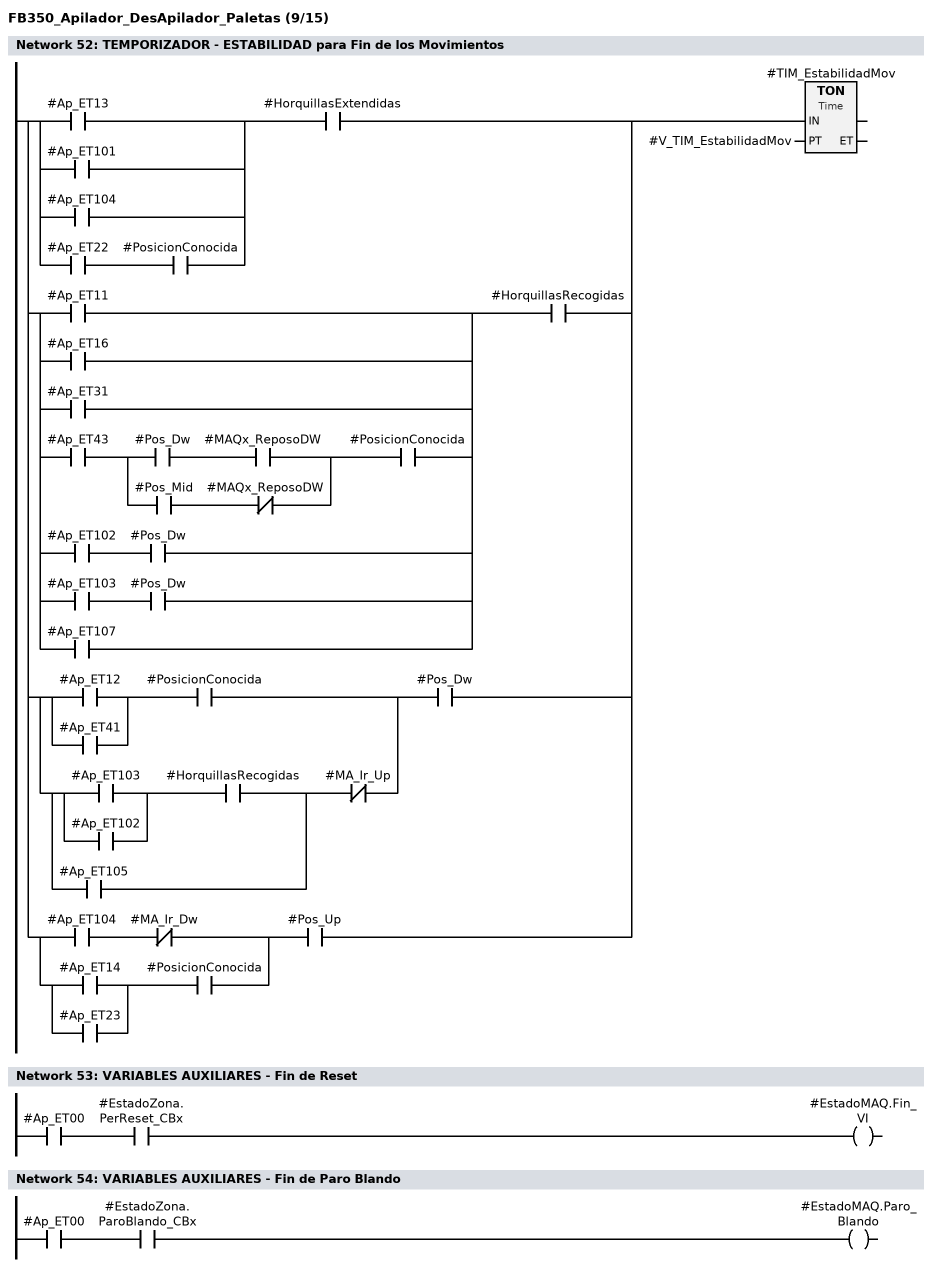
   RUNG wire#powerrail
      Contact( #Ap_ET13 )
      wire#w1
      Contact( #HorquillasExtendidas )
      wire#w2
      { S7_Templates := "time_type := Time" } #TIM_EstabilidadMov.TON(pt := #V_TIM_EstabilidadMov, et =>)
   END_RUNG
   RUNG wire#powerrail
      Contact( #Ap_ET101 )
   END_RUNG wire#w1
   RUNG wire#powerrail
      Contact( #Ap_ET104 )
   END_RUNG wire#w1
   RUNG wire#powerrail
      Contact( #Ap_ET22 )
      Contact( #PosicionConocida )
   END_RUNG wire#w1
   RUNG wire#powerrail
      Contact( #Ap_ET11 )
      wire#w3
      Contact( #HorquillasRecogidas )
   END_RUNG wire#w2
   RUNG wire#powerrail
      Contact( #Ap_ET16 )
   END_RUNG wire#w3
   RUNG wire#powerrail
      Contact( #Ap_ET31 )
   END_RUNG wire#w3
   RUNG wire#powerrail
      Contact( #Ap_ET43 )
      wire#w4
      Contact( #Pos_Dw )
      Contact( #MAQx_ReposoDW )
      wire#w5
      Contact( #PosicionConocida )
   END_RUNG wire#w3
   RUNG wire#w4
      Contact( #Pos_Mid )
      I_Contact( #MAQx_ReposoDW )
   END_RUNG wire#w5
   RUNG wire#powerrail
      Contact( #Ap_ET102 )
      Contact( #Pos_Dw )
   END_RUNG wire#w3
   RUNG wire#powerrail
      Contact( #Ap_ET103 )
      Contact( #Pos_Dw )
   END_RUNG wire#w3
   RUNG wire#powerrail
      Contact( #Ap_ET107 )
   END_RUNG wire#w3
   RUNG wire#powerrail
      Contact( #Ap_ET12 )
      wire#w6
      Contact( #PosicionConocida )
      wire#w7
      Contact( #Pos_Dw )
   END_RUNG wire#w2
   RUNG wire#powerrail
      Contact( #Ap_ET41 )
   END_RUNG wire#w6
   RUNG wire#powerrail
      Contact( #Ap_ET103 )
      wire#w8
      Contact( #HorquillasRecogidas )
      wire#w9
      I_Contact( #MA_Ir_Up )
   END_RUNG wire#w7
   RUNG wire#powerrail
      Contact( #Ap_ET102 )
   END_RUNG wire#w8
   RUNG wire#powerrail
      Contact( #Ap_ET105 )
   END_RUNG wire#w9
   RUNG wire#powerrail
      Contact( #Ap_ET104 )
      I_Contact( #MA_Ir_Dw )
      wire#w10
      Contact( #Pos_Up )
   END_RUNG wire#w2
   RUNG wire#powerrail
      Contact( #Ap_ET14 )
      wire#w11
      Contact( #PosicionConocida )
   END_RUNG wire#w10
   RUNG wire#powerrail
      Contact( #Ap_ET23 )
   END_RUNG wire#w11
   // the same network as SCL:
   #TIM_EstabilidadMov(IN := ((#Ap_ET13 OR #Ap_ET101 OR #Ap_ET104 OR (#Ap_ET22 AND #PosicionConocida)) AND #HorquillasExtendidas) OR ((#Ap_ET11 OR #Ap_ET16 OR #Ap_ET31 OR (#Ap_ET43 AND ((#Pos_Dw AND #MAQx_ReposoDW) OR (#Pos_Mid AND NOT #MAQx_ReposoDW)) AND #PosicionConocida) OR (#Ap_ET102 AND #Pos_Dw) OR (#Ap_ET103 AND #Pos_Dw) OR #Ap_ET107) AND #HorquillasRecogidas) OR ((((#Ap_ET12 OR #Ap_ET41) AND #PosicionConocida) OR ((((#Ap_ET103 OR #Ap_ET102) AND #HorquillasRecogidas) OR #Ap_ET105) AND NOT #MA_Ir_Up)) AND #Pos_Dw) OR (((#Ap_ET104 AND NOT #MA_Ir_Dw) OR ((#Ap_ET14 OR #Ap_ET23) AND #PosicionConocida)) AND #Pos_Up),   // TON
                       PT := #V_TIM_EstabilidadMov);
END_REGION

REGION Network 53: VARIABLES AUXILIARES - Fin de Reset
   RUNG wire#powerrail
      Contact( #Ap_ET00 )
      Contact( #EstadoZona.PerReset_CBx )
      Coil( #EstadoMAQ.Fin_VI )
   END_RUNG
   // the same network as SCL:
   #EstadoMAQ.Fin_VI := #Ap_ET00 AND #EstadoZona.PerReset_CBx;
END_REGION

REGION Network 54: VARIABLES AUXILIARES - Fin de Paro Blando
   RUNG wire#powerrail
      Contact( #Ap_ET00 )
      Contact( #EstadoZona.ParoBlando_CBx )
      Coil( #EstadoMAQ.Paro_Blando )
   END_RUNG
   // the same network as SCL:
   #EstadoMAQ.Paro_Blando := #Ap_ET00 AND #EstadoZona.ParoBlando_CBx;
END_REGION

REGION Network 55: VARIABLES AUXILIARES - Posicion Conocida
   // MODIFICACION DANI: SI MUEVO EN MANUAL NO PIERDE LA POSCION
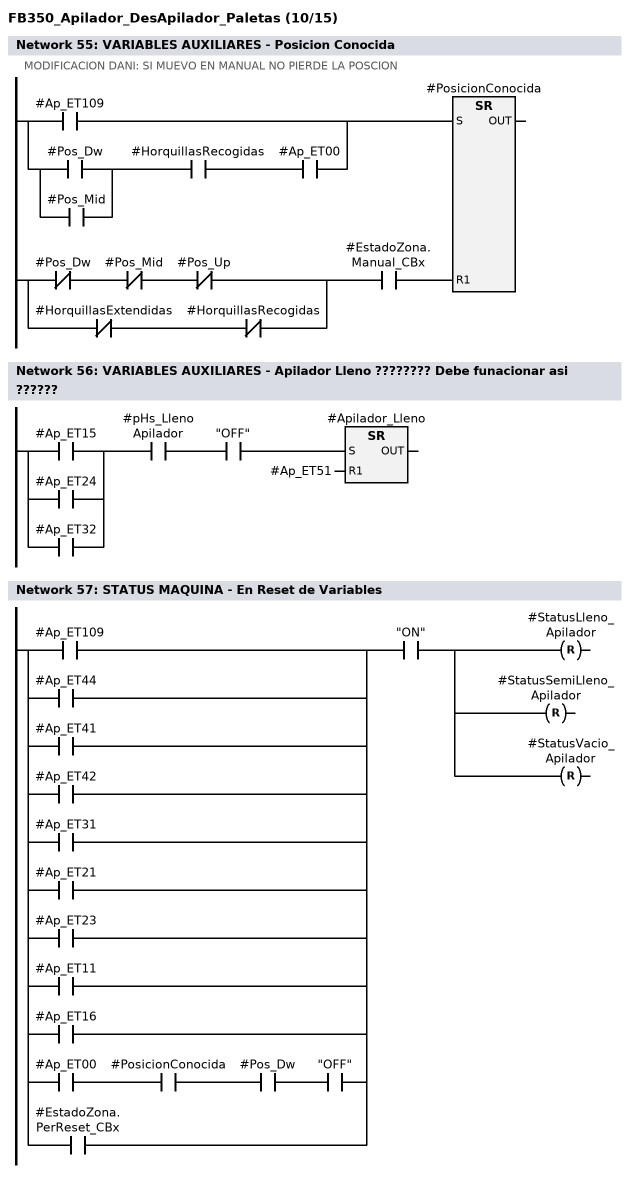
   RUNG wire#powerrail
      Contact( #Ap_ET109 )
      wire#w1
      S_SR(operand := #PosicionConocida, r1 := wire#w4)
   END_RUNG
   RUNG wire#powerrail
      Contact( #Pos_Dw )
      wire#w2
      Contact( #HorquillasRecogidas )
      Contact( #Ap_ET00 )
   END_RUNG wire#w1
   RUNG wire#powerrail
      Contact( #Pos_Mid )
   END_RUNG wire#w2
   RUNG wire#powerrail
      I_Contact( #Pos_Dw )
      I_Contact( #Pos_Mid )
      I_Contact( #Pos_Up )
      wire#w3
      Contact( #EstadoZona.Manual_CBx )
   END_RUNG wire#w4
   RUNG wire#powerrail
      I_Contact( #HorquillasExtendidas )
      I_Contact( #HorquillasRecogidas )
   END_RUNG wire#w3
   // the same network as SCL:
   IF #Ap_ET109 OR ((#Pos_Dw OR #Pos_Mid) AND #HorquillasRecogidas AND #Ap_ET00) THEN
       #PosicionConocida := TRUE;   // SR flip-flop
   END_IF;
   IF ((NOT #Pos_Dw AND NOT #Pos_Mid AND NOT #Pos_Up) OR (NOT #HorquillasExtendidas AND NOT #HorquillasRecogidas)) AND #EstadoZona.Manual_CBx THEN
       #PosicionConocida := FALSE;
   END_IF;
END_REGION

REGION Network 56: VARIABLES AUXILIARES - Apilador Lleno ???????? Debe funacionar asi ??????
   RUNG wire#powerrail
      Contact( #Ap_ET15 )
      wire#w1
      Contact( #pHs_LlenoApilador )
      Contact( "OFF" )
      S_SR(operand := #Apilador_Lleno, r1 := #Ap_ET51)
   END_RUNG
   RUNG wire#powerrail
      Contact( #Ap_ET24 )
   END_RUNG wire#w1
   RUNG wire#powerrail
      Contact( #Ap_ET32 )
   END_RUNG wire#w1
   // the same network as SCL:
   IF (#Ap_ET15 OR #Ap_ET24 OR #Ap_ET32) AND #pHs_LlenoApilador AND "OFF" THEN
       #Apilador_Lleno := TRUE;   // SR flip-flop
   END_IF;
   IF #Ap_ET51 THEN #Apilador_Lleno := FALSE; END_IF;
END_REGION

REGION Network 57: STATUS MAQUINA - En Reset de Variables
   RUNG wire#powerrail
      Contact( #Ap_ET109 )
      wire#w1
      Contact( "ON" )
      wire#w2
      R_Coil( #StatusLleno_Apilador )
   END_RUNG
   RUNG wire#powerrail
      Contact( #Ap_ET44 )
   END_RUNG wire#w1
   RUNG wire#powerrail
      Contact( #Ap_ET41 )
   END_RUNG wire#w1
   RUNG wire#powerrail
      Contact( #Ap_ET42 )
   END_RUNG wire#w1
   RUNG wire#powerrail
      Contact( #Ap_ET31 )
   END_RUNG wire#w1
   RUNG wire#powerrail
      Contact( #Ap_ET21 )
   END_RUNG wire#w1
   RUNG wire#powerrail
      Contact( #Ap_ET23 )
   END_RUNG wire#w1
   RUNG wire#powerrail
      Contact( #Ap_ET11 )
   END_RUNG wire#w1
   RUNG wire#powerrail
      Contact( #Ap_ET16 )
   END_RUNG wire#w1
   RUNG wire#powerrail
      Contact( #Ap_ET00 )
      Contact( #PosicionConocida )
      Contact( #Pos_Dw )
      Contact( "OFF" )
   END_RUNG wire#w1
   RUNG wire#powerrail
      Contact( #EstadoZona.PerReset_CBx )
   END_RUNG wire#w1
   RUNG wire#w2
      R_Coil( #StatusSemiLleno_Apilador )
   END_RUNG
   RUNG wire#w2
      R_Coil( #StatusVacio_Apilador )
   END_RUNG
   // the same network as SCL:
   IF (#Ap_ET109 OR #Ap_ET44 OR #Ap_ET41 OR #Ap_ET42 OR #Ap_ET31 OR #Ap_ET21 OR #Ap_ET23 OR #Ap_ET11 OR #Ap_ET16 OR (#Ap_ET00 AND #PosicionConocida AND #Pos_Dw AND "OFF") OR #EstadoZona.PerReset_CBx) AND "ON" THEN
       #StatusLleno_Apilador := FALSE;
       #StatusSemiLleno_Apilador := FALSE;
       #StatusVacio_Apilador := FALSE;
   END_IF;
END_REGION

REGION Network 58: STATUS MAQUINA - En set de Variables
   // DANI SI ESTA EN ETAPA 0, POS CONOCIDA Y POS REPOSO ACTUALICE EL ESTATUS
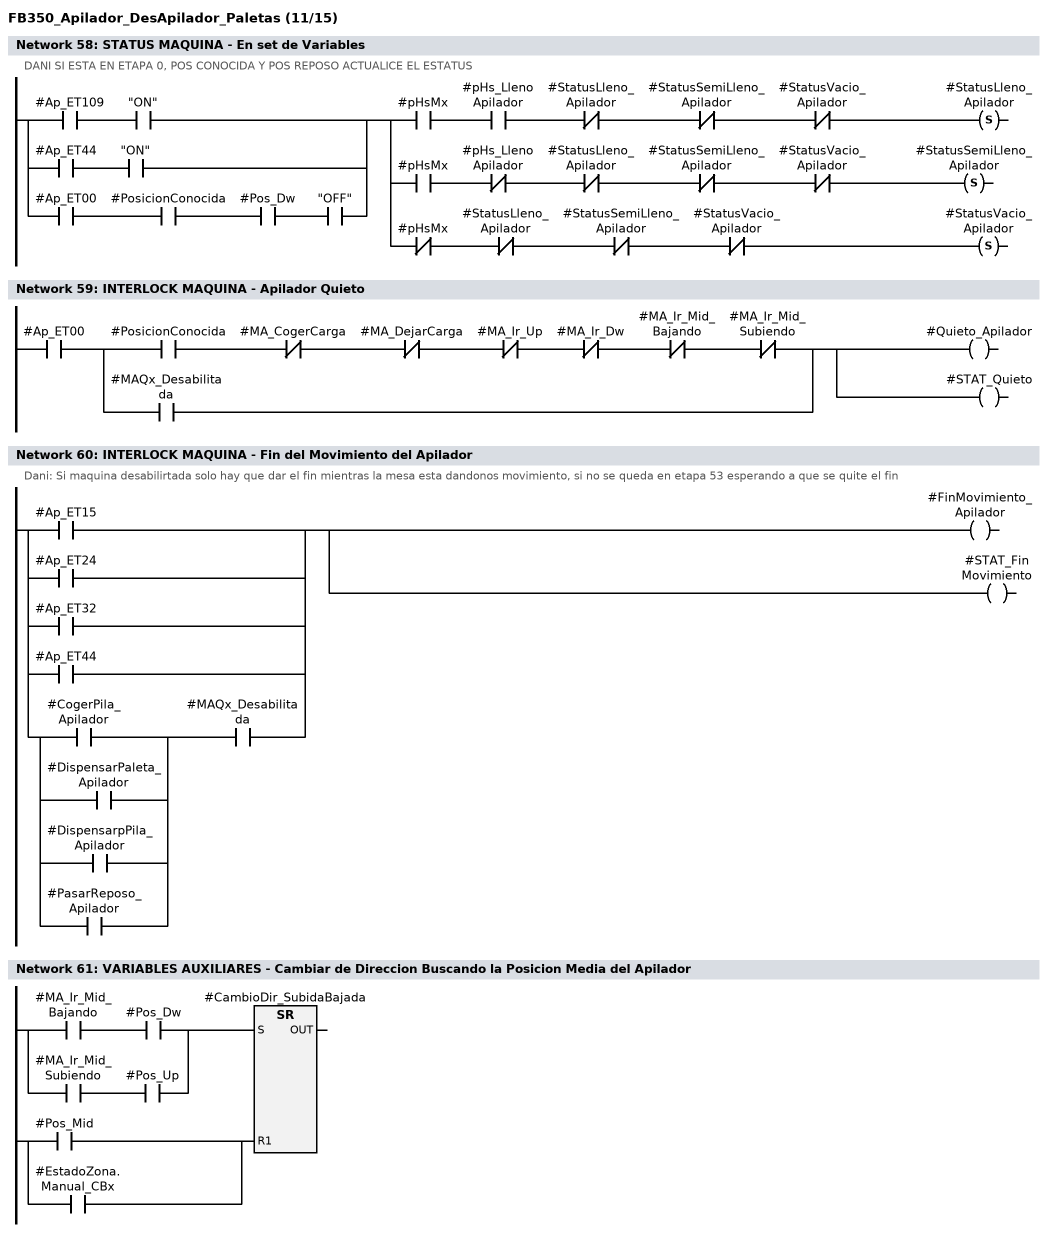
   RUNG wire#powerrail
      Contact( #Ap_ET109 )
      Contact( "ON" )
      wire#w1
      Contact( #pHsMx )
      Contact( #pHs_LlenoApilador )
      I_Contact( #StatusLleno_Apilador )
      I_Contact( #StatusSemiLleno_Apilador )
      I_Contact( #StatusVacio_Apilador )
      S_Coil( #StatusLleno_Apilador )
   END_RUNG
   RUNG wire#powerrail
      Contact( #Ap_ET44 )
      Contact( "ON" )
   END_RUNG wire#w1
   RUNG wire#powerrail
      Contact( #Ap_ET00 )
      Contact( #PosicionConocida )
      Contact( #Pos_Dw )
      Contact( "OFF" )
   END_RUNG wire#w1
   RUNG wire#w1
      Contact( #pHsMx )
      I_Contact( #pHs_LlenoApilador )
      I_Contact( #StatusLleno_Apilador )
      I_Contact( #StatusSemiLleno_Apilador )
      I_Contact( #StatusVacio_Apilador )
      S_Coil( #StatusSemiLleno_Apilador )
   END_RUNG
   RUNG wire#w1
      I_Contact( #pHsMx )
      I_Contact( #StatusLleno_Apilador )
      I_Contact( #StatusSemiLleno_Apilador )
      I_Contact( #StatusVacio_Apilador )
      S_Coil( #StatusVacio_Apilador )
   END_RUNG
   // the same network as SCL:
   #_w1 := (#Ap_ET109 AND "ON") OR (#Ap_ET44 AND "ON") OR (#Ap_ET00 AND #PosicionConocida AND #Pos_Dw AND "OFF");
   IF #_w1 AND #pHsMx AND #pHs_LlenoApilador AND NOT #StatusLleno_Apilador AND NOT #StatusSemiLleno_Apilador AND NOT #StatusVacio_Apilador THEN
       #StatusLleno_Apilador := TRUE;
   END_IF;
   IF #_w1 AND #pHsMx AND NOT #pHs_LlenoApilador AND NOT #StatusLleno_Apilador AND NOT #StatusSemiLleno_Apilador AND NOT #StatusVacio_Apilador THEN
       #StatusSemiLleno_Apilador := TRUE;
   END_IF;
   IF #_w1 AND NOT #pHsMx AND NOT #StatusLleno_Apilador AND NOT #StatusSemiLleno_Apilador AND NOT #StatusVacio_Apilador THEN
       #StatusVacio_Apilador := TRUE;
   END_IF;
END_REGION

REGION Network 59: INTERLOCK MAQUINA - Apilador Quieto
   RUNG wire#powerrail
      Contact( #Ap_ET00 )
      wire#w1
      Contact( #PosicionConocida )
      I_Contact( #MA_CogerCarga )
      I_Contact( #MA_DejarCarga )
      I_Contact( #MA_Ir_Up )
      I_Contact( #MA_Ir_Dw )
      I_Contact( #MA_Ir_Mid_Bajando )
      I_Contact( #MA_Ir_Mid_Subiendo )
      wire#w2
      Coil( #Quieto_Apilador )
   END_RUNG
   RUNG wire#w1
      Contact( #MAQx_Desabilitada )
   END_RUNG wire#w2
   RUNG wire#w2
      Coil( #STAT_Quieto )
   END_RUNG
   // the same network as SCL:
   #Quieto_Apilador := #Ap_ET00 AND ((#PosicionConocida AND NOT #MA_CogerCarga AND NOT #MA_DejarCarga AND NOT #MA_Ir_Up AND NOT #MA_Ir_Dw AND NOT #MA_Ir_Mid_Bajando AND NOT #MA_Ir_Mid_Subiendo) OR #MAQx_Desabilitada);
   #STAT_Quieto := #Quieto_Apilador;
END_REGION

REGION Network 60: INTERLOCK MAQUINA - Fin del Movimiento del Apilador
   // Dani: Si maquina desabilirtada solo hay que dar el fin mientras la mesa esta dandonos movimiento, si no se queda en etapa 53 esperando a que se quite el fin
   RUNG wire#powerrail
      Contact( #Ap_ET15 )
      wire#w1
      Coil( #FinMovimiento_Apilador )
   END_RUNG
   RUNG wire#powerrail
      Contact( #Ap_ET24 )
   END_RUNG wire#w1
   RUNG wire#powerrail
      Contact( #Ap_ET32 )
   END_RUNG wire#w1
   RUNG wire#powerrail
      Contact( #Ap_ET44 )
   END_RUNG wire#w1
   RUNG wire#powerrail
      Contact( #CogerPila_Apilador )
      wire#w2
      Contact( #MAQx_Desabilitada )
   END_RUNG wire#w1
   RUNG wire#powerrail
      Contact( #DispensarPaleta_Apilador )
   END_RUNG wire#w2
   RUNG wire#powerrail
      Contact( #DispensarpPila_Apilador )
   END_RUNG wire#w2
   RUNG wire#powerrail
      Contact( #PasarReposo_Apilador )
   END_RUNG wire#w2
   RUNG wire#w1
      Coil( #STAT_FinMovimiento )
   END_RUNG
   // the same network as SCL:
   #FinMovimiento_Apilador := #Ap_ET15 OR #Ap_ET24 OR #Ap_ET32 OR #Ap_ET44 OR ((#CogerPila_Apilador OR #DispensarPaleta_Apilador OR #DispensarpPila_Apilador OR #PasarReposo_Apilador) AND #MAQx_Desabilitada);
   #STAT_FinMovimiento := #FinMovimiento_Apilador;
END_REGION

REGION Network 61: VARIABLES AUXILIARES - Cambiar de Direccion Buscando la Posicion Media del Apilador
   RUNG wire#powerrail
      Contact( #MA_Ir_Mid_Bajando )
      Contact( #Pos_Dw )
      wire#w1
      S_SR(operand := #CambioDir_SubidaBajada, r1 := wire#w2)
   END_RUNG
   RUNG wire#powerrail
      Contact( #MA_Ir_Mid_Subiendo )
      Contact( #Pos_Up )
   END_RUNG wire#w1
   RUNG wire#powerrail
      Contact( #Pos_Mid )
   END_RUNG wire#w2
   RUNG wire#powerrail
      Contact( #EstadoZona.Manual_CBx )
   END_RUNG wire#w2
   // the same network as SCL:
   IF (#MA_Ir_Mid_Bajando AND #Pos_Dw) OR (#MA_Ir_Mid_Subiendo AND #Pos_Up) THEN
       #CambioDir_SubidaBajada := TRUE;   // SR flip-flop
   END_IF;
   IF #Pos_Mid OR #EstadoZona.Manual_CBx THEN #CambioDir_SubidaBajada := FALSE; END_IF;
END_REGION

REGION Network 62: SALIDAS EXTERIORES - Hoquilla - Coger Carga / Extender 4 Horquillas
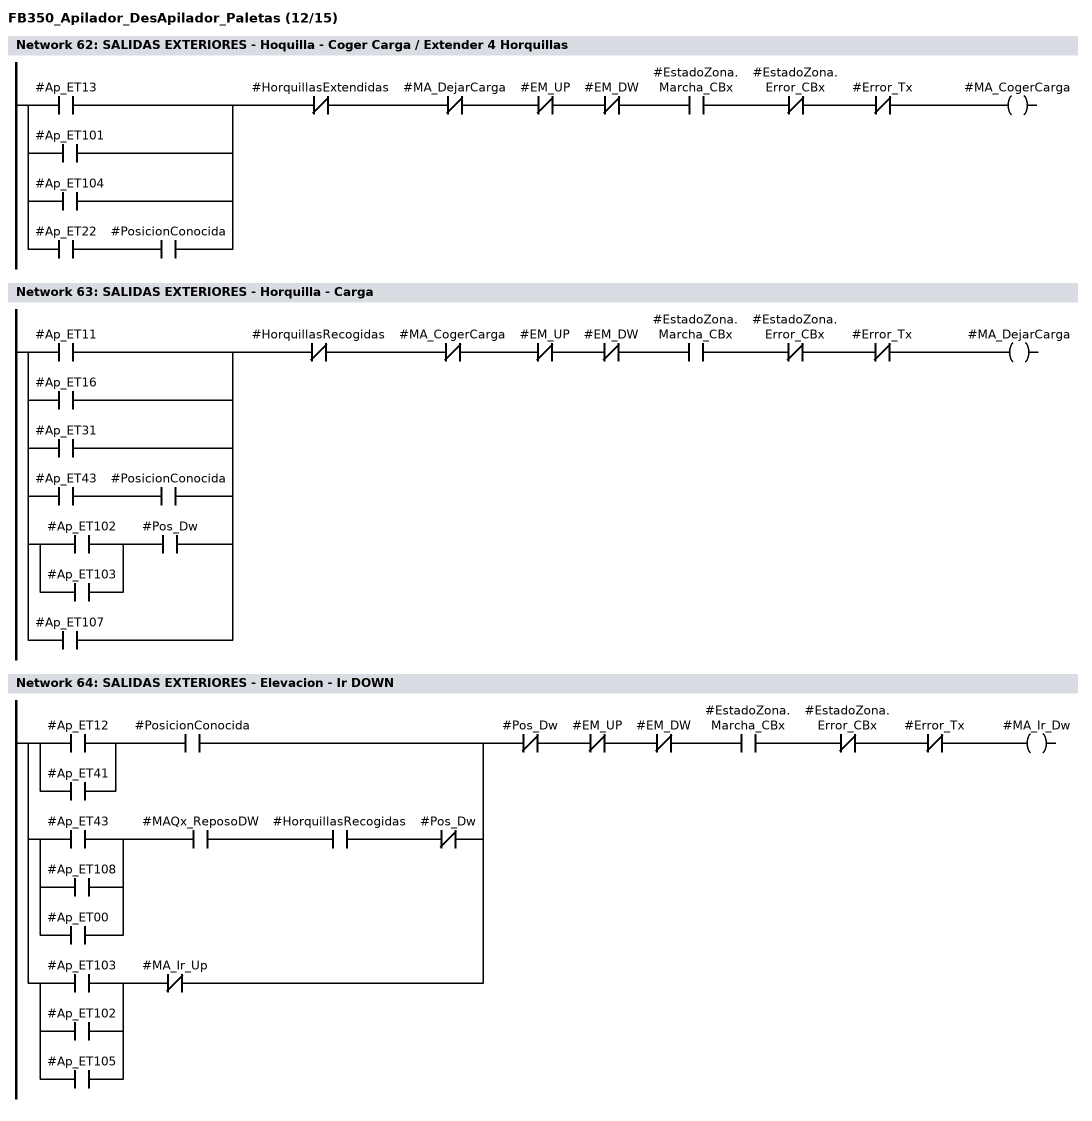
   RUNG wire#powerrail
      Contact( #Ap_ET13 )
      wire#w1
      I_Contact( #HorquillasExtendidas )
      I_Contact( #MA_DejarCarga )
      I_Contact( #EM_UP )
      I_Contact( #EM_DW )
      Contact( #EstadoZona.Marcha_CBx )
      I_Contact( #EstadoZona.Error_CBx )
      I_Contact( #Error_Tx )
      Coil( #MA_CogerCarga )
   END_RUNG
   RUNG wire#powerrail
      Contact( #Ap_ET101 )
   END_RUNG wire#w1
   RUNG wire#powerrail
      Contact( #Ap_ET104 )
   END_RUNG wire#w1
   RUNG wire#powerrail
      Contact( #Ap_ET22 )
      Contact( #PosicionConocida )
   END_RUNG wire#w1
   // the same network as SCL:
   #MA_CogerCarga := (#Ap_ET13 OR #Ap_ET101 OR #Ap_ET104 OR (#Ap_ET22 AND #PosicionConocida)) AND NOT #HorquillasExtendidas AND NOT #MA_DejarCarga AND NOT #EM_UP AND NOT #EM_DW AND #EstadoZona.Marcha_CBx AND NOT #EstadoZona.Error_CBx AND NOT #Error_Tx;
END_REGION

REGION Network 63: SALIDAS EXTERIORES - Horquilla - Carga
   RUNG wire#powerrail
      Contact( #Ap_ET11 )
      wire#w1
      I_Contact( #HorquillasRecogidas )
      I_Contact( #MA_CogerCarga )
      I_Contact( #EM_UP )
      I_Contact( #EM_DW )
      Contact( #EstadoZona.Marcha_CBx )
      I_Contact( #EstadoZona.Error_CBx )
      I_Contact( #Error_Tx )
      Coil( #MA_DejarCarga )
   END_RUNG
   RUNG wire#powerrail
      Contact( #Ap_ET16 )
   END_RUNG wire#w1
   RUNG wire#powerrail
      Contact( #Ap_ET31 )
   END_RUNG wire#w1
   RUNG wire#powerrail
      Contact( #Ap_ET43 )
      Contact( #PosicionConocida )
   END_RUNG wire#w1
   RUNG wire#powerrail
      Contact( #Ap_ET102 )
      wire#w2
      Contact( #Pos_Dw )
   END_RUNG wire#w1
   RUNG wire#powerrail
      Contact( #Ap_ET103 )
   END_RUNG wire#w2
   RUNG wire#powerrail
      Contact( #Ap_ET107 )
   END_RUNG wire#w1
   // the same network as SCL:
   #MA_DejarCarga := (#Ap_ET11 OR #Ap_ET16 OR #Ap_ET31 OR (#Ap_ET43 AND #PosicionConocida) OR ((#Ap_ET102 OR #Ap_ET103) AND #Pos_Dw) OR #Ap_ET107) AND NOT #HorquillasRecogidas AND NOT #MA_CogerCarga AND NOT #EM_UP AND NOT #EM_DW AND #EstadoZona.Marcha_CBx AND NOT #EstadoZona.Error_CBx AND NOT #Error_Tx;
END_REGION

REGION Network 64: SALIDAS EXTERIORES - Elevacion - Ir DOWN
   RUNG wire#powerrail
      Contact( #Ap_ET12 )
      wire#w1
      Contact( #PosicionConocida )
      wire#w2
      I_Contact( #Pos_Dw )
      I_Contact( #EM_UP )
      I_Contact( #EM_DW )
      Contact( #EstadoZona.Marcha_CBx )
      I_Contact( #EstadoZona.Error_CBx )
      I_Contact( #Error_Tx )
      Coil( #MA_Ir_Dw )
   END_RUNG
   RUNG wire#powerrail
      Contact( #Ap_ET41 )
   END_RUNG wire#w1
   RUNG wire#powerrail
      Contact( #Ap_ET43 )
      wire#w3
      Contact( #MAQx_ReposoDW )
      Contact( #HorquillasRecogidas )
      I_Contact( #Pos_Dw )
   END_RUNG wire#w2
   RUNG wire#powerrail
      Contact( #Ap_ET108 )
   END_RUNG wire#w3
   RUNG wire#powerrail
      Contact( #Ap_ET00 )
   END_RUNG wire#w3
   RUNG wire#powerrail
      Contact( #Ap_ET103 )
      wire#w4
      I_Contact( #MA_Ir_Up )
   END_RUNG wire#w2
   RUNG wire#powerrail
      Contact( #Ap_ET102 )
   END_RUNG wire#w4
   RUNG wire#powerrail
      Contact( #Ap_ET105 )
   END_RUNG wire#w4
   // the same network as SCL:
   #MA_Ir_Dw := (((#Ap_ET12 OR #Ap_ET41) AND #PosicionConocida) OR ((#Ap_ET43 OR #Ap_ET108 OR #Ap_ET00) AND #MAQx_ReposoDW AND #HorquillasRecogidas AND NOT #Pos_Dw) OR ((#Ap_ET103 OR #Ap_ET102 OR #Ap_ET105) AND NOT #MA_Ir_Up)) AND NOT #Pos_Dw AND NOT #EM_UP AND NOT #EM_DW AND #EstadoZona.Marcha_CBx AND NOT #EstadoZona.Error_CBx AND NOT #Error_Tx;
END_REGION

REGION Network 65: SALIDAS EXTERIORES - Elevacion - Ir MID Bajando
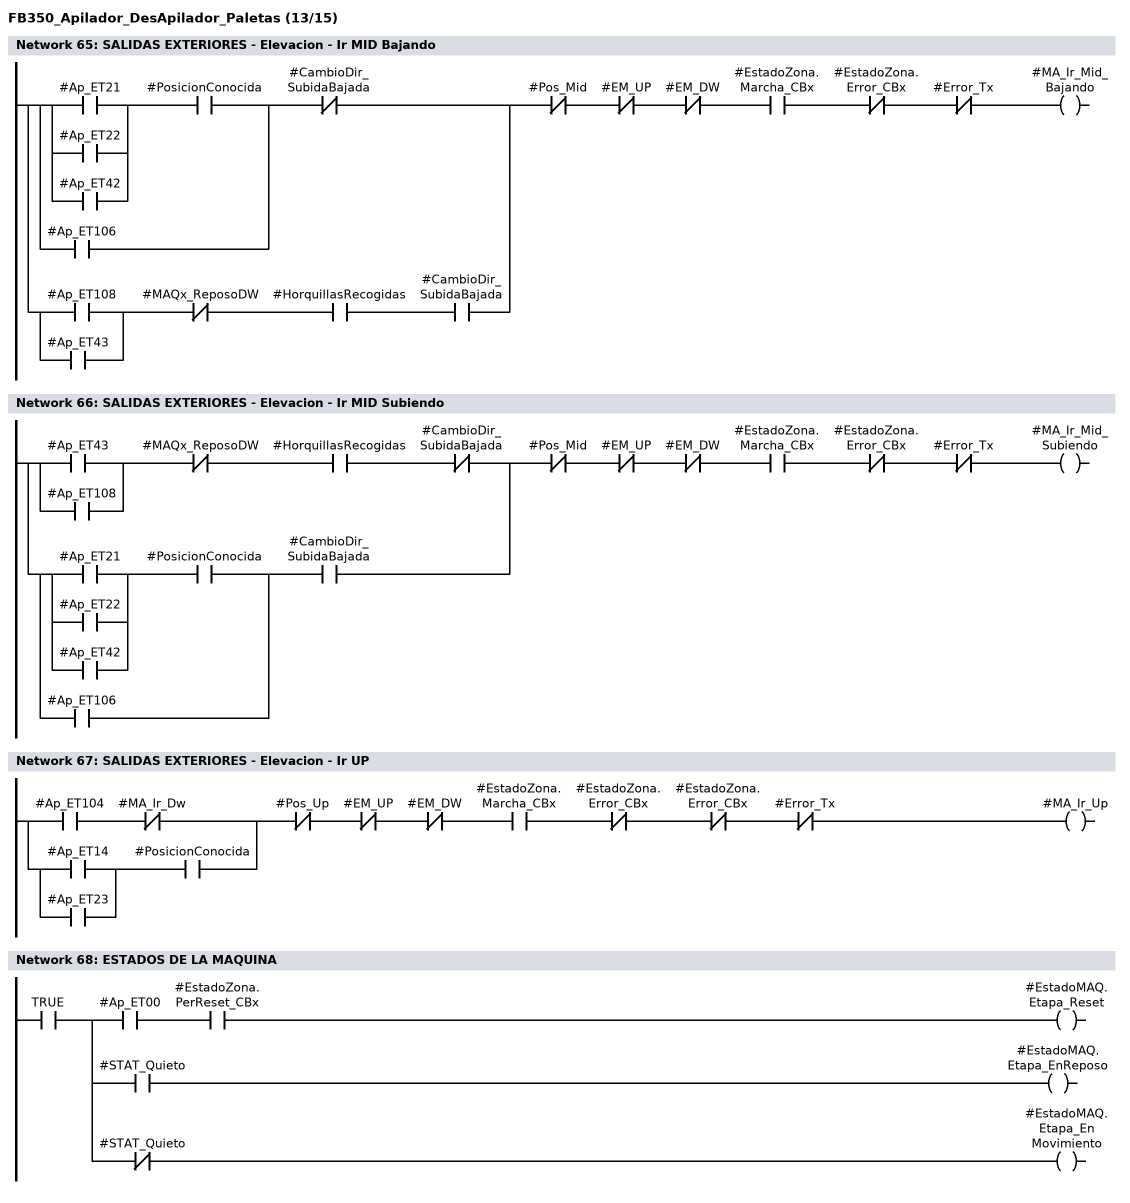
   RUNG wire#powerrail
      Contact( #Ap_ET21 )
      wire#w1
      Contact( #PosicionConocida )
      wire#w2
      I_Contact( #CambioDir_SubidaBajada )
      wire#w3
      I_Contact( #Pos_Mid )
      I_Contact( #EM_UP )
      I_Contact( #EM_DW )
      Contact( #EstadoZona.Marcha_CBx )
      I_Contact( #EstadoZona.Error_CBx )
      I_Contact( #Error_Tx )
      Coil( #MA_Ir_Mid_Bajando )
   END_RUNG
   RUNG wire#powerrail
      Contact( #Ap_ET22 )
   END_RUNG wire#w1
   RUNG wire#powerrail
      Contact( #Ap_ET42 )
   END_RUNG wire#w1
   RUNG wire#powerrail
      Contact( #Ap_ET106 )
   END_RUNG wire#w2
   RUNG wire#powerrail
      Contact( #Ap_ET108 )
      wire#w4
      I_Contact( #MAQx_ReposoDW )
      Contact( #HorquillasRecogidas )
      Contact( #CambioDir_SubidaBajada )
   END_RUNG wire#w3
   RUNG wire#powerrail
      Contact( #Ap_ET43 )
   END_RUNG wire#w4
   // the same network as SCL:
   #MA_Ir_Mid_Bajando := (((((#Ap_ET21 OR #Ap_ET22 OR #Ap_ET42) AND #PosicionConocida) OR #Ap_ET106) AND NOT #CambioDir_SubidaBajada) OR ((#Ap_ET108 OR #Ap_ET43) AND NOT #MAQx_ReposoDW AND #HorquillasRecogidas AND #CambioDir_SubidaBajada)) AND NOT #Pos_Mid AND NOT #EM_UP AND NOT #EM_DW AND #EstadoZona.Marcha_CBx AND NOT #EstadoZona.Error_CBx AND NOT #Error_Tx;
END_REGION

REGION Network 66: SALIDAS EXTERIORES - Elevacion - Ir MID Subiendo
   RUNG wire#powerrail
      Contact( #Ap_ET43 )
      wire#w1
      I_Contact( #MAQx_ReposoDW )
      Contact( #HorquillasRecogidas )
      I_Contact( #CambioDir_SubidaBajada )
      wire#w2
      I_Contact( #Pos_Mid )
      I_Contact( #EM_UP )
      I_Contact( #EM_DW )
      Contact( #EstadoZona.Marcha_CBx )
      I_Contact( #EstadoZona.Error_CBx )
      I_Contact( #Error_Tx )
      Coil( #MA_Ir_Mid_Subiendo )
   END_RUNG
   RUNG wire#powerrail
      Contact( #Ap_ET108 )
   END_RUNG wire#w1
   RUNG wire#powerrail
      Contact( #Ap_ET21 )
      wire#w3
      Contact( #PosicionConocida )
      wire#w4
      Contact( #CambioDir_SubidaBajada )
   END_RUNG wire#w2
   RUNG wire#powerrail
      Contact( #Ap_ET22 )
   END_RUNG wire#w3
   RUNG wire#powerrail
      Contact( #Ap_ET42 )
   END_RUNG wire#w3
   RUNG wire#powerrail
      Contact( #Ap_ET106 )
   END_RUNG wire#w4
   // the same network as SCL:
   #MA_Ir_Mid_Subiendo := (((#Ap_ET43 OR #Ap_ET108) AND NOT #MAQx_ReposoDW AND #HorquillasRecogidas AND NOT #CambioDir_SubidaBajada) OR ((((#Ap_ET21 OR #Ap_ET22 OR #Ap_ET42) AND #PosicionConocida) OR #Ap_ET106) AND #CambioDir_SubidaBajada)) AND NOT #Pos_Mid AND NOT #EM_UP AND NOT #EM_DW AND #EstadoZona.Marcha_CBx AND NOT #EstadoZona.Error_CBx AND NOT #Error_Tx;
END_REGION

REGION Network 67: SALIDAS EXTERIORES - Elevacion - Ir UP
   RUNG wire#powerrail
      Contact( #Ap_ET104 )
      I_Contact( #MA_Ir_Dw )
      wire#w1
      I_Contact( #Pos_Up )
      I_Contact( #EM_UP )
      I_Contact( #EM_DW )
      Contact( #EstadoZona.Marcha_CBx )
      I_Contact( #EstadoZona.Error_CBx )
      I_Contact( #EstadoZona.Error_CBx )
      I_Contact( #Error_Tx )
      Coil( #MA_Ir_Up )
   END_RUNG
   RUNG wire#powerrail
      Contact( #Ap_ET14 )
      wire#w2
      Contact( #PosicionConocida )
   END_RUNG wire#w1
   RUNG wire#powerrail
      Contact( #Ap_ET23 )
   END_RUNG wire#w2
   // the same network as SCL:
   #MA_Ir_Up := ((#Ap_ET104 AND NOT #MA_Ir_Dw) OR ((#Ap_ET14 OR #Ap_ET23) AND #PosicionConocida)) AND NOT #Pos_Up AND NOT #EM_UP AND NOT #EM_DW AND #EstadoZona.Marcha_CBx AND NOT #EstadoZona.Error_CBx AND NOT #EstadoZona.Error_CBx AND NOT #Error_Tx;
END_REGION

REGION Network 68: ESTADOS DE LA MAQUINA
   RUNG wire#powerrail
      Contact( TRUE )
      wire#w1
      Contact( #Ap_ET00 )
      Contact( #EstadoZona.PerReset_CBx )
      Coil( #EstadoMAQ.Etapa_Reset )
   END_RUNG
   RUNG wire#w1
      Contact( #STAT_Quieto )
      Coil( #EstadoMAQ.Etapa_EnReposo )
   END_RUNG
   RUNG wire#w1
      I_Contact( #STAT_Quieto )
      Coil( #EstadoMAQ.Etapa_EnMovimiento )
   END_RUNG
   // the same network as SCL:
   #EstadoMAQ.Etapa_Reset := TRUE AND #Ap_ET00 AND #EstadoZona.PerReset_CBx;
   #EstadoMAQ.Etapa_EnReposo := TRUE AND #STAT_Quieto;
   #EstadoMAQ.Etapa_EnMovimiento := TRUE AND NOT #STAT_Quieto;
END_REGION

REGION Network 69: ENTRADAS DE LA MAQUINA
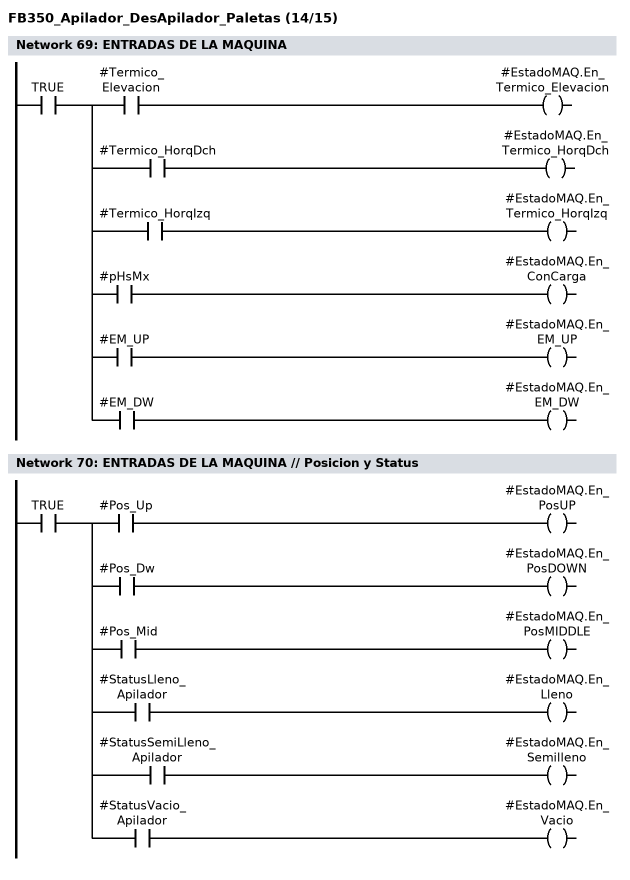
   RUNG wire#powerrail
      Contact( TRUE )
      wire#w1
      Contact( #Termico_Elevacion )
      Coil( #EstadoMAQ.En_Termico_Elevacion )
   END_RUNG
   RUNG wire#w1
      Contact( #Termico_HorqDch )
      Coil( #EstadoMAQ.En_Termico_HorqDch )
   END_RUNG
   RUNG wire#w1
      Contact( #Termico_HorqIzq )
      Coil( #EstadoMAQ.En_Termico_HorqIzq )
   END_RUNG
   RUNG wire#w1
      Contact( #pHsMx )
      Coil( #EstadoMAQ.En_ConCarga )
   END_RUNG
   RUNG wire#w1
      Contact( #EM_UP )
      Coil( #EstadoMAQ.En_EM_UP )
   END_RUNG
   RUNG wire#w1
      Contact( #EM_DW )
      Coil( #EstadoMAQ.En_EM_DW )
   END_RUNG
   // the same network as SCL:
   #EstadoMAQ.En_Termico_Elevacion := TRUE AND #Termico_Elevacion;
   #EstadoMAQ.En_Termico_HorqDch := TRUE AND #Termico_HorqDch;
   #EstadoMAQ.En_Termico_HorqIzq := TRUE AND #Termico_HorqIzq;
   #EstadoMAQ.En_ConCarga := TRUE AND #pHsMx;
   #EstadoMAQ.En_EM_UP := TRUE AND #EM_UP;
   #EstadoMAQ.En_EM_DW := TRUE AND #EM_DW;
END_REGION

REGION Network 70: ENTRADAS DE LA MAQUINA // Posicion y Status
   RUNG wire#powerrail
      Contact( TRUE )
      wire#w1
      Contact( #Pos_Up )
      Coil( #EstadoMAQ.En_PosUP )
   END_RUNG
   RUNG wire#w1
      Contact( #Pos_Dw )
      Coil( #EstadoMAQ.En_PosDOWN )
   END_RUNG
   RUNG wire#w1
      Contact( #Pos_Mid )
      Coil( #EstadoMAQ.En_PosMIDDLE )
   END_RUNG
   RUNG wire#w1
      Contact( #StatusLleno_Apilador )
      Coil( #EstadoMAQ.En_Lleno )
   END_RUNG
   RUNG wire#w1
      Contact( #StatusSemiLleno_Apilador )
      Coil( #EstadoMAQ.En_Semilleno )
   END_RUNG
   RUNG wire#w1
      Contact( #StatusVacio_Apilador )
      Coil( #EstadoMAQ.En_Vacio )
   END_RUNG
   // the same network as SCL:
   #EstadoMAQ.En_PosUP := TRUE AND #Pos_Up;
   #EstadoMAQ.En_PosDOWN := TRUE AND #Pos_Dw;
   #EstadoMAQ.En_PosMIDDLE := TRUE AND #Pos_Mid;
   #EstadoMAQ.En_Lleno := TRUE AND #StatusLleno_Apilador;
   #EstadoMAQ.En_Semilleno := TRUE AND #StatusSemiLleno_Apilador;
   #EstadoMAQ.En_Vacio := TRUE AND #StatusVacio_Apilador;
END_REGION

REGION Network 71: ENTRADAS DE LA MAQUINA // Sensores de las horquillas
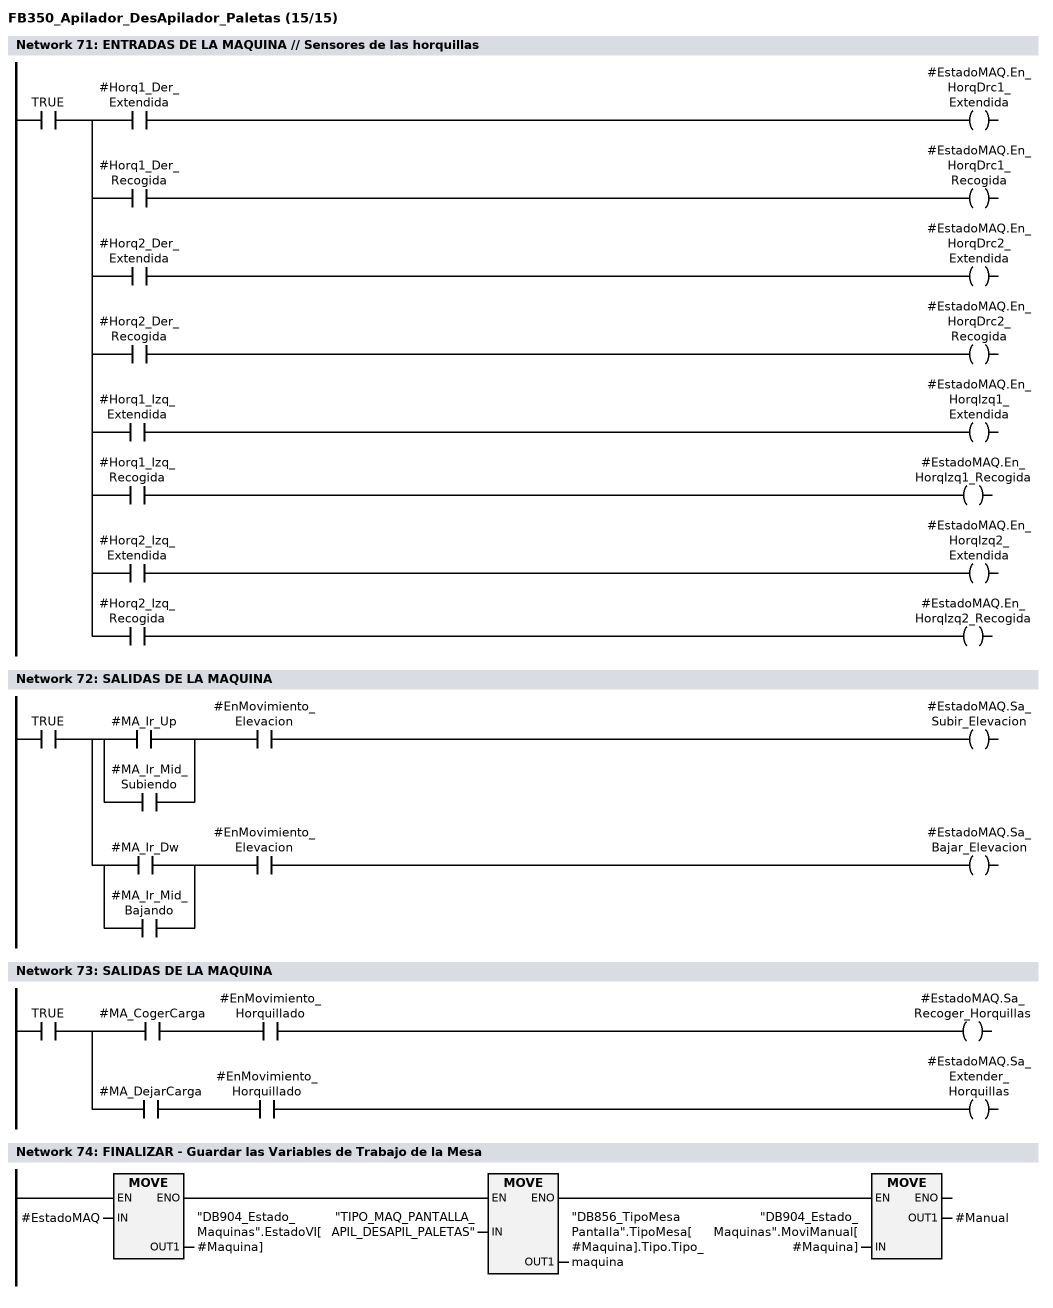
   RUNG wire#powerrail
      Contact( TRUE )
      wire#w1
      Contact( #Horq1_Der_Extendida )
      Coil( #EstadoMAQ.En_HorqDrc1_Extendida )
   END_RUNG
   RUNG wire#w1
      Contact( #Horq1_Der_Recogida )
      Coil( #EstadoMAQ.En_HorqDrc1_Recogida )
   END_RUNG
   RUNG wire#w1
      Contact( #Horq2_Der_Extendida )
      Coil( #EstadoMAQ.En_HorqDrc2_Extendida )
   END_RUNG
   RUNG wire#w1
      Contact( #Horq2_Der_Recogida )
      Coil( #EstadoMAQ.En_HorqDrc2_Recogida )
   END_RUNG
   RUNG wire#w1
      Contact( #Horq1_Izq_Extendida )
      Coil( #EstadoMAQ.En_HorqIzq1_Extendida )
   END_RUNG
   RUNG wire#w1
      Contact( #Horq1_Izq_Recogida )
      Coil( #EstadoMAQ.En_HorqIzq1_Recogida )
   END_RUNG
   RUNG wire#w1
      Contact( #Horq2_Izq_Extendida )
      Coil( #EstadoMAQ.En_HorqIzq2_Extendida )
   END_RUNG
   RUNG wire#w1
      Contact( #Horq2_Izq_Recogida )
      Coil( #EstadoMAQ.En_HorqIzq2_Recogida )
   END_RUNG
   // the same network as SCL:
   #EstadoMAQ.En_HorqDrc1_Extendida := TRUE AND #Horq1_Der_Extendida;
   #EstadoMAQ.En_HorqDrc1_Recogida := TRUE AND #Horq1_Der_Recogida;
   #EstadoMAQ.En_HorqDrc2_Extendida := TRUE AND #Horq2_Der_Extendida;
   #EstadoMAQ.En_HorqDrc2_Recogida := TRUE AND #Horq2_Der_Recogida;
   #EstadoMAQ.En_HorqIzq1_Extendida := TRUE AND #Horq1_Izq_Extendida;
   #EstadoMAQ.En_HorqIzq1_Recogida := TRUE AND #Horq1_Izq_Recogida;
   #EstadoMAQ.En_HorqIzq2_Extendida := TRUE AND #Horq2_Izq_Extendida;
   #EstadoMAQ.En_HorqIzq2_Recogida := TRUE AND #Horq2_Izq_Recogida;
END_REGION

REGION Network 72: SALIDAS DE LA MAQUINA
   RUNG wire#powerrail
      Contact( TRUE )
      wire#w1
      Contact( #MA_Ir_Up )
      wire#w2
      Contact( #EnMovimiento_Elevacion )
      Coil( #EstadoMAQ.Sa_Subir_Elevacion )
   END_RUNG
   RUNG wire#w1
      Contact( #MA_Ir_Mid_Subiendo )
   END_RUNG wire#w2
   RUNG wire#w1
      Contact( #MA_Ir_Dw )
      wire#w3
      Contact( #EnMovimiento_Elevacion )
      Coil( #EstadoMAQ.Sa_Bajar_Elevacion )
   END_RUNG
   RUNG wire#w1
      Contact( #MA_Ir_Mid_Bajando )
   END_RUNG wire#w3
   // the same network as SCL:
   #EstadoMAQ.Sa_Subir_Elevacion := TRUE AND (#MA_Ir_Up OR #MA_Ir_Mid_Subiendo) AND #EnMovimiento_Elevacion;
   #EstadoMAQ.Sa_Bajar_Elevacion := TRUE AND (#MA_Ir_Dw OR #MA_Ir_Mid_Bajando) AND #EnMovimiento_Elevacion;
END_REGION

REGION Network 73: SALIDAS DE LA MAQUINA
   RUNG wire#powerrail
      Contact( TRUE )
      wire#w1
      Contact( #MA_CogerCarga )
      Contact( #EnMovimiento_Horquillado )
      Coil( #EstadoMAQ.Sa_Recoger_Horquillas )
   END_RUNG
   RUNG wire#w1
      Contact( #MA_DejarCarga )
      Contact( #EnMovimiento_Horquillado )
      Coil( #EstadoMAQ.Sa_Extender_Horquillas )
   END_RUNG
   // the same network as SCL:
   #EstadoMAQ.Sa_Recoger_Horquillas := TRUE AND #MA_CogerCarga AND #EnMovimiento_Horquillado;
   #EstadoMAQ.Sa_Extender_Horquillas := TRUE AND #MA_DejarCarga AND #EnMovimiento_Horquillado;
END_REGION

REGION Network 74: FINALIZAR - Guardar las Variables de Trabajo de la Mesa
   RUNG wire#powerrail
      Move(in := #EstadoMAQ, out1 => "DB904_Estado_Maquinas".EstadoVI[#Maquina])
      Move(in := "TIPO_MAQ_PANTALLA_APIL_DESAPIL_PALETAS", out1 => "DB856_TipoMesaPantalla".TipoMesa[#Maquina].Tipo.Tipo_maquina)
      Move(in := "DB904_Estado_Maquinas".MoviManual[#Maquina], out1 => #Manual)
   END_RUNG
   // the same network as SCL:
   "DB904_Estado_Maquinas".EstadoVI[#Maquina] := #EstadoMAQ;
   "DB856_TipoMesaPantalla".TipoMesa[#Maquina].Tipo.Tipo_maquina := "TIPO_MAQ_PANTALLA_APIL_DESAPIL_PALETAS";
   #Manual := "DB904_Estado_Maquinas".MoviManual[#Maquina];
END_REGION
END_FUNCTION_BLOCK

FUNCTION_BLOCK "FB351_DesRemontador_Remontador_Horquilla"   // FB351, LAD
TITLE = Control del Ramal de Salidas
{ S7_Optimized_Access := 'FALSE' }
AUTHOR : REFORMAR
NAME : 20160211
VERSION : 3.1
// Dani Palacios: Modificación octubre 2017 para poder desabilitar la maquina con un bit (por ejemplo en la puesta a punto si no esta montada o en el simulador)
// La modificación esta sin probar y es todo lo relativo a la variable Maquina_Desabilitada
// (bloqueo evolución desde etapa 0, bloqueo activación salidas en etapa 0 , fin vi sin mirar detectores y activación posición de reposo sin mirar detectores y variabkles de fin de movimiento).
// ES RESPONSABILIDAD DEL QUE DESABILITA LA MAQUINA QUE ESTA ESTE EN UNA POSICION QUE PERMITA EL MOVIMIENTO DE LAS CARGAS A TRAVES DE ELLA
// stored: AutoNumber false, SetENOAutomatically false
   VAR_INPUT
      Maquina : UInt;   // Numero de Maquina (Mesa)
      Error_Tx : Bool;   // Error en el Tx
      EnTension : Bool;   // Existe Tension en la Mesa
      MAQx_Desabilitada : Bool;   // Config MAQ. >>> DesHabilitada
      TipoPaleta : Bool;   // Si 1, EUR. Si 0, medio paleta
      Termico_Elevacion : Bool;   // Termico de la Elevacion
      Termico_Horquilla : Bool;   // Termico de la Horquilla
      ParElevacion_ErrorRotura : Bool;
      pHsMx : Bool;   // pHs de la Mesa
      EnMovimiento_Tx : Bool;   // En Movimiento Tx
      ELEV_SegUp : Bool;   // ELEV >> Seguridad Up
      ELEV_SegDw : Bool;   // ELEV >> Seguridad Down
      ELEV_PosUp : Bool;   // ELEV >> Posicion Up
      ELEV_PosMid : Bool;   // ELEV >> Posicion Midle
      ELEV_PosDw : Bool;   // ELEV >> Posicion Down
      ELEV_EnMovimiento : Bool;   // ELEV >> En Movimiento
      HORQ_SegRecogida : Bool;   // HORQ >> Seguridad Atras
      HORQ_SegExtendida : Bool;   // HORQ >> Seguridad Adelante
      HORQ_Recogida : Bool;   // HORQ >> Posicion Atras
      HORQ_Medio : Bool;   // HORQ >> Posicion Medio
      HORQ_Extendida : Bool;   // HORQ >> Posicion Adelante
      HORQ_CV_Recogida : Bool;   // HORQ >> Cambio de Velocidad Atras
      HORQ_CV_Medio : Bool;   // HORQ >> Cambio de Velocidad Medio
      HORQ_CV_Extendida : Bool;   // HORQ >> Cambio de Velocidad Adelante
      HORQ_EnMovimiento : Bool;   // HORQ >> En Movimiento
      Elev_Carga_OK : Bool;
      RH_PasarReposo : Bool;   // Interlock >> Pasar a Reposo
      RH_SubirPaleta : Bool;   // Interlock >> Subir Paleta
      RH_DejarPaleta : Bool;   // Interlock >> Dejar Paleta
      RH_RemontarPaleta : Bool;   // Interlock >> Remontar Paleta
      RH_DesRemontarPaleta : Bool;   // Interlock >> DesRemontar Paleta
      V_TIM_EstabilidadMov : Time;   // TIM de Estabilidad de los Mov.
      V_TOut_Elevacion : Int := 7000;   // TimeOut del Mov. de Elevacion
      V_TOut_Horquillado : Int := 7000;   // TimeOut del Mov. de Horquillado
   END_VAR
   VAR_OUTPUT
      RH_Quieto : Bool;   // Interlock >> Quieto
      RH_FinMovimiento : Bool;   // Interlock >> Fin del Movimiento
   END_VAR
   VAR
      Rh_ET00 : Bool;
      Rh_ET100 : Bool;
      Rh_ET101 : Bool;
      Rh_ET102 : Bool;
      Rh_ET103 : Bool;
      Rh_ET104 : Bool;
      Rh_ET105 : Bool;
      Rh_ET106 : Bool;
      Rh_ET107 : Bool;
      Rh_ET108 : Bool;
      Rh_ET109 : Bool;
      Rh_ET11 : Bool;
      Rh_ET12 : Bool;
      Rh_ET13 : Bool;
      Rh_ET14 : Bool;
      Rh_ET15 : Bool;
      Rh_ET16 : Bool;
      Rh_ET21 : Bool;
      Rh_ET22 : Bool;
      Rh_ET23 : Bool;
      Rh_ET24 : Bool;
      Rh_ET31 : Bool;
      Rh_ET32 : Bool;
      Rh_ET41 : Bool;
      Rh_ET42 : Bool;
      Rh_ET43 : Bool;
      Rh_ET44 : Bool;
      Rh_ET51 : Bool;
      Rh_ET52 : Bool;
      Rh_ET53 : Bool;
      PosicionConocida : Bool;
      STAT_Quieto : Bool;   // Interna >> Quieto la Maquina
      STAT_FinMovimiento : Bool;   // Interna >> Fin de Movimiento
      CambioDir_SubidaBajada : Bool;   // Interna >> Cambio de Dir. Subida o Bajada
      MA_Ir_Up : Bool;
      MA_Ir_Dw : Bool;
      MA_Ir_Mid_Bajando : Bool;
      MA_Ir_Mid_Subiendo : Bool;
      MA_Ir_Adelante : Bool;
      MA_Ir_Atras : Bool;
      HORQ_VelocidadRapida : Bool;
      TIM_EstabilidadMov { S7_SetPoint := 'True'} : TON_TIME;
      TMP_EnTension { S7_SetPoint := 'True'} : "FB910_CNT_UHS";
      TOut_Elevacion { S7_SetPoint := 'True'} : "FB910_CNT_UHS";
      TOut_Horquillado { S7_SetPoint := 'True'} : "FB910_CNT_UHS";
      Manual : "MoviManualMaquina_Remontador";
   END_VAR
   VAR_TEMP
      EstadoZona : "EstadoZona";   // Estado de Zona de la Mesa
      EstadoMAQ : "EstadoMaquina_Remontador";   // Estado del Vehiculo Inteliguente de la Maquina
      Aux_ET00 : Bool;
   END_VAR
BEGIN

REGION Network 1: INICIALIZAR - Recoger las Variables de Estado de la Maquina
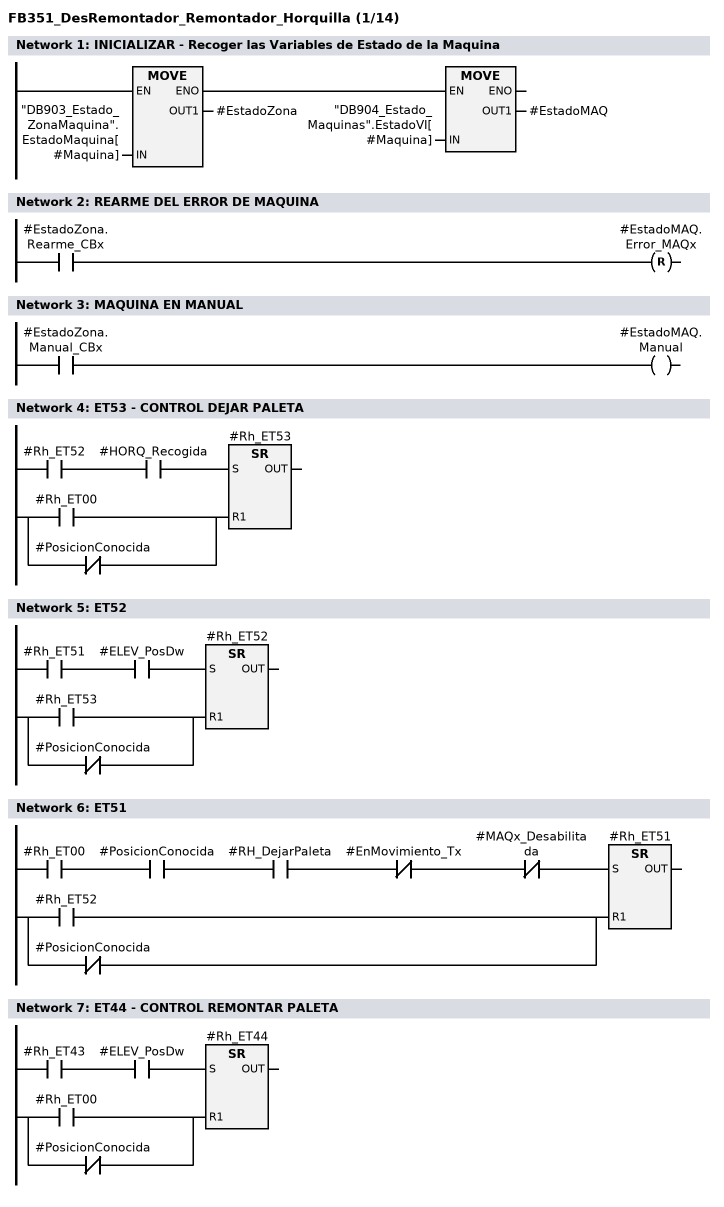
   RUNG wire#powerrail
      Move(in := "DB903_Estado_ZonaMaquina".EstadoMaquina[#Maquina], out1 => #EstadoZona)
      Move(in := "DB904_Estado_Maquinas".EstadoVI[#Maquina], out1 => #EstadoMAQ)
   END_RUNG
   // the same network as SCL:
   #EstadoZona := "DB903_Estado_ZonaMaquina".EstadoMaquina[#Maquina];
   #EstadoMAQ := "DB904_Estado_Maquinas".EstadoVI[#Maquina];
END_REGION

REGION Network 2: REARME DEL ERROR DE MAQUINA
   RUNG wire#powerrail
      Contact( #EstadoZona.Rearme_CBx )
      R_Coil( #EstadoMAQ.Error_MAQx )
   END_RUNG
   // the same network as SCL:
   IF #EstadoZona.Rearme_CBx THEN #EstadoMAQ.Error_MAQx := FALSE; END_IF;
END_REGION

REGION Network 3: MAQUINA EN MANUAL
   RUNG wire#powerrail
      Contact( #EstadoZona.Manual_CBx )
      Coil( #EstadoMAQ.Manual )
   END_RUNG
   // the same network as SCL:
   #EstadoMAQ.Manual := #EstadoZona.Manual_CBx;
END_REGION

REGION Network 4: ET53 - CONTROL DEJAR PALETA
   RUNG wire#powerrail
      Contact( #Rh_ET52 )
      Contact( #HORQ_Recogida )
      S_SR(operand := #Rh_ET53, r1 := wire#w1)
   END_RUNG
   RUNG wire#powerrail
      Contact( #Rh_ET00 )
   END_RUNG wire#w1
   RUNG wire#powerrail
      I_Contact( #PosicionConocida )
   END_RUNG wire#w1
   // the same network as SCL:
   IF #Rh_ET52 AND #HORQ_Recogida THEN
       #Rh_ET53 := TRUE;   // SR flip-flop
   END_IF;
   IF #Rh_ET00 OR NOT #PosicionConocida THEN #Rh_ET53 := FALSE; END_IF;
END_REGION

REGION Network 5: ET52
   RUNG wire#powerrail
      Contact( #Rh_ET51 )
      Contact( #ELEV_PosDw )
      S_SR(operand := #Rh_ET52, r1 := wire#w1)
   END_RUNG
   RUNG wire#powerrail
      Contact( #Rh_ET53 )
   END_RUNG wire#w1
   RUNG wire#powerrail
      I_Contact( #PosicionConocida )
   END_RUNG wire#w1
   // the same network as SCL:
   IF #Rh_ET51 AND #ELEV_PosDw THEN
       #Rh_ET52 := TRUE;   // SR flip-flop
   END_IF;
   IF #Rh_ET53 OR NOT #PosicionConocida THEN #Rh_ET52 := FALSE; END_IF;
END_REGION

REGION Network 6: ET51
   RUNG wire#powerrail
      Contact( #Rh_ET00 )
      Contact( #PosicionConocida )
      Contact( #RH_DejarPaleta )
      I_Contact( #EnMovimiento_Tx )
      I_Contact( #MAQx_Desabilitada )
      S_SR(operand := #Rh_ET51, r1 := wire#w1)
   END_RUNG
   RUNG wire#powerrail
      Contact( #Rh_ET52 )
   END_RUNG wire#w1
   RUNG wire#powerrail
      I_Contact( #PosicionConocida )
   END_RUNG wire#w1
   // the same network as SCL:
   IF #Rh_ET00 AND #PosicionConocida AND #RH_DejarPaleta AND NOT #EnMovimiento_Tx AND NOT #MAQx_Desabilitada THEN
       #Rh_ET51 := TRUE;   // SR flip-flop
   END_IF;
   IF #Rh_ET52 OR NOT #PosicionConocida THEN #Rh_ET51 := FALSE; END_IF;
END_REGION

REGION Network 7: ET44 - CONTROL REMONTAR PALETA
   RUNG wire#powerrail
      Contact( #Rh_ET43 )
      Contact( #ELEV_PosDw )
      S_SR(operand := #Rh_ET44, r1 := wire#w1)
   END_RUNG
   RUNG wire#powerrail
      Contact( #Rh_ET00 )
   END_RUNG wire#w1
   RUNG wire#powerrail
      I_Contact( #PosicionConocida )
   END_RUNG wire#w1
   // the same network as SCL:
   IF #Rh_ET43 AND #ELEV_PosDw THEN
       #Rh_ET44 := TRUE;   // SR flip-flop
   END_IF;
   IF #Rh_ET00 OR NOT #PosicionConocida THEN #Rh_ET44 := FALSE; END_IF;
END_REGION

REGION Network 8: ET43
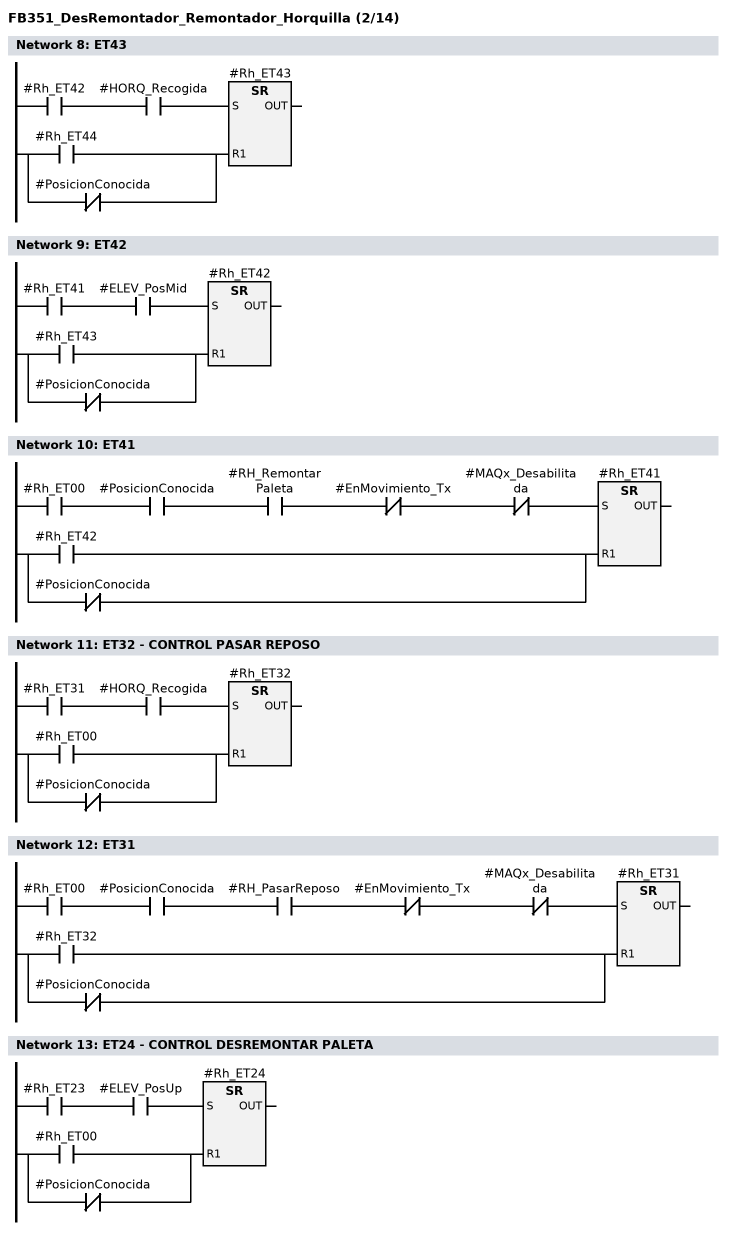
   RUNG wire#powerrail
      Contact( #Rh_ET42 )
      Contact( #HORQ_Recogida )
      S_SR(operand := #Rh_ET43, r1 := wire#w1)
   END_RUNG
   RUNG wire#powerrail
      Contact( #Rh_ET44 )
   END_RUNG wire#w1
   RUNG wire#powerrail
      I_Contact( #PosicionConocida )
   END_RUNG wire#w1
   // the same network as SCL:
   IF #Rh_ET42 AND #HORQ_Recogida THEN
       #Rh_ET43 := TRUE;   // SR flip-flop
   END_IF;
   IF #Rh_ET44 OR NOT #PosicionConocida THEN #Rh_ET43 := FALSE; END_IF;
END_REGION

REGION Network 9: ET42
   RUNG wire#powerrail
      Contact( #Rh_ET41 )
      Contact( #ELEV_PosMid )
      S_SR(operand := #Rh_ET42, r1 := wire#w1)
   END_RUNG
   RUNG wire#powerrail
      Contact( #Rh_ET43 )
   END_RUNG wire#w1
   RUNG wire#powerrail
      I_Contact( #PosicionConocida )
   END_RUNG wire#w1
   // the same network as SCL:
   IF #Rh_ET41 AND #ELEV_PosMid THEN
       #Rh_ET42 := TRUE;   // SR flip-flop
   END_IF;
   IF #Rh_ET43 OR NOT #PosicionConocida THEN #Rh_ET42 := FALSE; END_IF;
END_REGION

REGION Network 10: ET41
   RUNG wire#powerrail
      Contact( #Rh_ET00 )
      Contact( #PosicionConocida )
      Contact( #RH_RemontarPaleta )
      I_Contact( #EnMovimiento_Tx )
      I_Contact( #MAQx_Desabilitada )
      S_SR(operand := #Rh_ET41, r1 := wire#w1)
   END_RUNG
   RUNG wire#powerrail
      Contact( #Rh_ET42 )
   END_RUNG wire#w1
   RUNG wire#powerrail
      I_Contact( #PosicionConocida )
   END_RUNG wire#w1
   // the same network as SCL:
   IF #Rh_ET00 AND #PosicionConocida AND #RH_RemontarPaleta AND NOT #EnMovimiento_Tx AND NOT #MAQx_Desabilitada THEN
       #Rh_ET41 := TRUE;   // SR flip-flop
   END_IF;
   IF #Rh_ET42 OR NOT #PosicionConocida THEN #Rh_ET41 := FALSE; END_IF;
END_REGION

REGION Network 11: ET32 - CONTROL PASAR REPOSO
   RUNG wire#powerrail
      Contact( #Rh_ET31 )
      Contact( #HORQ_Recogida )
      S_SR(operand := #Rh_ET32, r1 := wire#w1)
   END_RUNG
   RUNG wire#powerrail
      Contact( #Rh_ET00 )
   END_RUNG wire#w1
   RUNG wire#powerrail
      I_Contact( #PosicionConocida )
   END_RUNG wire#w1
   // the same network as SCL:
   IF #Rh_ET31 AND #HORQ_Recogida THEN
       #Rh_ET32 := TRUE;   // SR flip-flop
   END_IF;
   IF #Rh_ET00 OR NOT #PosicionConocida THEN #Rh_ET32 := FALSE; END_IF;
END_REGION

REGION Network 12: ET31
   RUNG wire#powerrail
      Contact( #Rh_ET00 )
      Contact( #PosicionConocida )
      Contact( #RH_PasarReposo )
      I_Contact( #EnMovimiento_Tx )
      I_Contact( #MAQx_Desabilitada )
      S_SR(operand := #Rh_ET31, r1 := wire#w1)
   END_RUNG
   RUNG wire#powerrail
      Contact( #Rh_ET32 )
   END_RUNG wire#w1
   RUNG wire#powerrail
      I_Contact( #PosicionConocida )
   END_RUNG wire#w1
   // the same network as SCL:
   IF #Rh_ET00 AND #PosicionConocida AND #RH_PasarReposo AND NOT #EnMovimiento_Tx AND NOT #MAQx_Desabilitada THEN
       #Rh_ET31 := TRUE;   // SR flip-flop
   END_IF;
   IF #Rh_ET32 OR NOT #PosicionConocida THEN #Rh_ET31 := FALSE; END_IF;
END_REGION

REGION Network 13: ET24 - CONTROL DESREMONTAR PALETA
   RUNG wire#powerrail
      Contact( #Rh_ET23 )
      Contact( #ELEV_PosUp )
      S_SR(operand := #Rh_ET24, r1 := wire#w1)
   END_RUNG
   RUNG wire#powerrail
      Contact( #Rh_ET00 )
   END_RUNG wire#w1
   RUNG wire#powerrail
      I_Contact( #PosicionConocida )
   END_RUNG wire#w1
   // the same network as SCL:
   IF #Rh_ET23 AND #ELEV_PosUp THEN
       #Rh_ET24 := TRUE;   // SR flip-flop
   END_IF;
   IF #Rh_ET00 OR NOT #PosicionConocida THEN #Rh_ET24 := FALSE; END_IF;
END_REGION

REGION Network 14: ET23
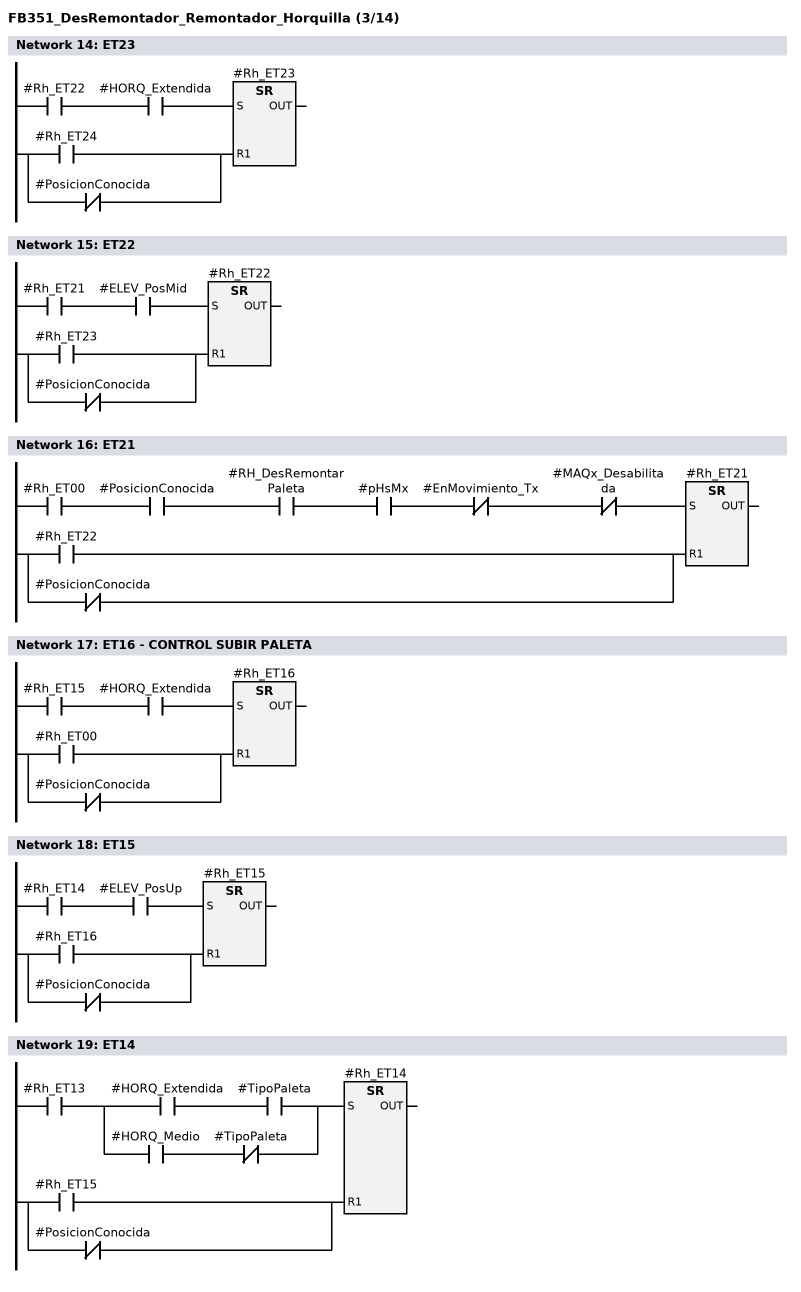
   RUNG wire#powerrail
      Contact( #Rh_ET22 )
      Contact( #HORQ_Extendida )
      S_SR(operand := #Rh_ET23, r1 := wire#w1)
   END_RUNG
   RUNG wire#powerrail
      Contact( #Rh_ET24 )
   END_RUNG wire#w1
   RUNG wire#powerrail
      I_Contact( #PosicionConocida )
   END_RUNG wire#w1
   // the same network as SCL:
   IF #Rh_ET22 AND #HORQ_Extendida THEN
       #Rh_ET23 := TRUE;   // SR flip-flop
   END_IF;
   IF #Rh_ET24 OR NOT #PosicionConocida THEN #Rh_ET23 := FALSE; END_IF;
END_REGION

REGION Network 15: ET22
   RUNG wire#powerrail
      Contact( #Rh_ET21 )
      Contact( #ELEV_PosMid )
      S_SR(operand := #Rh_ET22, r1 := wire#w1)
   END_RUNG
   RUNG wire#powerrail
      Contact( #Rh_ET23 )
   END_RUNG wire#w1
   RUNG wire#powerrail
      I_Contact( #PosicionConocida )
   END_RUNG wire#w1
   // the same network as SCL:
   IF #Rh_ET21 AND #ELEV_PosMid THEN
       #Rh_ET22 := TRUE;   // SR flip-flop
   END_IF;
   IF #Rh_ET23 OR NOT #PosicionConocida THEN #Rh_ET22 := FALSE; END_IF;
END_REGION

REGION Network 16: ET21
   RUNG wire#powerrail
      Contact( #Rh_ET00 )
      Contact( #PosicionConocida )
      Contact( #RH_DesRemontarPaleta )
      Contact( #pHsMx )
      I_Contact( #EnMovimiento_Tx )
      I_Contact( #MAQx_Desabilitada )
      S_SR(operand := #Rh_ET21, r1 := wire#w1)
   END_RUNG
   RUNG wire#powerrail
      Contact( #Rh_ET22 )
   END_RUNG wire#w1
   RUNG wire#powerrail
      I_Contact( #PosicionConocida )
   END_RUNG wire#w1
   // the same network as SCL:
   IF #Rh_ET00 AND #PosicionConocida AND #RH_DesRemontarPaleta AND #pHsMx AND NOT #EnMovimiento_Tx AND NOT #MAQx_Desabilitada THEN
       #Rh_ET21 := TRUE;   // SR flip-flop
   END_IF;
   IF #Rh_ET22 OR NOT #PosicionConocida THEN #Rh_ET21 := FALSE; END_IF;
END_REGION

REGION Network 17: ET16 - CONTROL SUBIR PALETA
   RUNG wire#powerrail
      Contact( #Rh_ET15 )
      Contact( #HORQ_Extendida )
      S_SR(operand := #Rh_ET16, r1 := wire#w1)
   END_RUNG
   RUNG wire#powerrail
      Contact( #Rh_ET00 )
   END_RUNG wire#w1
   RUNG wire#powerrail
      I_Contact( #PosicionConocida )
   END_RUNG wire#w1
   // the same network as SCL:
   IF #Rh_ET15 AND #HORQ_Extendida THEN
       #Rh_ET16 := TRUE;   // SR flip-flop
   END_IF;
   IF #Rh_ET00 OR NOT #PosicionConocida THEN #Rh_ET16 := FALSE; END_IF;
END_REGION

REGION Network 18: ET15
   RUNG wire#powerrail
      Contact( #Rh_ET14 )
      Contact( #ELEV_PosUp )
      S_SR(operand := #Rh_ET15, r1 := wire#w1)
   END_RUNG
   RUNG wire#powerrail
      Contact( #Rh_ET16 )
   END_RUNG wire#w1
   RUNG wire#powerrail
      I_Contact( #PosicionConocida )
   END_RUNG wire#w1
   // the same network as SCL:
   IF #Rh_ET14 AND #ELEV_PosUp THEN
       #Rh_ET15 := TRUE;   // SR flip-flop
   END_IF;
   IF #Rh_ET16 OR NOT #PosicionConocida THEN #Rh_ET15 := FALSE; END_IF;
END_REGION

REGION Network 19: ET14
   RUNG wire#powerrail
      Contact( #Rh_ET13 )
      wire#w1
      Contact( #HORQ_Extendida )
      Contact( #TipoPaleta )
      wire#w2
      S_SR(operand := #Rh_ET14, r1 := wire#w3)
   END_RUNG
   RUNG wire#w1
      Contact( #HORQ_Medio )
      I_Contact( #TipoPaleta )
   END_RUNG wire#w2
   RUNG wire#powerrail
      Contact( #Rh_ET15 )
   END_RUNG wire#w3
   RUNG wire#powerrail
      I_Contact( #PosicionConocida )
   END_RUNG wire#w3
   // the same network as SCL:
   IF #Rh_ET13 AND ((#HORQ_Extendida AND #TipoPaleta) OR (#HORQ_Medio AND NOT #TipoPaleta)) THEN
       #Rh_ET14 := TRUE;   // SR flip-flop
   END_IF;
   IF #Rh_ET15 OR NOT #PosicionConocida THEN #Rh_ET14 := FALSE; END_IF;
END_REGION

REGION Network 20: ET13
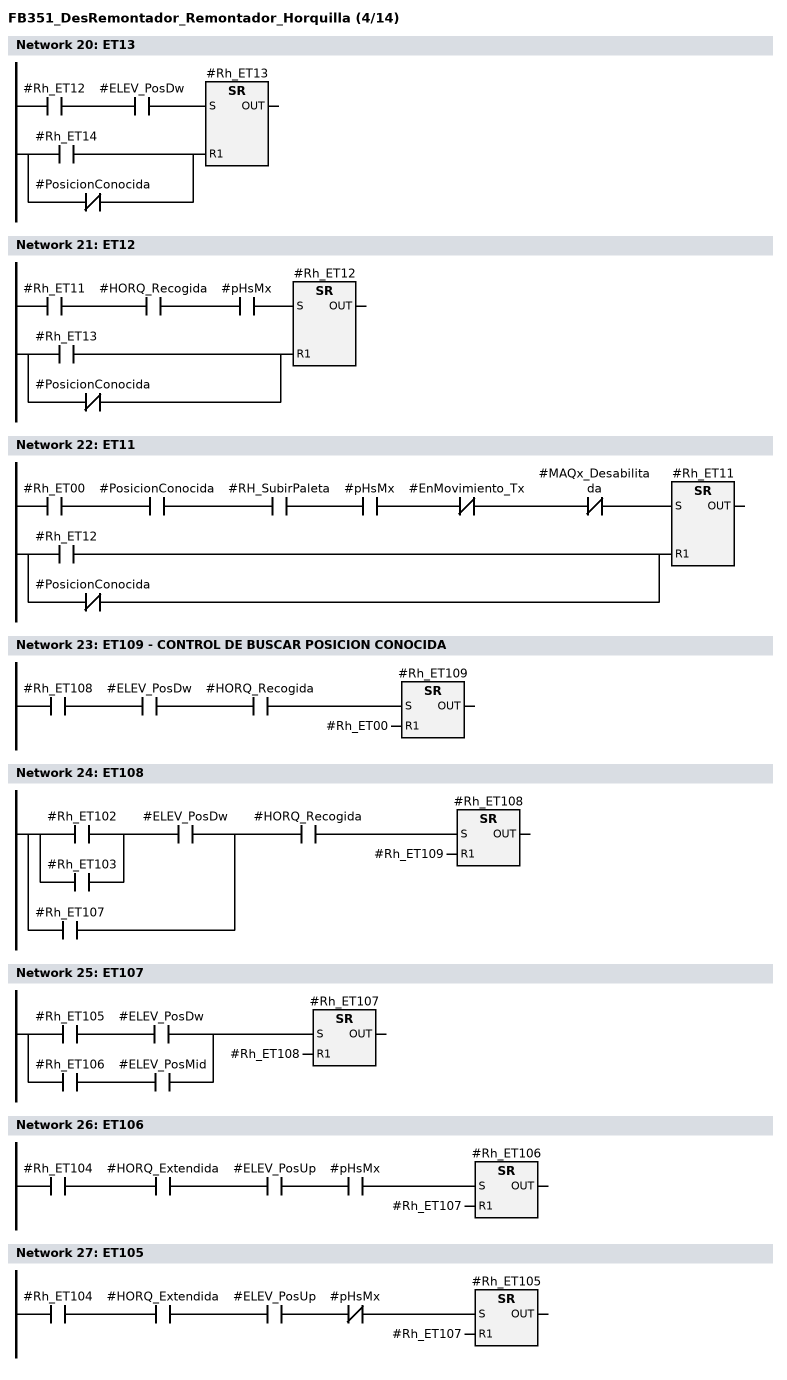
   RUNG wire#powerrail
      Contact( #Rh_ET12 )
      Contact( #ELEV_PosDw )
      S_SR(operand := #Rh_ET13, r1 := wire#w1)
   END_RUNG
   RUNG wire#powerrail
      Contact( #Rh_ET14 )
   END_RUNG wire#w1
   RUNG wire#powerrail
      I_Contact( #PosicionConocida )
   END_RUNG wire#w1
   // the same network as SCL:
   IF #Rh_ET12 AND #ELEV_PosDw THEN
       #Rh_ET13 := TRUE;   // SR flip-flop
   END_IF;
   IF #Rh_ET14 OR NOT #PosicionConocida THEN #Rh_ET13 := FALSE; END_IF;
END_REGION

REGION Network 21: ET12
   RUNG wire#powerrail
      Contact( #Rh_ET11 )
      Contact( #HORQ_Recogida )
      Contact( #pHsMx )
      S_SR(operand := #Rh_ET12, r1 := wire#w1)
   END_RUNG
   RUNG wire#powerrail
      Contact( #Rh_ET13 )
   END_RUNG wire#w1
   RUNG wire#powerrail
      I_Contact( #PosicionConocida )
   END_RUNG wire#w1
   // the same network as SCL:
   IF #Rh_ET11 AND #HORQ_Recogida AND #pHsMx THEN
       #Rh_ET12 := TRUE;   // SR flip-flop
   END_IF;
   IF #Rh_ET13 OR NOT #PosicionConocida THEN #Rh_ET12 := FALSE; END_IF;
END_REGION

REGION Network 22: ET11
   RUNG wire#powerrail
      Contact( #Rh_ET00 )
      Contact( #PosicionConocida )
      Contact( #RH_SubirPaleta )
      Contact( #pHsMx )
      I_Contact( #EnMovimiento_Tx )
      I_Contact( #MAQx_Desabilitada )
      S_SR(operand := #Rh_ET11, r1 := wire#w1)
   END_RUNG
   RUNG wire#powerrail
      Contact( #Rh_ET12 )
   END_RUNG wire#w1
   RUNG wire#powerrail
      I_Contact( #PosicionConocida )
   END_RUNG wire#w1
   // the same network as SCL:
   IF #Rh_ET00 AND #PosicionConocida AND #RH_SubirPaleta AND #pHsMx AND NOT #EnMovimiento_Tx AND NOT #MAQx_Desabilitada THEN
       #Rh_ET11 := TRUE;   // SR flip-flop
   END_IF;
   IF #Rh_ET12 OR NOT #PosicionConocida THEN #Rh_ET11 := FALSE; END_IF;
END_REGION

REGION Network 23: ET109 - CONTROL DE BUSCAR POSICION CONOCIDA
   RUNG wire#powerrail
      Contact( #Rh_ET108 )
      Contact( #ELEV_PosDw )
      Contact( #HORQ_Recogida )
      S_SR(operand := #Rh_ET109, r1 := #Rh_ET00)
   END_RUNG
   // the same network as SCL:
   IF #Rh_ET108 AND #ELEV_PosDw AND #HORQ_Recogida THEN
       #Rh_ET109 := TRUE;   // SR flip-flop
   END_IF;
   IF #Rh_ET00 THEN #Rh_ET109 := FALSE; END_IF;
END_REGION

REGION Network 24: ET108
   RUNG wire#powerrail
      Contact( #Rh_ET102 )
      wire#w1
      Contact( #ELEV_PosDw )
      wire#w2
      Contact( #HORQ_Recogida )
      S_SR(operand := #Rh_ET108, r1 := #Rh_ET109)
   END_RUNG
   RUNG wire#powerrail
      Contact( #Rh_ET103 )
   END_RUNG wire#w1
   RUNG wire#powerrail
      Contact( #Rh_ET107 )
   END_RUNG wire#w2
   // the same network as SCL:
   IF (((#Rh_ET102 OR #Rh_ET103) AND #ELEV_PosDw) OR #Rh_ET107) AND #HORQ_Recogida THEN
       #Rh_ET108 := TRUE;   // SR flip-flop
   END_IF;
   IF #Rh_ET109 THEN #Rh_ET108 := FALSE; END_IF;
END_REGION

REGION Network 25: ET107
   RUNG wire#powerrail
      Contact( #Rh_ET105 )
      Contact( #ELEV_PosDw )
      wire#w1
      S_SR(operand := #Rh_ET107, r1 := #Rh_ET108)
   END_RUNG
   RUNG wire#powerrail
      Contact( #Rh_ET106 )
      Contact( #ELEV_PosMid )
   END_RUNG wire#w1
   // the same network as SCL:
   IF (#Rh_ET105 AND #ELEV_PosDw) OR (#Rh_ET106 AND #ELEV_PosMid) THEN
       #Rh_ET107 := TRUE;   // SR flip-flop
   END_IF;
   IF #Rh_ET108 THEN #Rh_ET107 := FALSE; END_IF;
END_REGION

REGION Network 26: ET106
   RUNG wire#powerrail
      Contact( #Rh_ET104 )
      Contact( #HORQ_Extendida )
      Contact( #ELEV_PosUp )
      Contact( #pHsMx )
      S_SR(operand := #Rh_ET106, r1 := #Rh_ET107)
   END_RUNG
   // the same network as SCL:
   IF #Rh_ET104 AND #HORQ_Extendida AND #ELEV_PosUp AND #pHsMx THEN
       #Rh_ET106 := TRUE;   // SR flip-flop
   END_IF;
   IF #Rh_ET107 THEN #Rh_ET106 := FALSE; END_IF;
END_REGION

REGION Network 27: ET105
   RUNG wire#powerrail
      Contact( #Rh_ET104 )
      Contact( #HORQ_Extendida )
      Contact( #ELEV_PosUp )
      I_Contact( #pHsMx )
      S_SR(operand := #Rh_ET105, r1 := #Rh_ET107)
   END_RUNG
   // the same network as SCL:
   IF #Rh_ET104 AND #HORQ_Extendida AND #ELEV_PosUp AND NOT #pHsMx THEN
       #Rh_ET105 := TRUE;   // SR flip-flop
   END_IF;
   IF #Rh_ET107 THEN #Rh_ET105 := FALSE; END_IF;
END_REGION

REGION Network 28: ET104
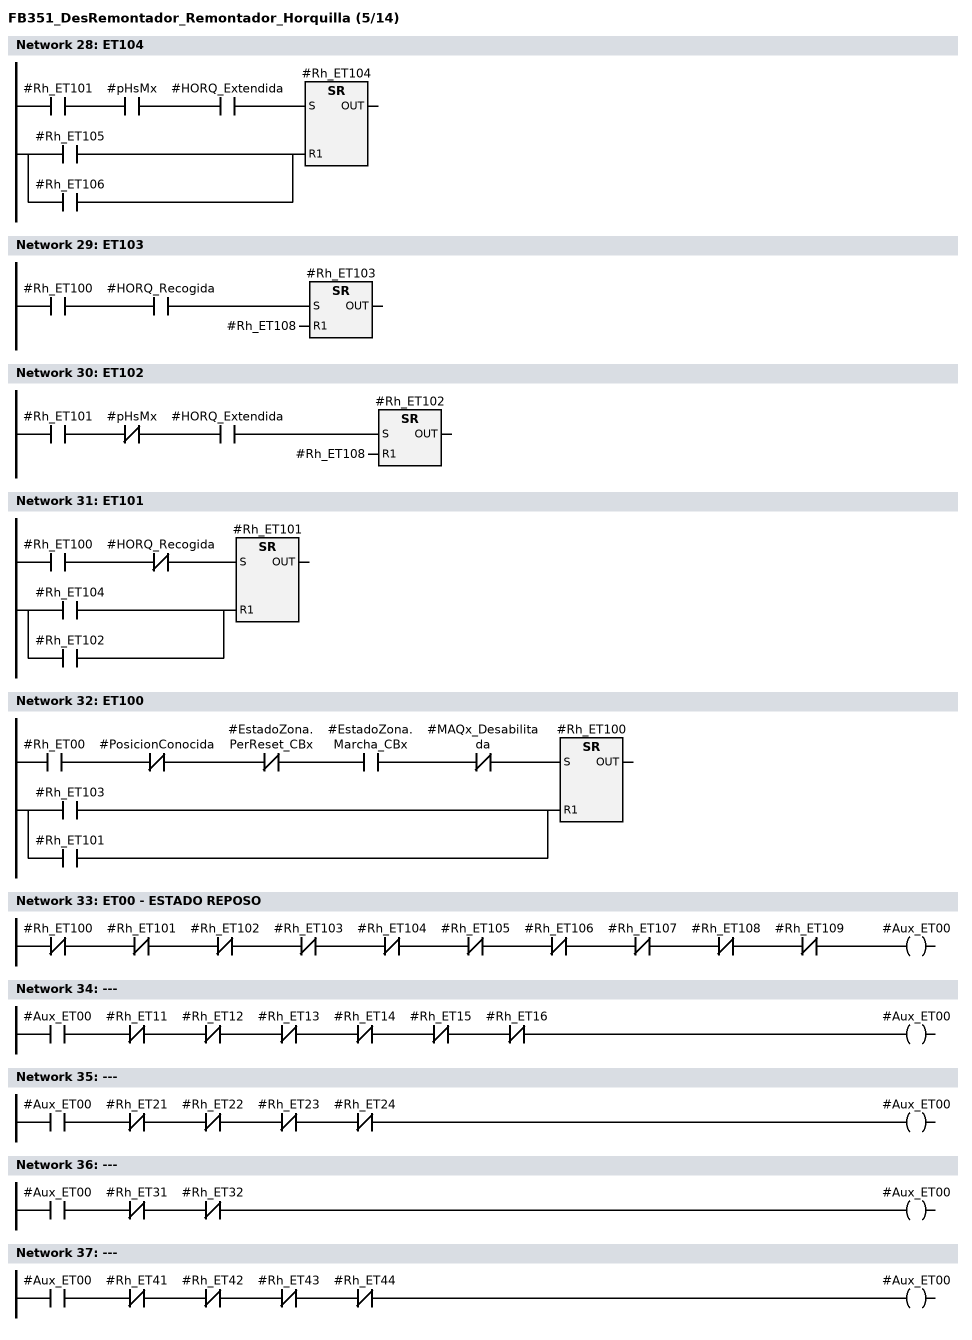
   RUNG wire#powerrail
      Contact( #Rh_ET101 )
      Contact( #pHsMx )
      Contact( #HORQ_Extendida )
      S_SR(operand := #Rh_ET104, r1 := wire#w1)
   END_RUNG
   RUNG wire#powerrail
      Contact( #Rh_ET105 )
   END_RUNG wire#w1
   RUNG wire#powerrail
      Contact( #Rh_ET106 )
   END_RUNG wire#w1
   // the same network as SCL:
   IF #Rh_ET101 AND #pHsMx AND #HORQ_Extendida THEN
       #Rh_ET104 := TRUE;   // SR flip-flop
   END_IF;
   IF #Rh_ET105 OR #Rh_ET106 THEN #Rh_ET104 := FALSE; END_IF;
END_REGION

REGION Network 29: ET103
   RUNG wire#powerrail
      Contact( #Rh_ET100 )
      Contact( #HORQ_Recogida )
      S_SR(operand := #Rh_ET103, r1 := #Rh_ET108)
   END_RUNG
   // the same network as SCL:
   IF #Rh_ET100 AND #HORQ_Recogida THEN
       #Rh_ET103 := TRUE;   // SR flip-flop
   END_IF;
   IF #Rh_ET108 THEN #Rh_ET103 := FALSE; END_IF;
END_REGION

REGION Network 30: ET102
   RUNG wire#powerrail
      Contact( #Rh_ET101 )
      I_Contact( #pHsMx )
      Contact( #HORQ_Extendida )
      S_SR(operand := #Rh_ET102, r1 := #Rh_ET108)
   END_RUNG
   // the same network as SCL:
   IF #Rh_ET101 AND NOT #pHsMx AND #HORQ_Extendida THEN
       #Rh_ET102 := TRUE;   // SR flip-flop
   END_IF;
   IF #Rh_ET108 THEN #Rh_ET102 := FALSE; END_IF;
END_REGION

REGION Network 31: ET101
   RUNG wire#powerrail
      Contact( #Rh_ET100 )
      I_Contact( #HORQ_Recogida )
      S_SR(operand := #Rh_ET101, r1 := wire#w1)
   END_RUNG
   RUNG wire#powerrail
      Contact( #Rh_ET104 )
   END_RUNG wire#w1
   RUNG wire#powerrail
      Contact( #Rh_ET102 )
   END_RUNG wire#w1
   // the same network as SCL:
   IF #Rh_ET100 AND NOT #HORQ_Recogida THEN
       #Rh_ET101 := TRUE;   // SR flip-flop
   END_IF;
   IF #Rh_ET104 OR #Rh_ET102 THEN #Rh_ET101 := FALSE; END_IF;
END_REGION

REGION Network 32: ET100
   RUNG wire#powerrail
      Contact( #Rh_ET00 )
      I_Contact( #PosicionConocida )
      I_Contact( #EstadoZona.PerReset_CBx )
      Contact( #EstadoZona.Marcha_CBx )
      I_Contact( #MAQx_Desabilitada )
      S_SR(operand := #Rh_ET100, r1 := wire#w1)
   END_RUNG
   RUNG wire#powerrail
      Contact( #Rh_ET103 )
   END_RUNG wire#w1
   RUNG wire#powerrail
      Contact( #Rh_ET101 )
   END_RUNG wire#w1
   // the same network as SCL:
   IF #Rh_ET00 AND NOT #PosicionConocida AND NOT #EstadoZona.PerReset_CBx AND #EstadoZona.Marcha_CBx AND NOT #MAQx_Desabilitada THEN
       #Rh_ET100 := TRUE;   // SR flip-flop
   END_IF;
   IF #Rh_ET103 OR #Rh_ET101 THEN #Rh_ET100 := FALSE; END_IF;
END_REGION

REGION Network 33: ET00 - ESTADO REPOSO
   RUNG wire#powerrail
      I_Contact( #Rh_ET100 )
      I_Contact( #Rh_ET101 )
      I_Contact( #Rh_ET102 )
      I_Contact( #Rh_ET103 )
      I_Contact( #Rh_ET104 )
      I_Contact( #Rh_ET105 )
      I_Contact( #Rh_ET106 )
      I_Contact( #Rh_ET107 )
      I_Contact( #Rh_ET108 )
      I_Contact( #Rh_ET109 )
      Coil( #Aux_ET00 )
   END_RUNG
   // the same network as SCL:
   #Aux_ET00 := NOT #Rh_ET100 AND NOT #Rh_ET101 AND NOT #Rh_ET102 AND NOT #Rh_ET103 AND NOT #Rh_ET104 AND NOT #Rh_ET105 AND NOT #Rh_ET106 AND NOT #Rh_ET107 AND NOT #Rh_ET108 AND NOT #Rh_ET109;
END_REGION

REGION Network 34: ---
   RUNG wire#powerrail
      Contact( #Aux_ET00 )
      I_Contact( #Rh_ET11 )
      I_Contact( #Rh_ET12 )
      I_Contact( #Rh_ET13 )
      I_Contact( #Rh_ET14 )
      I_Contact( #Rh_ET15 )
      I_Contact( #Rh_ET16 )
      Coil( #Aux_ET00 )
   END_RUNG
   // the same network as SCL:
   #Aux_ET00 := #Aux_ET00 AND NOT #Rh_ET11 AND NOT #Rh_ET12 AND NOT #Rh_ET13 AND NOT #Rh_ET14 AND NOT #Rh_ET15 AND NOT #Rh_ET16;
END_REGION

REGION Network 35: ---
   RUNG wire#powerrail
      Contact( #Aux_ET00 )
      I_Contact( #Rh_ET21 )
      I_Contact( #Rh_ET22 )
      I_Contact( #Rh_ET23 )
      I_Contact( #Rh_ET24 )
      Coil( #Aux_ET00 )
   END_RUNG
   // the same network as SCL:
   #Aux_ET00 := #Aux_ET00 AND NOT #Rh_ET21 AND NOT #Rh_ET22 AND NOT #Rh_ET23 AND NOT #Rh_ET24;
END_REGION

REGION Network 36: ---
   RUNG wire#powerrail
      Contact( #Aux_ET00 )
      I_Contact( #Rh_ET31 )
      I_Contact( #Rh_ET32 )
      Coil( #Aux_ET00 )
   END_RUNG
   // the same network as SCL:
   #Aux_ET00 := #Aux_ET00 AND NOT #Rh_ET31 AND NOT #Rh_ET32;
END_REGION

REGION Network 37: ---
   RUNG wire#powerrail
      Contact( #Aux_ET00 )
      I_Contact( #Rh_ET41 )
      I_Contact( #Rh_ET42 )
      I_Contact( #Rh_ET43 )
      I_Contact( #Rh_ET44 )
      Coil( #Aux_ET00 )
   END_RUNG
   // the same network as SCL:
   #Aux_ET00 := #Aux_ET00 AND NOT #Rh_ET41 AND NOT #Rh_ET42 AND NOT #Rh_ET43 AND NOT #Rh_ET44;
END_REGION

REGION Network 38: ---
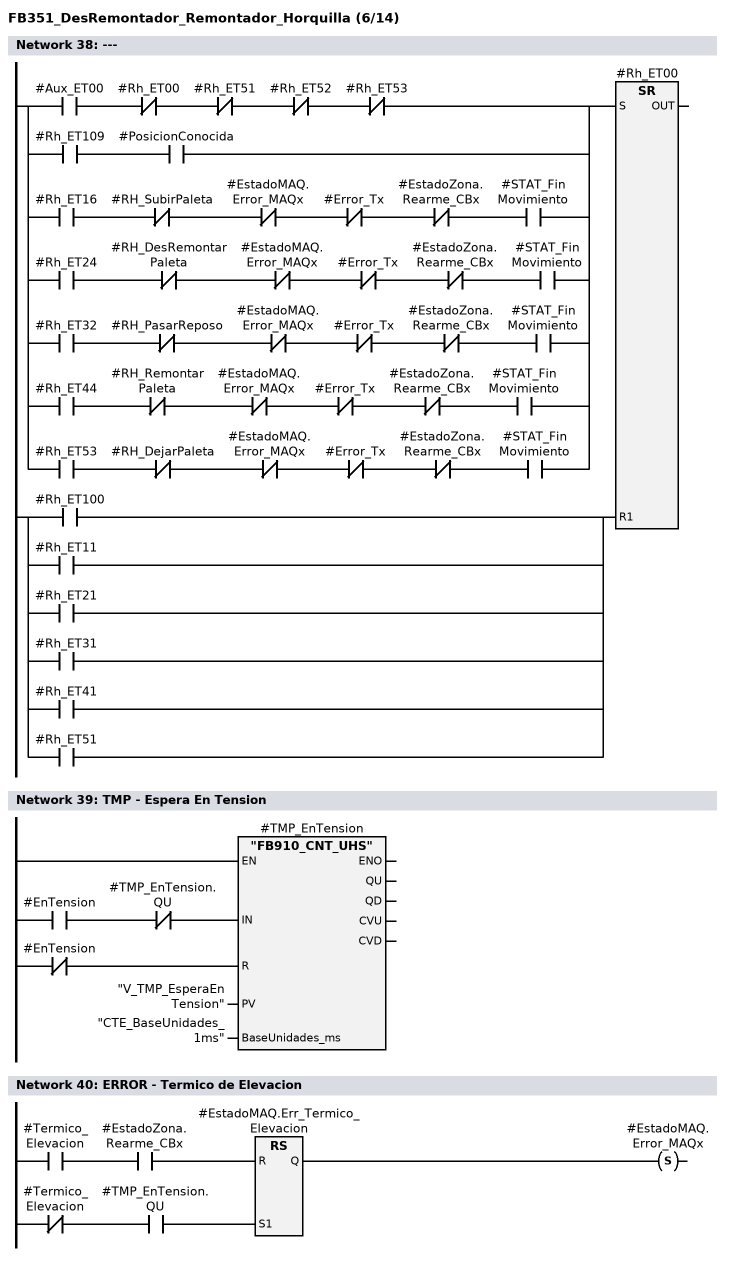
   RUNG wire#powerrail
      Contact( #Aux_ET00 )
      I_Contact( #Rh_ET00 )
      I_Contact( #Rh_ET51 )
      I_Contact( #Rh_ET52 )
      I_Contact( #Rh_ET53 )
      wire#w1
      S_SR(operand := #Rh_ET00, r1 := wire#w2)
   END_RUNG
   RUNG wire#powerrail
      Contact( #Rh_ET109 )
      Contact( #PosicionConocida )
   END_RUNG wire#w1
   RUNG wire#powerrail
      Contact( #Rh_ET16 )
      I_Contact( #RH_SubirPaleta )
      I_Contact( #EstadoMAQ.Error_MAQx )
      I_Contact( #Error_Tx )
      I_Contact( #EstadoZona.Rearme_CBx )
      Contact( #STAT_FinMovimiento )
   END_RUNG wire#w1
   RUNG wire#powerrail
      Contact( #Rh_ET24 )
      I_Contact( #RH_DesRemontarPaleta )
      I_Contact( #EstadoMAQ.Error_MAQx )
      I_Contact( #Error_Tx )
      I_Contact( #EstadoZona.Rearme_CBx )
      Contact( #STAT_FinMovimiento )
   END_RUNG wire#w1
   RUNG wire#powerrail
      Contact( #Rh_ET32 )
      I_Contact( #RH_PasarReposo )
      I_Contact( #EstadoMAQ.Error_MAQx )
      I_Contact( #Error_Tx )
      I_Contact( #EstadoZona.Rearme_CBx )
      Contact( #STAT_FinMovimiento )
   END_RUNG wire#w1
   RUNG wire#powerrail
      Contact( #Rh_ET44 )
      I_Contact( #RH_RemontarPaleta )
      I_Contact( #EstadoMAQ.Error_MAQx )
      I_Contact( #Error_Tx )
      I_Contact( #EstadoZona.Rearme_CBx )
      Contact( #STAT_FinMovimiento )
   END_RUNG wire#w1
   RUNG wire#powerrail
      Contact( #Rh_ET53 )
      I_Contact( #RH_DejarPaleta )
      I_Contact( #EstadoMAQ.Error_MAQx )
      I_Contact( #Error_Tx )
      I_Contact( #EstadoZona.Rearme_CBx )
      Contact( #STAT_FinMovimiento )
   END_RUNG wire#w1
   RUNG wire#powerrail
      Contact( #Rh_ET100 )
   END_RUNG wire#w2
   RUNG wire#powerrail
      Contact( #Rh_ET11 )
   END_RUNG wire#w2
   RUNG wire#powerrail
      Contact( #Rh_ET21 )
   END_RUNG wire#w2
   RUNG wire#powerrail
      Contact( #Rh_ET31 )
   END_RUNG wire#w2
   RUNG wire#powerrail
      Contact( #Rh_ET41 )
   END_RUNG wire#w2
   RUNG wire#powerrail
      Contact( #Rh_ET51 )
   END_RUNG wire#w2
   // the same network as SCL:
   IF (#Aux_ET00 AND NOT #Rh_ET00 AND NOT #Rh_ET51 AND NOT #Rh_ET52 AND NOT #Rh_ET53) OR (#Rh_ET109 AND #PosicionConocida) OR (#Rh_ET16 AND NOT #RH_SubirPaleta AND NOT #EstadoMAQ.Error_MAQx AND NOT #Error_Tx AND NOT #EstadoZona.Rearme_CBx AND #STAT_FinMovimiento) OR (#Rh_ET24 AND NOT #RH_DesRemontarPaleta AND NOT #EstadoMAQ.Error_MAQx AND NOT #Error_Tx AND NOT #EstadoZona.Rearme_CBx AND #STAT_FinMovimiento) OR (#Rh_ET32 AND NOT #RH_PasarReposo AND NOT #EstadoMAQ.Error_MAQx AND NOT #Error_Tx AND NOT #EstadoZona.Rearme_CBx AND #STAT_FinMovimiento) OR (#Rh_ET44 AND NOT #RH_RemontarPaleta AND NOT #EstadoMAQ.Error_MAQx AND NOT #Error_Tx AND NOT #EstadoZona.Rearme_CBx AND #STAT_FinMovimiento) OR (#Rh_ET53 AND NOT #RH_DejarPaleta AND NOT #EstadoMAQ.Error_MAQx AND NOT #Error_Tx AND NOT #EstadoZona.Rearme_CBx AND #STAT_FinMovimiento) THEN
       #Rh_ET00 := TRUE;   // SR flip-flop
   END_IF;
   IF #Rh_ET100 OR #Rh_ET11 OR #Rh_ET21 OR #Rh_ET31 OR #Rh_ET41 OR #Rh_ET51 THEN #Rh_ET00 := FALSE; END_IF;
END_REGION

REGION Network 39: TMP - Espera En Tension
   RUNG wire#powerrail
      #TMP_EnTension(IN := wire#w1, R := wire#w2, PV := "V_TMP_EsperaEnTension", BaseUnidades_ms := "CTE_BaseUnidades_1ms", QU =>, QD =>, CVU =>, CVD =>)
   END_RUNG
   RUNG wire#powerrail
      Contact( #EnTension )
      I_Contact( #TMP_EnTension.QU )
   END_RUNG wire#w1
   RUNG wire#powerrail
      I_Contact( #EnTension )
   END_RUNG wire#w2
   // the same network as SCL:
   #TMP_EnTension(IN := #EnTension AND NOT #TMP_EnTension.QU,   // "FB910_CNT_UHS"
                  R := NOT #EnTension,
                  PV := "V_TMP_EsperaEnTension",
                  BaseUnidades_ms := "CTE_BaseUnidades_1ms");
END_REGION

REGION Network 40: ERROR - Termico de Elevacion
   RUNG wire#powerrail
      Contact( #Termico_Elevacion )
      Contact( #EstadoZona.Rearme_CBx )
      S_RS(operand := #EstadoMAQ.Err_Termico_Elevacion, s1 := wire#w1)
      S_Coil( #EstadoMAQ.Error_MAQx )
   END_RUNG
   RUNG wire#powerrail
      I_Contact( #Termico_Elevacion )
      Contact( #TMP_EnTension.QU )
   END_RUNG wire#w1
   // the same network as SCL:
   IF #Termico_Elevacion AND #EstadoZona.Rearme_CBx THEN
       #EstadoMAQ.Err_Termico_Elevacion := FALSE;   // RS flip-flop
   END_IF;
   IF NOT #Termico_Elevacion AND #TMP_EnTension.QU THEN #EstadoMAQ.Err_Termico_Elevacion := TRUE; END_IF;
   IF #EstadoMAQ.Err_Termico_Elevacion THEN #EstadoMAQ.Error_MAQx := TRUE; END_IF;
END_REGION

REGION Network 41: ERROR - Termico de Horquilla
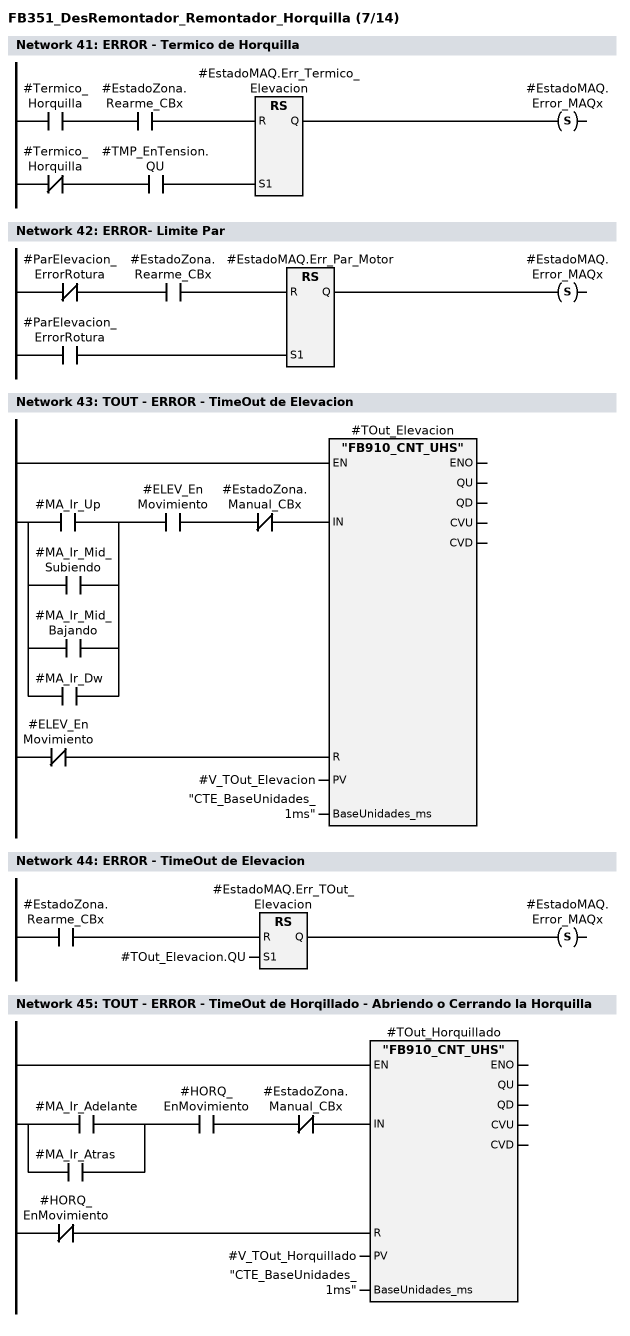
   RUNG wire#powerrail
      Contact( #Termico_Horquilla )
      Contact( #EstadoZona.Rearme_CBx )
      S_RS(operand := #EstadoMAQ.Err_Termico_Elevacion, s1 := wire#w1)
      S_Coil( #EstadoMAQ.Error_MAQx )
   END_RUNG
   RUNG wire#powerrail
      I_Contact( #Termico_Horquilla )
      Contact( #TMP_EnTension.QU )
   END_RUNG wire#w1
   // the same network as SCL:
   IF #Termico_Horquilla AND #EstadoZona.Rearme_CBx THEN
       #EstadoMAQ.Err_Termico_Elevacion := FALSE;   // RS flip-flop
   END_IF;
   IF NOT #Termico_Horquilla AND #TMP_EnTension.QU THEN #EstadoMAQ.Err_Termico_Elevacion := TRUE; END_IF;
   IF #EstadoMAQ.Err_Termico_Elevacion THEN #EstadoMAQ.Error_MAQx := TRUE; END_IF;
END_REGION

REGION Network 42: ERROR- Limite Par
   RUNG wire#powerrail
      I_Contact( #ParElevacion_ErrorRotura )
      Contact( #EstadoZona.Rearme_CBx )
      S_RS(operand := #EstadoMAQ.Err_Par_Motor, s1 := wire#w1)
      S_Coil( #EstadoMAQ.Error_MAQx )
   END_RUNG
   RUNG wire#powerrail
      Contact( #ParElevacion_ErrorRotura )
   END_RUNG wire#w1
   // the same network as SCL:
   IF NOT #ParElevacion_ErrorRotura AND #EstadoZona.Rearme_CBx THEN
       #EstadoMAQ.Err_Par_Motor := FALSE;   // RS flip-flop
   END_IF;
   IF #ParElevacion_ErrorRotura THEN #EstadoMAQ.Err_Par_Motor := TRUE; END_IF;
   IF #EstadoMAQ.Err_Par_Motor THEN #EstadoMAQ.Error_MAQx := TRUE; END_IF;
END_REGION

REGION Network 43: TOUT - ERROR - TimeOut de Elevacion
   RUNG wire#powerrail
      #TOut_Elevacion(IN := wire#w2, R := wire#w3, PV := #V_TOut_Elevacion, BaseUnidades_ms := "CTE_BaseUnidades_1ms", QU =>, QD =>, CVU =>, CVD =>)
   END_RUNG
   RUNG wire#powerrail
      Contact( #MA_Ir_Up )
      wire#w1
      Contact( #ELEV_EnMovimiento )
      I_Contact( #EstadoZona.Manual_CBx )
   END_RUNG wire#w2
   RUNG wire#powerrail
      Contact( #MA_Ir_Mid_Subiendo )
   END_RUNG wire#w1
   RUNG wire#powerrail
      Contact( #MA_Ir_Mid_Bajando )
   END_RUNG wire#w1
   RUNG wire#powerrail
      Contact( #MA_Ir_Dw )
   END_RUNG wire#w1
   RUNG wire#powerrail
      I_Contact( #ELEV_EnMovimiento )
   END_RUNG wire#w3
   // the same network as SCL:
   #TOut_Elevacion(IN := (#MA_Ir_Up OR #MA_Ir_Mid_Subiendo OR #MA_Ir_Mid_Bajando OR #MA_Ir_Dw) AND #ELEV_EnMovimiento AND NOT #EstadoZona.Manual_CBx,   // "FB910_CNT_UHS"
                   R := NOT #ELEV_EnMovimiento,
                   PV := #V_TOut_Elevacion,
                   BaseUnidades_ms := "CTE_BaseUnidades_1ms");
END_REGION

REGION Network 44: ERROR - TimeOut de Elevacion
   RUNG wire#powerrail
      Contact( #EstadoZona.Rearme_CBx )
      S_RS(operand := #EstadoMAQ.Err_TOut_Elevacion, s1 := #TOut_Elevacion.QU)
      S_Coil( #EstadoMAQ.Error_MAQx )
   END_RUNG
   // the same network as SCL:
   IF #EstadoZona.Rearme_CBx THEN
       #EstadoMAQ.Err_TOut_Elevacion := FALSE;   // RS flip-flop
   END_IF;
   IF #TOut_Elevacion.QU THEN #EstadoMAQ.Err_TOut_Elevacion := TRUE; END_IF;
   IF #EstadoMAQ.Err_TOut_Elevacion THEN #EstadoMAQ.Error_MAQx := TRUE; END_IF;
END_REGION

REGION Network 45: TOUT - ERROR - TimeOut de Horqillado - Abriendo o Cerrando la Horquilla
   RUNG wire#powerrail
      #TOut_Horquillado(IN := wire#w2, R := wire#w3, PV := #V_TOut_Horquillado, BaseUnidades_ms := "CTE_BaseUnidades_1ms", QU =>, QD =>, CVU =>, CVD =>)
   END_RUNG
   RUNG wire#powerrail
      Contact( #MA_Ir_Adelante )
      wire#w1
      Contact( #HORQ_EnMovimiento )
      I_Contact( #EstadoZona.Manual_CBx )
   END_RUNG wire#w2
   RUNG wire#powerrail
      Contact( #MA_Ir_Atras )
   END_RUNG wire#w1
   RUNG wire#powerrail
      I_Contact( #HORQ_EnMovimiento )
   END_RUNG wire#w3
   // the same network as SCL:
   #TOut_Horquillado(IN := (#MA_Ir_Adelante OR #MA_Ir_Atras) AND #HORQ_EnMovimiento AND NOT #EstadoZona.Manual_CBx,   // "FB910_CNT_UHS"
                     R := NOT #HORQ_EnMovimiento,
                     PV := #V_TOut_Horquillado,
                     BaseUnidades_ms := "CTE_BaseUnidades_1ms");
END_REGION

REGION Network 46: ERROR - TimeOut de Horqillado - Abriendo la Horquilla
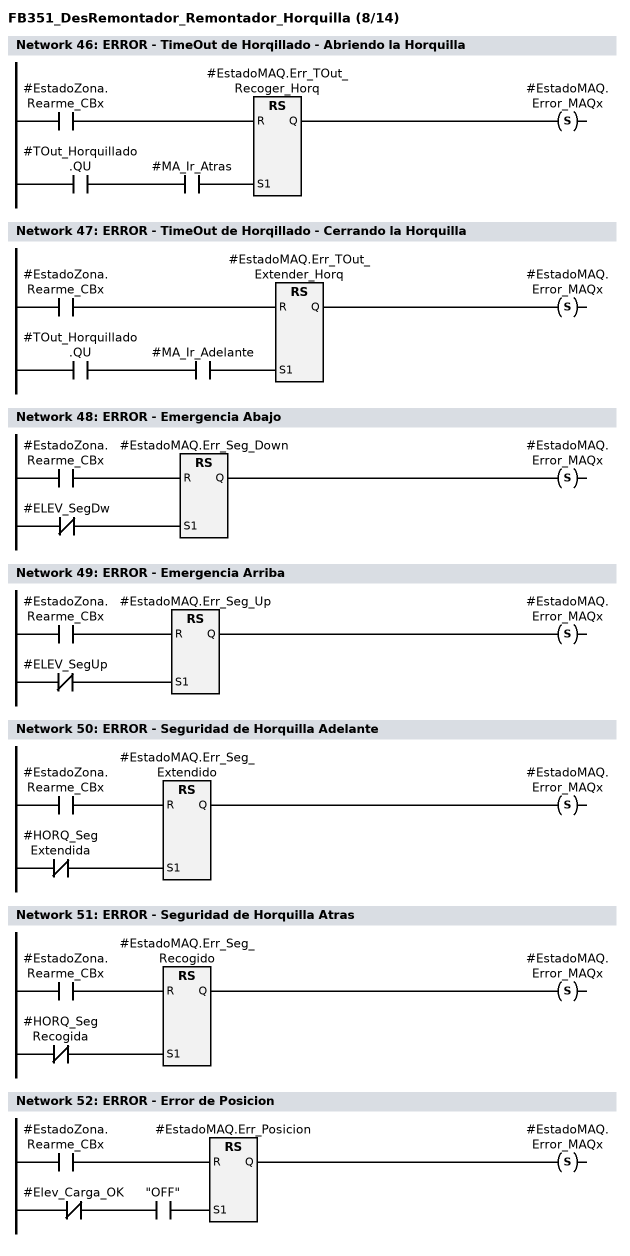
   RUNG wire#powerrail
      Contact( #EstadoZona.Rearme_CBx )
      S_RS(operand := #EstadoMAQ.Err_TOut_Recoger_Horq, s1 := wire#w1)
      S_Coil( #EstadoMAQ.Error_MAQx )
   END_RUNG
   RUNG wire#powerrail
      Contact( #TOut_Horquillado.QU )
      Contact( #MA_Ir_Atras )
   END_RUNG wire#w1
   // the same network as SCL:
   IF #EstadoZona.Rearme_CBx THEN
       #EstadoMAQ.Err_TOut_Recoger_Horq := FALSE;   // RS flip-flop
   END_IF;
   IF #TOut_Horquillado.QU AND #MA_Ir_Atras THEN #EstadoMAQ.Err_TOut_Recoger_Horq := TRUE; END_IF;
   IF #EstadoMAQ.Err_TOut_Recoger_Horq THEN #EstadoMAQ.Error_MAQx := TRUE; END_IF;
END_REGION

REGION Network 47: ERROR - TimeOut de Horqillado - Cerrando la Horquilla
   RUNG wire#powerrail
      Contact( #EstadoZona.Rearme_CBx )
      S_RS(operand := #EstadoMAQ.Err_TOut_Extender_Horq, s1 := wire#w1)
      S_Coil( #EstadoMAQ.Error_MAQx )
   END_RUNG
   RUNG wire#powerrail
      Contact( #TOut_Horquillado.QU )
      Contact( #MA_Ir_Adelante )
   END_RUNG wire#w1
   // the same network as SCL:
   IF #EstadoZona.Rearme_CBx THEN
       #EstadoMAQ.Err_TOut_Extender_Horq := FALSE;   // RS flip-flop
   END_IF;
   IF #TOut_Horquillado.QU AND #MA_Ir_Adelante THEN #EstadoMAQ.Err_TOut_Extender_Horq := TRUE; END_IF;
   IF #EstadoMAQ.Err_TOut_Extender_Horq THEN #EstadoMAQ.Error_MAQx := TRUE; END_IF;
END_REGION

REGION Network 48: ERROR - Emergencia Abajo
   RUNG wire#powerrail
      Contact( #EstadoZona.Rearme_CBx )
      S_RS(operand := #EstadoMAQ.Err_Seg_Down, s1 := wire#w1)
      S_Coil( #EstadoMAQ.Error_MAQx )
   END_RUNG
   RUNG wire#powerrail
      I_Contact( #ELEV_SegDw )
   END_RUNG wire#w1
   // the same network as SCL:
   IF #EstadoZona.Rearme_CBx THEN
       #EstadoMAQ.Err_Seg_Down := FALSE;   // RS flip-flop
   END_IF;
   IF NOT #ELEV_SegDw THEN #EstadoMAQ.Err_Seg_Down := TRUE; END_IF;
   IF #EstadoMAQ.Err_Seg_Down THEN #EstadoMAQ.Error_MAQx := TRUE; END_IF;
END_REGION

REGION Network 49: ERROR - Emergencia Arriba
   RUNG wire#powerrail
      Contact( #EstadoZona.Rearme_CBx )
      S_RS(operand := #EstadoMAQ.Err_Seg_Up, s1 := wire#w1)
      S_Coil( #EstadoMAQ.Error_MAQx )
   END_RUNG
   RUNG wire#powerrail
      I_Contact( #ELEV_SegUp )
   END_RUNG wire#w1
   // the same network as SCL:
   IF #EstadoZona.Rearme_CBx THEN
       #EstadoMAQ.Err_Seg_Up := FALSE;   // RS flip-flop
   END_IF;
   IF NOT #ELEV_SegUp THEN #EstadoMAQ.Err_Seg_Up := TRUE; END_IF;
   IF #EstadoMAQ.Err_Seg_Up THEN #EstadoMAQ.Error_MAQx := TRUE; END_IF;
END_REGION

REGION Network 50: ERROR - Seguridad de Horquilla Adelante
   RUNG wire#powerrail
      Contact( #EstadoZona.Rearme_CBx )
      S_RS(operand := #EstadoMAQ.Err_Seg_Extendido, s1 := wire#w1)
      S_Coil( #EstadoMAQ.Error_MAQx )
   END_RUNG
   RUNG wire#powerrail
      I_Contact( #HORQ_SegExtendida )
   END_RUNG wire#w1
   // the same network as SCL:
   IF #EstadoZona.Rearme_CBx THEN
       #EstadoMAQ.Err_Seg_Extendido := FALSE;   // RS flip-flop
   END_IF;
   IF NOT #HORQ_SegExtendida THEN #EstadoMAQ.Err_Seg_Extendido := TRUE; END_IF;
   IF #EstadoMAQ.Err_Seg_Extendido THEN #EstadoMAQ.Error_MAQx := TRUE; END_IF;
END_REGION

REGION Network 51: ERROR - Seguridad de Horquilla Atras
   RUNG wire#powerrail
      Contact( #EstadoZona.Rearme_CBx )
      S_RS(operand := #EstadoMAQ.Err_Seg_Recogido, s1 := wire#w1)
      S_Coil( #EstadoMAQ.Error_MAQx )
   END_RUNG
   RUNG wire#powerrail
      I_Contact( #HORQ_SegRecogida )
   END_RUNG wire#w1
   // the same network as SCL:
   IF #EstadoZona.Rearme_CBx THEN
       #EstadoMAQ.Err_Seg_Recogido := FALSE;   // RS flip-flop
   END_IF;
   IF NOT #HORQ_SegRecogida THEN #EstadoMAQ.Err_Seg_Recogido := TRUE; END_IF;
   IF #EstadoMAQ.Err_Seg_Recogido THEN #EstadoMAQ.Error_MAQx := TRUE; END_IF;
END_REGION

REGION Network 52: ERROR - Error de Posicion
   RUNG wire#powerrail
      Contact( #EstadoZona.Rearme_CBx )
      S_RS(operand := #EstadoMAQ.Err_Posicion, s1 := wire#w1)
      S_Coil( #EstadoMAQ.Error_MAQx )
   END_RUNG
   RUNG wire#powerrail
      I_Contact( #Elev_Carga_OK )
      Contact( "OFF" )
   END_RUNG wire#w1
   // the same network as SCL:
   IF #EstadoZona.Rearme_CBx THEN
       #EstadoMAQ.Err_Posicion := FALSE;   // RS flip-flop
   END_IF;
   IF NOT #Elev_Carga_OK AND "OFF" THEN #EstadoMAQ.Err_Posicion := TRUE; END_IF;
   IF #EstadoMAQ.Err_Posicion THEN #EstadoMAQ.Error_MAQx := TRUE; END_IF;
END_REGION

REGION Network 53: Error Carga
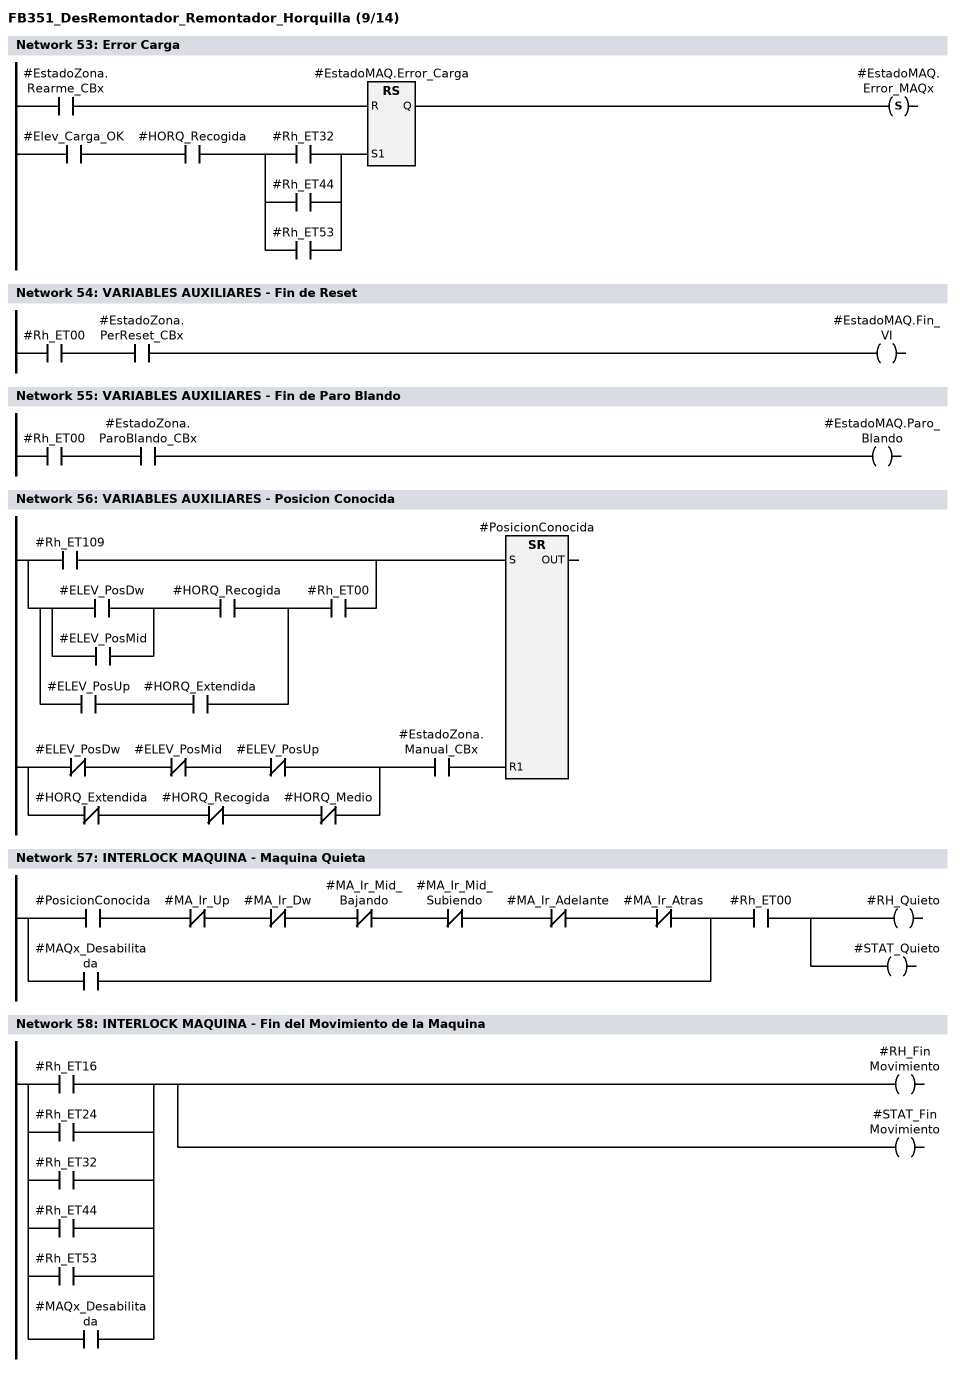
   RUNG wire#powerrail
      Contact( #EstadoZona.Rearme_CBx )
      S_RS(operand := #EstadoMAQ.Error_Carga, s1 := wire#w2)
      S_Coil( #EstadoMAQ.Error_MAQx )
   END_RUNG
   RUNG wire#powerrail
      Contact( #Elev_Carga_OK )
      Contact( #HORQ_Recogida )
      wire#w1
      Contact( #Rh_ET32 )
   END_RUNG wire#w2
   RUNG wire#w1
      Contact( #Rh_ET44 )
   END_RUNG wire#w2
   RUNG wire#w1
      Contact( #Rh_ET53 )
   END_RUNG wire#w2
   // the same network as SCL:
   IF #EstadoZona.Rearme_CBx THEN
       #EstadoMAQ.Error_Carga := FALSE;   // RS flip-flop
   END_IF;
   IF #Elev_Carga_OK AND #HORQ_Recogida AND (#Rh_ET32 OR #Rh_ET44 OR #Rh_ET53) THEN
       #EstadoMAQ.Error_Carga := TRUE;
   END_IF;
   IF #EstadoMAQ.Error_Carga THEN #EstadoMAQ.Error_MAQx := TRUE; END_IF;
END_REGION

REGION Network 54: VARIABLES AUXILIARES - Fin de Reset
   RUNG wire#powerrail
      Contact( #Rh_ET00 )
      Contact( #EstadoZona.PerReset_CBx )
      Coil( #EstadoMAQ.Fin_VI )
   END_RUNG
   // the same network as SCL:
   #EstadoMAQ.Fin_VI := #Rh_ET00 AND #EstadoZona.PerReset_CBx;
END_REGION

REGION Network 55: VARIABLES AUXILIARES - Fin de Paro Blando
   RUNG wire#powerrail
      Contact( #Rh_ET00 )
      Contact( #EstadoZona.ParoBlando_CBx )
      Coil( #EstadoMAQ.Paro_Blando )
   END_RUNG
   // the same network as SCL:
   #EstadoMAQ.Paro_Blando := #Rh_ET00 AND #EstadoZona.ParoBlando_CBx;
END_REGION

REGION Network 56: VARIABLES AUXILIARES - Posicion Conocida
   RUNG wire#powerrail
      Contact( #Rh_ET109 )
      wire#w1
      S_SR(operand := #PosicionConocida, r1 := wire#w5)
   END_RUNG
   RUNG wire#powerrail
      Contact( #ELEV_PosDw )
      wire#w2
      Contact( #HORQ_Recogida )
      wire#w3
      Contact( #Rh_ET00 )
   END_RUNG wire#w1
   RUNG wire#powerrail
      Contact( #ELEV_PosMid )
   END_RUNG wire#w2
   RUNG wire#powerrail
      Contact( #ELEV_PosUp )
      Contact( #HORQ_Extendida )
   END_RUNG wire#w3
   RUNG wire#powerrail
      I_Contact( #ELEV_PosDw )
      I_Contact( #ELEV_PosMid )
      I_Contact( #ELEV_PosUp )
      wire#w4
      Contact( #EstadoZona.Manual_CBx )
   END_RUNG wire#w5
   RUNG wire#powerrail
      I_Contact( #HORQ_Extendida )
      I_Contact( #HORQ_Recogida )
      I_Contact( #HORQ_Medio )
   END_RUNG wire#w4
   // the same network as SCL:
   IF #Rh_ET109 OR ((((#ELEV_PosDw OR #ELEV_PosMid) AND #HORQ_Recogida) OR (#ELEV_PosUp AND #HORQ_Extendida)) AND #Rh_ET00) THEN
       #PosicionConocida := TRUE;   // SR flip-flop
   END_IF;
   IF ((NOT #ELEV_PosDw AND NOT #ELEV_PosMid AND NOT #ELEV_PosUp) OR (NOT #HORQ_Extendida AND NOT #HORQ_Recogida AND NOT #HORQ_Medio)) AND #EstadoZona.Manual_CBx THEN
       #PosicionConocida := FALSE;
   END_IF;
END_REGION

REGION Network 57: INTERLOCK MAQUINA - Maquina Quieta
   RUNG wire#powerrail
      Contact( #PosicionConocida )
      I_Contact( #MA_Ir_Up )
      I_Contact( #MA_Ir_Dw )
      I_Contact( #MA_Ir_Mid_Bajando )
      I_Contact( #MA_Ir_Mid_Subiendo )
      I_Contact( #MA_Ir_Adelante )
      I_Contact( #MA_Ir_Atras )
      wire#w1
      Contact( #Rh_ET00 )
      wire#w2
      Coil( #RH_Quieto )
   END_RUNG
   RUNG wire#powerrail
      Contact( #MAQx_Desabilitada )
   END_RUNG wire#w1
   RUNG wire#w2
      Coil( #STAT_Quieto )
   END_RUNG
   // the same network as SCL:
   #RH_Quieto := ((#PosicionConocida AND NOT #MA_Ir_Up AND NOT #MA_Ir_Dw AND NOT #MA_Ir_Mid_Bajando AND NOT #MA_Ir_Mid_Subiendo AND NOT #MA_Ir_Adelante AND NOT #MA_Ir_Atras) OR #MAQx_Desabilitada) AND #Rh_ET00;
   #STAT_Quieto := #RH_Quieto;
END_REGION

REGION Network 58: INTERLOCK MAQUINA - Fin del Movimiento de la Maquina
   RUNG wire#powerrail
      Contact( #Rh_ET16 )
      wire#w1
      Coil( #RH_FinMovimiento )
   END_RUNG
   RUNG wire#powerrail
      Contact( #Rh_ET24 )
   END_RUNG wire#w1
   RUNG wire#powerrail
      Contact( #Rh_ET32 )
   END_RUNG wire#w1
   RUNG wire#powerrail
      Contact( #Rh_ET44 )
   END_RUNG wire#w1
   RUNG wire#powerrail
      Contact( #Rh_ET53 )
   END_RUNG wire#w1
   RUNG wire#powerrail
      Contact( #MAQx_Desabilitada )
   END_RUNG wire#w1
   RUNG wire#w1
      Coil( #STAT_FinMovimiento )
   END_RUNG
   // the same network as SCL:
   #RH_FinMovimiento := #Rh_ET16 OR #Rh_ET24 OR #Rh_ET32 OR #Rh_ET44 OR #Rh_ET53 OR #MAQx_Desabilitada;
   #STAT_FinMovimiento := #RH_FinMovimiento;
END_REGION

REGION Network 59: VARIABLES AUXILIARES - Cambiar de Direccion Buscando la Posicion Media
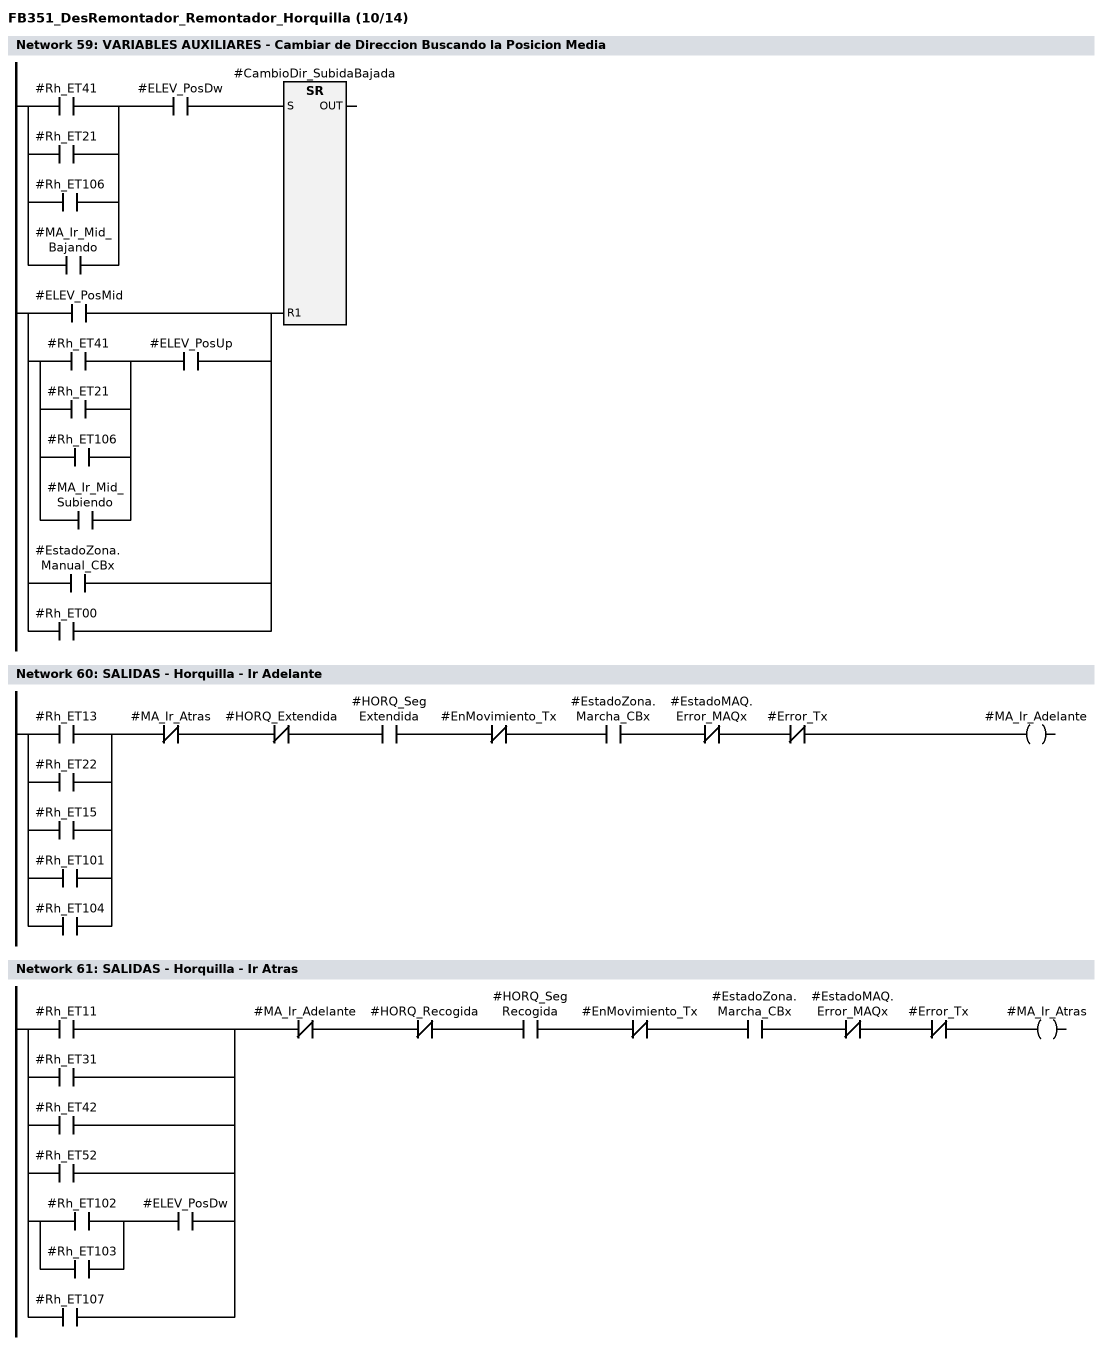
   RUNG wire#powerrail
      Contact( #Rh_ET41 )
      wire#w1
      Contact( #ELEV_PosDw )
      S_SR(operand := #CambioDir_SubidaBajada, r1 := wire#w3)
   END_RUNG
   RUNG wire#powerrail
      Contact( #Rh_ET21 )
   END_RUNG wire#w1
   RUNG wire#powerrail
      Contact( #Rh_ET106 )
   END_RUNG wire#w1
   RUNG wire#powerrail
      Contact( #MA_Ir_Mid_Bajando )
   END_RUNG wire#w1
   RUNG wire#powerrail
      Contact( #ELEV_PosMid )
   END_RUNG wire#w3
   RUNG wire#powerrail
      Contact( #Rh_ET41 )
      wire#w2
      Contact( #ELEV_PosUp )
   END_RUNG wire#w3
   RUNG wire#powerrail
      Contact( #Rh_ET21 )
   END_RUNG wire#w2
   RUNG wire#powerrail
      Contact( #Rh_ET106 )
   END_RUNG wire#w2
   RUNG wire#powerrail
      Contact( #MA_Ir_Mid_Subiendo )
   END_RUNG wire#w2
   RUNG wire#powerrail
      Contact( #EstadoZona.Manual_CBx )
   END_RUNG wire#w3
   RUNG wire#powerrail
      Contact( #Rh_ET00 )
   END_RUNG wire#w3
   // the same network as SCL:
   IF (#Rh_ET41 OR #Rh_ET21 OR #Rh_ET106 OR #MA_Ir_Mid_Bajando) AND #ELEV_PosDw THEN
       #CambioDir_SubidaBajada := TRUE;   // SR flip-flop
   END_IF;
   IF #ELEV_PosMid OR ((#Rh_ET41 OR #Rh_ET21 OR #Rh_ET106 OR #MA_Ir_Mid_Subiendo) AND #ELEV_PosUp) OR #EstadoZona.Manual_CBx OR #Rh_ET00 THEN
       #CambioDir_SubidaBajada := FALSE;
   END_IF;
END_REGION

REGION Network 60: SALIDAS - Horquilla - Ir Adelante
   RUNG wire#powerrail
      Contact( #Rh_ET13 )
      wire#w1
      I_Contact( #MA_Ir_Atras )
      I_Contact( #HORQ_Extendida )
      Contact( #HORQ_SegExtendida )
      I_Contact( #EnMovimiento_Tx )
      Contact( #EstadoZona.Marcha_CBx )
      I_Contact( #EstadoMAQ.Error_MAQx )
      I_Contact( #Error_Tx )
      Coil( #MA_Ir_Adelante )
   END_RUNG
   RUNG wire#powerrail
      Contact( #Rh_ET22 )
   END_RUNG wire#w1
   RUNG wire#powerrail
      Contact( #Rh_ET15 )
   END_RUNG wire#w1
   RUNG wire#powerrail
      Contact( #Rh_ET101 )
   END_RUNG wire#w1
   RUNG wire#powerrail
      Contact( #Rh_ET104 )
   END_RUNG wire#w1
   // the same network as SCL:
   #MA_Ir_Adelante := (#Rh_ET13 OR #Rh_ET22 OR #Rh_ET15 OR #Rh_ET101 OR #Rh_ET104) AND NOT #MA_Ir_Atras AND NOT #HORQ_Extendida AND #HORQ_SegExtendida AND NOT #EnMovimiento_Tx AND #EstadoZona.Marcha_CBx AND NOT #EstadoMAQ.Error_MAQx AND NOT #Error_Tx;
END_REGION

REGION Network 61: SALIDAS - Horquilla - Ir Atras
   RUNG wire#powerrail
      Contact( #Rh_ET11 )
      wire#w1
      I_Contact( #MA_Ir_Adelante )
      I_Contact( #HORQ_Recogida )
      Contact( #HORQ_SegRecogida )
      I_Contact( #EnMovimiento_Tx )
      Contact( #EstadoZona.Marcha_CBx )
      I_Contact( #EstadoMAQ.Error_MAQx )
      I_Contact( #Error_Tx )
      Coil( #MA_Ir_Atras )
   END_RUNG
   RUNG wire#powerrail
      Contact( #Rh_ET31 )
   END_RUNG wire#w1
   RUNG wire#powerrail
      Contact( #Rh_ET42 )
   END_RUNG wire#w1
   RUNG wire#powerrail
      Contact( #Rh_ET52 )
   END_RUNG wire#w1
   RUNG wire#powerrail
      Contact( #Rh_ET102 )
      wire#w2
      Contact( #ELEV_PosDw )
   END_RUNG wire#w1
   RUNG wire#powerrail
      Contact( #Rh_ET103 )
   END_RUNG wire#w2
   RUNG wire#powerrail
      Contact( #Rh_ET107 )
   END_RUNG wire#w1
   // the same network as SCL:
   #MA_Ir_Atras := (#Rh_ET11 OR #Rh_ET31 OR #Rh_ET42 OR #Rh_ET52 OR ((#Rh_ET102 OR #Rh_ET103) AND #ELEV_PosDw) OR #Rh_ET107) AND NOT #MA_Ir_Adelante AND NOT #HORQ_Recogida AND #HORQ_SegRecogida AND NOT #EnMovimiento_Tx AND #EstadoZona.Marcha_CBx AND NOT #EstadoMAQ.Error_MAQx AND NOT #Error_Tx;
END_REGION

REGION Network 62: SALIDAS - Elevacion - Ir DOWN
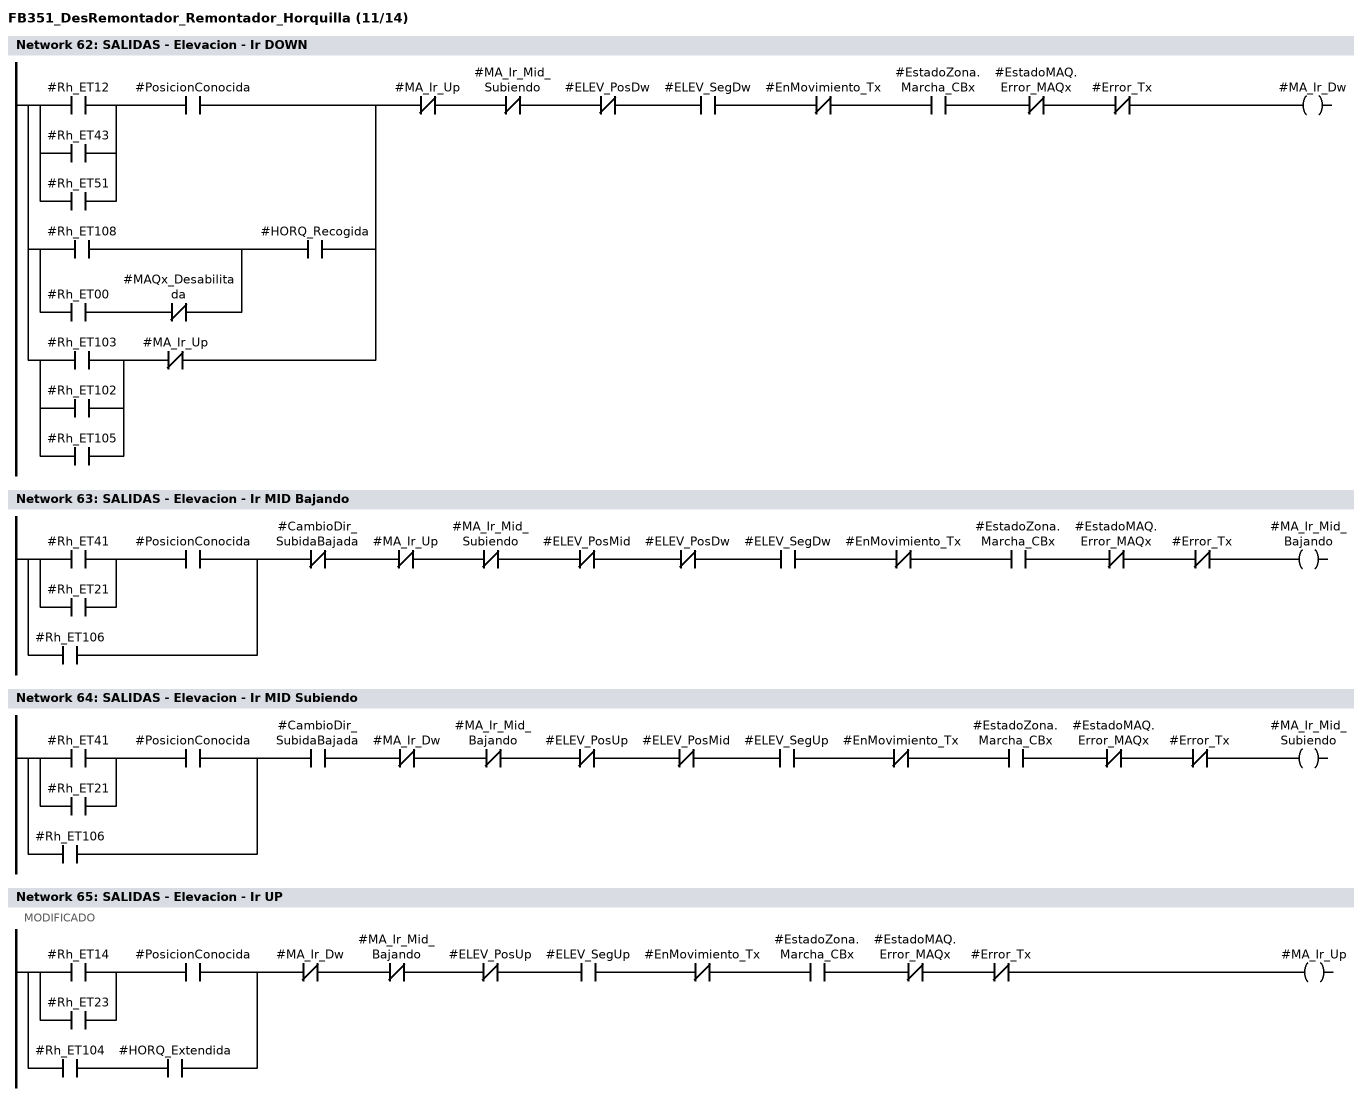
   RUNG wire#powerrail
      Contact( #Rh_ET12 )
      wire#w1
      Contact( #PosicionConocida )
      wire#w2
      I_Contact( #MA_Ir_Up )
      I_Contact( #MA_Ir_Mid_Subiendo )
      I_Contact( #ELEV_PosDw )
      Contact( #ELEV_SegDw )
      I_Contact( #EnMovimiento_Tx )
      Contact( #EstadoZona.Marcha_CBx )
      I_Contact( #EstadoMAQ.Error_MAQx )
      I_Contact( #Error_Tx )
      Coil( #MA_Ir_Dw )
   END_RUNG
   RUNG wire#powerrail
      Contact( #Rh_ET43 )
   END_RUNG wire#w1
   RUNG wire#powerrail
      Contact( #Rh_ET51 )
   END_RUNG wire#w1
   RUNG wire#powerrail
      Contact( #Rh_ET108 )
      wire#w3
      Contact( #HORQ_Recogida )
   END_RUNG wire#w2
   RUNG wire#powerrail
      Contact( #Rh_ET00 )
      I_Contact( #MAQx_Desabilitada )
   END_RUNG wire#w3
   RUNG wire#powerrail
      Contact( #Rh_ET103 )
      wire#w4
      I_Contact( #MA_Ir_Up )
   END_RUNG wire#w2
   RUNG wire#powerrail
      Contact( #Rh_ET102 )
   END_RUNG wire#w4
   RUNG wire#powerrail
      Contact( #Rh_ET105 )
   END_RUNG wire#w4
   // the same network as SCL:
   #MA_Ir_Dw := (((#Rh_ET12 OR #Rh_ET43 OR #Rh_ET51) AND #PosicionConocida) OR ((#Rh_ET108 OR (#Rh_ET00 AND NOT #MAQx_Desabilitada)) AND #HORQ_Recogida) OR ((#Rh_ET103 OR #Rh_ET102 OR #Rh_ET105) AND NOT #MA_Ir_Up)) AND NOT #MA_Ir_Up AND NOT #MA_Ir_Mid_Subiendo AND NOT #ELEV_PosDw AND #ELEV_SegDw AND NOT #EnMovimiento_Tx AND #EstadoZona.Marcha_CBx AND NOT #EstadoMAQ.Error_MAQx AND NOT #Error_Tx;
END_REGION

REGION Network 63: SALIDAS - Elevacion - Ir MID Bajando
   RUNG wire#powerrail
      Contact( #Rh_ET41 )
      wire#w1
      Contact( #PosicionConocida )
      wire#w2
      I_Contact( #CambioDir_SubidaBajada )
      I_Contact( #MA_Ir_Up )
      I_Contact( #MA_Ir_Mid_Subiendo )
      I_Contact( #ELEV_PosMid )
      I_Contact( #ELEV_PosDw )
      Contact( #ELEV_SegDw )
      I_Contact( #EnMovimiento_Tx )
      Contact( #EstadoZona.Marcha_CBx )
      I_Contact( #EstadoMAQ.Error_MAQx )
      I_Contact( #Error_Tx )
      Coil( #MA_Ir_Mid_Bajando )
   END_RUNG
   RUNG wire#powerrail
      Contact( #Rh_ET21 )
   END_RUNG wire#w1
   RUNG wire#powerrail
      Contact( #Rh_ET106 )
   END_RUNG wire#w2
   // the same network as SCL:
   #MA_Ir_Mid_Bajando := (((#Rh_ET41 OR #Rh_ET21) AND #PosicionConocida) OR #Rh_ET106) AND NOT #CambioDir_SubidaBajada AND NOT #MA_Ir_Up AND NOT #MA_Ir_Mid_Subiendo AND NOT #ELEV_PosMid AND NOT #ELEV_PosDw AND #ELEV_SegDw AND NOT #EnMovimiento_Tx AND #EstadoZona.Marcha_CBx AND NOT #EstadoMAQ.Error_MAQx AND NOT #Error_Tx;
END_REGION

REGION Network 64: SALIDAS - Elevacion - Ir MID Subiendo
   RUNG wire#powerrail
      Contact( #Rh_ET41 )
      wire#w1
      Contact( #PosicionConocida )
      wire#w2
      Contact( #CambioDir_SubidaBajada )
      I_Contact( #MA_Ir_Dw )
      I_Contact( #MA_Ir_Mid_Bajando )
      I_Contact( #ELEV_PosUp )
      I_Contact( #ELEV_PosMid )
      Contact( #ELEV_SegUp )
      I_Contact( #EnMovimiento_Tx )
      Contact( #EstadoZona.Marcha_CBx )
      I_Contact( #EstadoMAQ.Error_MAQx )
      I_Contact( #Error_Tx )
      Coil( #MA_Ir_Mid_Subiendo )
   END_RUNG
   RUNG wire#powerrail
      Contact( #Rh_ET21 )
   END_RUNG wire#w1
   RUNG wire#powerrail
      Contact( #Rh_ET106 )
   END_RUNG wire#w2
   // the same network as SCL:
   #MA_Ir_Mid_Subiendo := (((#Rh_ET41 OR #Rh_ET21) AND #PosicionConocida) OR #Rh_ET106) AND #CambioDir_SubidaBajada AND NOT #MA_Ir_Dw AND NOT #MA_Ir_Mid_Bajando AND NOT #ELEV_PosUp AND NOT #ELEV_PosMid AND #ELEV_SegUp AND NOT #EnMovimiento_Tx AND #EstadoZona.Marcha_CBx AND NOT #EstadoMAQ.Error_MAQx AND NOT #Error_Tx;
END_REGION

REGION Network 65: SALIDAS - Elevacion - Ir UP
   // MODIFICADO
   RUNG wire#powerrail
      Contact( #Rh_ET14 )
      wire#w1
      Contact( #PosicionConocida )
      wire#w2
      I_Contact( #MA_Ir_Dw )
      I_Contact( #MA_Ir_Mid_Bajando )
      I_Contact( #ELEV_PosUp )
      Contact( #ELEV_SegUp )
      I_Contact( #EnMovimiento_Tx )
      Contact( #EstadoZona.Marcha_CBx )
      I_Contact( #EstadoMAQ.Error_MAQx )
      I_Contact( #Error_Tx )
      Coil( #MA_Ir_Up )
   END_RUNG
   RUNG wire#powerrail
      Contact( #Rh_ET23 )
   END_RUNG wire#w1
   RUNG wire#powerrail
      Contact( #Rh_ET104 )
      Contact( #HORQ_Extendida )
   END_RUNG wire#w2
   // the same network as SCL:
   #MA_Ir_Up := (((#Rh_ET14 OR #Rh_ET23) AND #PosicionConocida) OR (#Rh_ET104 AND #HORQ_Extendida)) AND NOT #MA_Ir_Dw AND NOT #MA_Ir_Mid_Bajando AND NOT #ELEV_PosUp AND #ELEV_SegUp AND NOT #EnMovimiento_Tx AND #EstadoZona.Marcha_CBx AND NOT #EstadoMAQ.Error_MAQx AND NOT #Error_Tx;
END_REGION

REGION Network 66: SALIDAS - Hoquilla - Velocidad Rapida
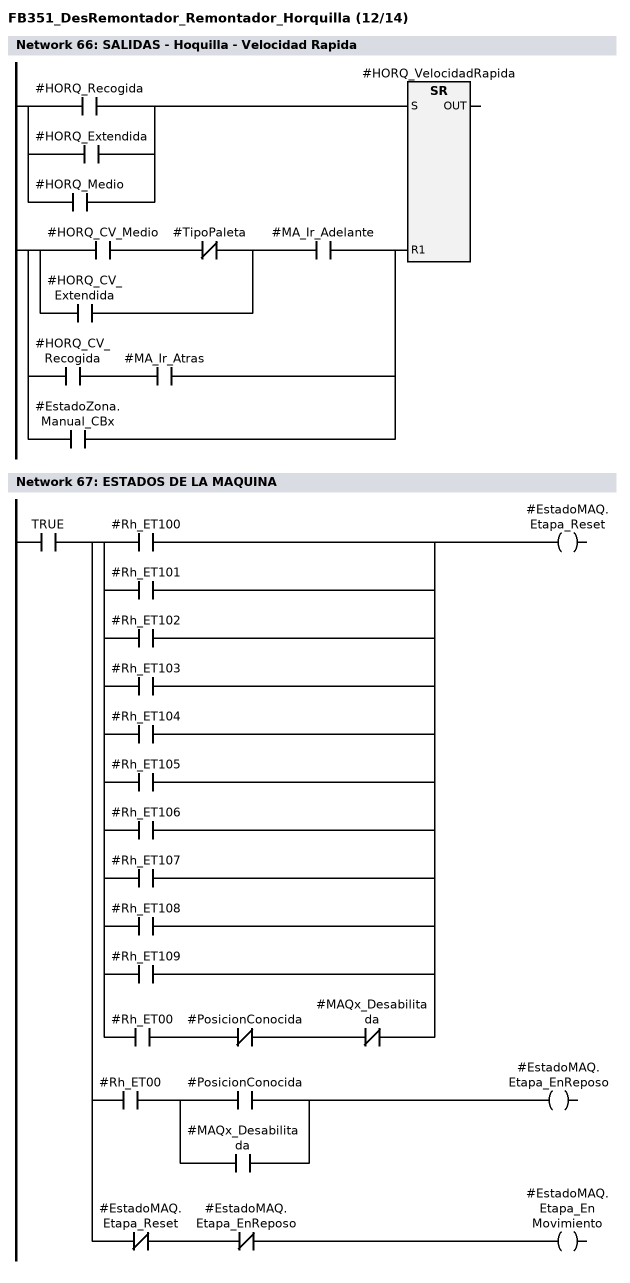
   RUNG wire#powerrail
      Contact( #HORQ_Recogida )
      wire#w1
      S_SR(operand := #HORQ_VelocidadRapida, r1 := wire#w3)
   END_RUNG
   RUNG wire#powerrail
      Contact( #HORQ_Extendida )
   END_RUNG wire#w1
   RUNG wire#powerrail
      Contact( #HORQ_Medio )
   END_RUNG wire#w1
   RUNG wire#powerrail
      Contact( #HORQ_CV_Medio )
      I_Contact( #TipoPaleta )
      wire#w2
      Contact( #MA_Ir_Adelante )
   END_RUNG wire#w3
   RUNG wire#powerrail
      Contact( #HORQ_CV_Extendida )
   END_RUNG wire#w2
   RUNG wire#powerrail
      Contact( #HORQ_CV_Recogida )
      Contact( #MA_Ir_Atras )
   END_RUNG wire#w3
   RUNG wire#powerrail
      Contact( #EstadoZona.Manual_CBx )
   END_RUNG wire#w3
   // the same network as SCL:
   IF #HORQ_Recogida OR #HORQ_Extendida OR #HORQ_Medio THEN
       #HORQ_VelocidadRapida := TRUE;   // SR flip-flop
   END_IF;
   IF (((#HORQ_CV_Medio AND NOT #TipoPaleta) OR #HORQ_CV_Extendida) AND #MA_Ir_Adelante) OR (#HORQ_CV_Recogida AND #MA_Ir_Atras) OR #EstadoZona.Manual_CBx THEN
       #HORQ_VelocidadRapida := FALSE;
   END_IF;
END_REGION

REGION Network 67: ESTADOS DE LA MAQUINA
   RUNG wire#powerrail
      Contact( TRUE )
      wire#w1
      Contact( #Rh_ET100 )
      wire#w2
      Coil( #EstadoMAQ.Etapa_Reset )
   END_RUNG
   RUNG wire#w1
      Contact( #Rh_ET101 )
   END_RUNG wire#w2
   RUNG wire#w1
      Contact( #Rh_ET102 )
   END_RUNG wire#w2
   RUNG wire#w1
      Contact( #Rh_ET103 )
   END_RUNG wire#w2
   RUNG wire#w1
      Contact( #Rh_ET104 )
   END_RUNG wire#w2
   RUNG wire#w1
      Contact( #Rh_ET105 )
   END_RUNG wire#w2
   RUNG wire#w1
      Contact( #Rh_ET106 )
   END_RUNG wire#w2
   RUNG wire#w1
      Contact( #Rh_ET107 )
   END_RUNG wire#w2
   RUNG wire#w1
      Contact( #Rh_ET108 )
   END_RUNG wire#w2
   RUNG wire#w1
      Contact( #Rh_ET109 )
   END_RUNG wire#w2
   RUNG wire#w1
      Contact( #Rh_ET00 )
      I_Contact( #PosicionConocida )
      I_Contact( #MAQx_Desabilitada )
   END_RUNG wire#w2
   RUNG wire#w1
      Contact( #Rh_ET00 )
      wire#w3
      Contact( #PosicionConocida )
      wire#w4
      Coil( #EstadoMAQ.Etapa_EnReposo )
   END_RUNG
   RUNG wire#w3
      Contact( #MAQx_Desabilitada )
   END_RUNG wire#w4
   RUNG wire#w1
      I_Contact( #EstadoMAQ.Etapa_Reset )
      I_Contact( #EstadoMAQ.Etapa_EnReposo )
      Coil( #EstadoMAQ.Etapa_EnMovimiento )
   END_RUNG
   // the same network as SCL:
   #EstadoMAQ.Etapa_Reset := TRUE AND (#Rh_ET100 OR #Rh_ET101 OR #Rh_ET102 OR #Rh_ET103 OR #Rh_ET104 OR #Rh_ET105 OR #Rh_ET106 OR #Rh_ET107 OR #Rh_ET108 OR #Rh_ET109 OR (#Rh_ET00 AND NOT #PosicionConocida AND NOT #MAQx_Desabilitada));
   #EstadoMAQ.Etapa_EnReposo := TRUE AND #Rh_ET00 AND (#PosicionConocida OR #MAQx_Desabilitada);
   #EstadoMAQ.Etapa_EnMovimiento := TRUE AND NOT #EstadoMAQ.Etapa_Reset AND NOT #EstadoMAQ.Etapa_EnReposo;
END_REGION

REGION Network 68: ENTRADAS DE LA MAQUINA
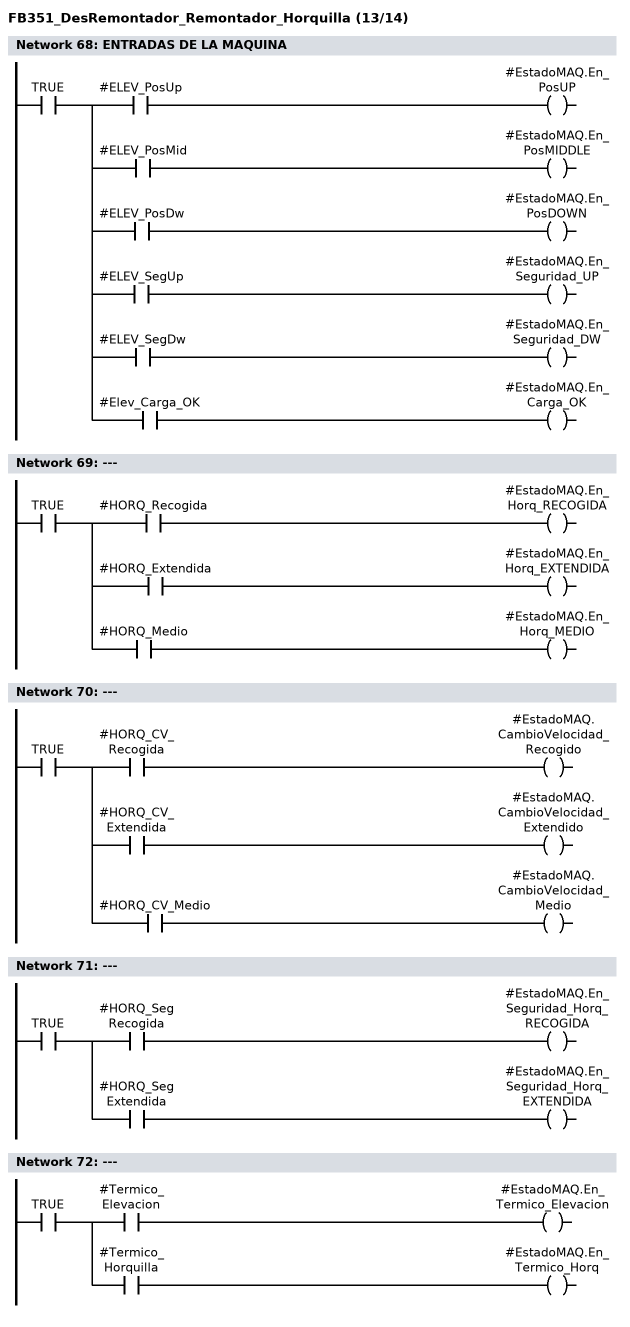
   RUNG wire#powerrail
      Contact( TRUE )
      wire#w1
      Contact( #ELEV_PosUp )
      Coil( #EstadoMAQ.En_PosUP )
   END_RUNG
   RUNG wire#w1
      Contact( #ELEV_PosMid )
      Coil( #EstadoMAQ.En_PosMIDDLE )
   END_RUNG
   RUNG wire#w1
      Contact( #ELEV_PosDw )
      Coil( #EstadoMAQ.En_PosDOWN )
   END_RUNG
   RUNG wire#w1
      Contact( #ELEV_SegUp )
      Coil( #EstadoMAQ.En_Seguridad_UP )
   END_RUNG
   RUNG wire#w1
      Contact( #ELEV_SegDw )
      Coil( #EstadoMAQ.En_Seguridad_DW )
   END_RUNG
   RUNG wire#w1
      Contact( #Elev_Carga_OK )
      Coil( #EstadoMAQ.En_Carga_OK )
   END_RUNG
   // the same network as SCL:
   #EstadoMAQ.En_PosUP := TRUE AND #ELEV_PosUp;
   #EstadoMAQ.En_PosMIDDLE := TRUE AND #ELEV_PosMid;
   #EstadoMAQ.En_PosDOWN := TRUE AND #ELEV_PosDw;
   #EstadoMAQ.En_Seguridad_UP := TRUE AND #ELEV_SegUp;
   #EstadoMAQ.En_Seguridad_DW := TRUE AND #ELEV_SegDw;
   #EstadoMAQ.En_Carga_OK := TRUE AND #Elev_Carga_OK;
END_REGION

REGION Network 69: ---
   RUNG wire#powerrail
      Contact( TRUE )
      wire#w1
      Contact( #HORQ_Recogida )
      Coil( #EstadoMAQ.En_Horq_RECOGIDA )
   END_RUNG
   RUNG wire#w1
      Contact( #HORQ_Extendida )
      Coil( #EstadoMAQ.En_Horq_EXTENDIDA )
   END_RUNG
   RUNG wire#w1
      Contact( #HORQ_Medio )
      Coil( #EstadoMAQ.En_Horq_MEDIO )
   END_RUNG
   // the same network as SCL:
   #EstadoMAQ.En_Horq_RECOGIDA := TRUE AND #HORQ_Recogida;
   #EstadoMAQ.En_Horq_EXTENDIDA := TRUE AND #HORQ_Extendida;
   #EstadoMAQ.En_Horq_MEDIO := TRUE AND #HORQ_Medio;
END_REGION

REGION Network 70: ---
   RUNG wire#powerrail
      Contact( TRUE )
      wire#w1
      Contact( #HORQ_CV_Recogida )
      Coil( #EstadoMAQ.CambioVelocidad_Recogido )
   END_RUNG
   RUNG wire#w1
      Contact( #HORQ_CV_Extendida )
      Coil( #EstadoMAQ.CambioVelocidad_Extendido )
   END_RUNG
   RUNG wire#w1
      Contact( #HORQ_CV_Medio )
      Coil( #EstadoMAQ.CambioVelocidad_Medio )
   END_RUNG
   // the same network as SCL:
   #EstadoMAQ.CambioVelocidad_Recogido := TRUE AND #HORQ_CV_Recogida;
   #EstadoMAQ.CambioVelocidad_Extendido := TRUE AND #HORQ_CV_Extendida;
   #EstadoMAQ.CambioVelocidad_Medio := TRUE AND #HORQ_CV_Medio;
END_REGION

REGION Network 71: ---
   RUNG wire#powerrail
      Contact( TRUE )
      wire#w1
      Contact( #HORQ_SegRecogida )
      Coil( #EstadoMAQ.En_Seguridad_Horq_RECOGIDA )
   END_RUNG
   RUNG wire#w1
      Contact( #HORQ_SegExtendida )
      Coil( #EstadoMAQ.En_Seguridad_Horq_EXTENDIDA )
   END_RUNG
   // the same network as SCL:
   #EstadoMAQ.En_Seguridad_Horq_RECOGIDA := TRUE AND #HORQ_SegRecogida;
   #EstadoMAQ.En_Seguridad_Horq_EXTENDIDA := TRUE AND #HORQ_SegExtendida;
END_REGION

REGION Network 72: ---
   RUNG wire#powerrail
      Contact( TRUE )
      wire#w1
      Contact( #Termico_Elevacion )
      Coil( #EstadoMAQ.En_Termico_Elevacion )
   END_RUNG
   RUNG wire#w1
      Contact( #Termico_Horquilla )
      Coil( #EstadoMAQ.En_Termico_Horq )
   END_RUNG
   // the same network as SCL:
   #EstadoMAQ.En_Termico_Elevacion := TRUE AND #Termico_Elevacion;
   #EstadoMAQ.En_Termico_Horq := TRUE AND #Termico_Horquilla;
END_REGION

REGION Network 73: SALIDAS DE LA MAQUINA
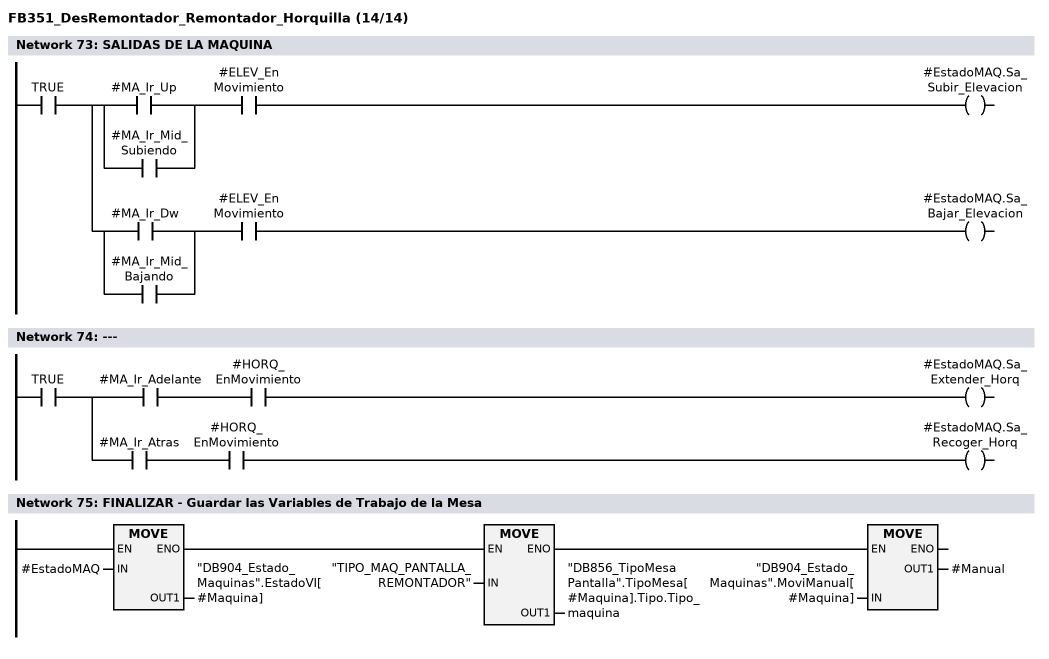
   RUNG wire#powerrail
      Contact( TRUE )
      wire#w1
      Contact( #MA_Ir_Up )
      wire#w2
      Contact( #ELEV_EnMovimiento )
      Coil( #EstadoMAQ.Sa_Subir_Elevacion )
   END_RUNG
   RUNG wire#w1
      Contact( #MA_Ir_Mid_Subiendo )
   END_RUNG wire#w2
   RUNG wire#w1
      Contact( #MA_Ir_Dw )
      wire#w3
      Contact( #ELEV_EnMovimiento )
      Coil( #EstadoMAQ.Sa_Bajar_Elevacion )
   END_RUNG
   RUNG wire#w1
      Contact( #MA_Ir_Mid_Bajando )
   END_RUNG wire#w3
   // the same network as SCL:
   #EstadoMAQ.Sa_Subir_Elevacion := TRUE AND (#MA_Ir_Up OR #MA_Ir_Mid_Subiendo) AND #ELEV_EnMovimiento;
   #EstadoMAQ.Sa_Bajar_Elevacion := TRUE AND (#MA_Ir_Dw OR #MA_Ir_Mid_Bajando) AND #ELEV_EnMovimiento;
END_REGION

REGION Network 74: ---
   RUNG wire#powerrail
      Contact( TRUE )
      wire#w1
      Contact( #MA_Ir_Adelante )
      Contact( #HORQ_EnMovimiento )
      Coil( #EstadoMAQ.Sa_Extender_Horq )
   END_RUNG
   RUNG wire#w1
      Contact( #MA_Ir_Atras )
      Contact( #HORQ_EnMovimiento )
      Coil( #EstadoMAQ.Sa_Recoger_Horq )
   END_RUNG
   // the same network as SCL:
   #EstadoMAQ.Sa_Extender_Horq := TRUE AND #MA_Ir_Adelante AND #HORQ_EnMovimiento;
   #EstadoMAQ.Sa_Recoger_Horq := TRUE AND #MA_Ir_Atras AND #HORQ_EnMovimiento;
END_REGION

REGION Network 75: FINALIZAR - Guardar las Variables de Trabajo de la Mesa
   RUNG wire#powerrail
      Move(in := #EstadoMAQ, out1 => "DB904_Estado_Maquinas".EstadoVI[#Maquina])
      Move(in := "TIPO_MAQ_PANTALLA_REMONTADOR", out1 => "DB856_TipoMesaPantalla".TipoMesa[#Maquina].Tipo.Tipo_maquina)
      Move(in := "DB904_Estado_Maquinas".MoviManual[#Maquina], out1 => #Manual)
   END_RUNG
   // the same network as SCL:
   "DB904_Estado_Maquinas".EstadoVI[#Maquina] := #EstadoMAQ;
   "DB856_TipoMesaPantalla".TipoMesa[#Maquina].Tipo.Tipo_maquina := "TIPO_MAQ_PANTALLA_REMONTADOR";
   #Manual := "DB904_Estado_Maquinas".MoviManual[#Maquina];
END_REGION
END_FUNCTION_BLOCK

FUNCTION_BLOCK "FB364_Mesa_ApiladorBandejas_ULMA"   // FB364, LAD
TITLE = Control del Ramal de Salidas
{ S7_Optimized_Access := 'FALSE' }
AUTHOR : TE_FSS
NAME : 20160211
VERSION : 3.2
// stored: AutoNumber false, SetENOAutomatically false
   VAR_INPUT
      Mesa : UInt;   // Mesa de la FB
      Error_Tx : Bool;   // Error en el Tx
      pHsMx : Bool;   // pHs de la Mesa
      Avance_Tx : Bool;   // Avance de Tx
      TP_Up : Bool;   // Detector de TP Arriba
      TP_Down : Bool;   // Detector de TP Abajo
      PRV_AVTF_Bandeja : Bool;   // E1 >> Aviso de Entrada de Bandeja
      PRV_AVTF_Pila_Bandejas : Bool;   // E1 >> Aviso de Entrada de Pila
      NXT_Carga_OK : Bool;   // S3 >> Permiso de Salida
      DejarCargaEnMesa : Bool;   // Dejar la Bandeja En la Mesa
      V_pHsMx : Int;   // Valor de Presencia
      V_ApHsMx : Int;   // Valor de Ausencia
      V_TOut_Atasco : Int;   // Valor de TimeOut de Entrada
      V_TOut_TP : Int;   // Valor de TmeOut de Tope
      V_Vaciado : Int;   // Valor de Vaciado
   END_VAR
   VAR_OUTPUT
      PRV_Carga_OK : Bool;   // E1 >> Permiso de Entrada
      NXT_AVTF_Bandeja : Bool;   // S3 >> Aviso de Salida de Bandeja
      NXT_AVTF_Pila : Bool;   // S3 >> Aviso de Salida de Pila
   END_VAR
   VAR_IN_OUT
      Ord_ApilarBandeja : Bool;   // Orden de Apilar Bandeja
      Ord_SalidaPila : Bool;   // Orden de Salida de Pila
   END_VAR
   VAR
      Mx_ET00 : Bool;
      Mx_ET01 : Bool;
      Mx_ET02 : Bool;
      Mx_ET10 : Bool;
      Mx_ET11 : Bool;
      Mx_ET50 : Bool;   // Descarga de Bandeja
      Mx_ET51 : Bool;   // Descarga de Bandeja
      Mx_ET60 : Bool;   // Ciclo Apilado
      Mx_ET61 : Bool;   // Ciclo Apilado
      Mx_ET70 : Bool;   // Descarga De Pila de Bandejas
      Mx_ET71 : Bool;   // Descarga De Pila de Bandejas
      STAT_NXT_AVTF_Bandeja : Bool;   // Interna >> Aviso de Salida de Bandeja
      STAT_NXT_AVTF_Pila : Bool;   // Interna >> Aviso de Salida de Pila
      MA_Avanzar_Tx : Bool;
      MA_Parar_Tx : Bool;
      MA_Subir_TP : Bool;
      MA_Bajar_TP : Bool;
      CNT_pHsMx { S7_SetPoint := 'True'} : "FB910_CNT_UHS";
      CNT_ApHsMx { S7_SetPoint := 'True'} : "FB910_CNT_UHS";
      TMP_Vaciado { S7_SetPoint := 'True'} : "FB910_CNT_UHS";
      TOut_Atasco { S7_SetPoint := 'True'} : "FB910_CNT_UHS";
      TOut_Subir_TP { S7_SetPoint := 'True'} : "FB910_CNT_UHS";
      TOut_Bajar_TP { S7_SetPoint := 'True'} : "FB910_CNT_UHS";
   END_VAR
   VAR_TEMP
      EstadoZona : "EstadoZona";   // Estado de Zona de la Mesa
      EstadoVI : "EstadosMesa";   // Estado del Vehiculo Inteliguente de la Mesa
      ConfigFB : "UDT_ConfigFB";   // Configuracion de la FB de la Mesa
      Aux_ET00 : Bool;
   END_VAR
BEGIN

REGION Network 1: INICIALIZAR - Recoger las Variables de Estado de la Mesa
   // Se recoge - Estado_CBx
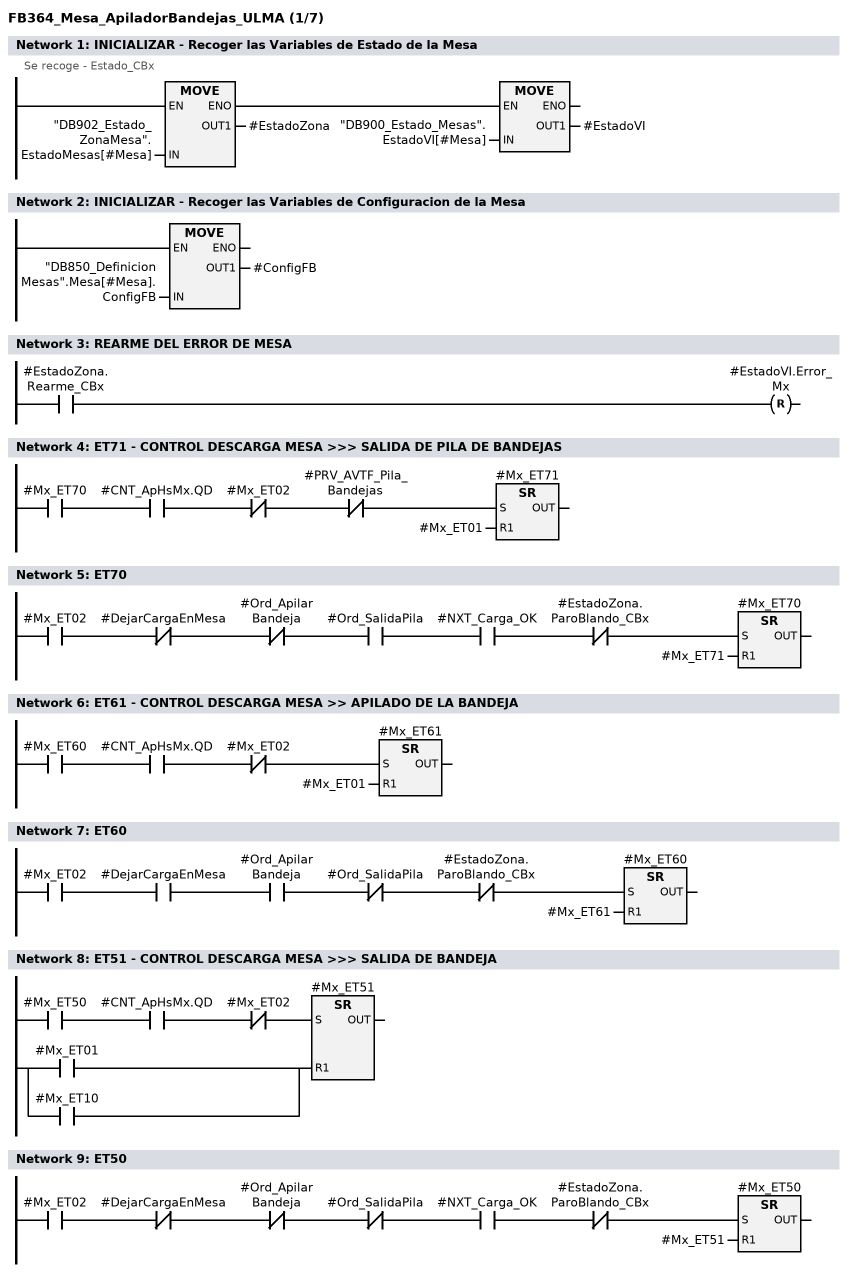
   RUNG wire#powerrail
      Move(in := "DB902_Estado_ZonaMesa".EstadoMesas[#Mesa], out1 => #EstadoZona)
      Move(in := "DB900_Estado_Mesas".EstadoVI[#Mesa], out1 => #EstadoVI)
   END_RUNG
   // the same network as SCL:
   #EstadoZona := "DB902_Estado_ZonaMesa".EstadoMesas[#Mesa];
   #EstadoVI := "DB900_Estado_Mesas".EstadoVI[#Mesa];
END_REGION

REGION Network 2: INICIALIZAR - Recoger las Variables de Configuracion de la Mesa
   RUNG wire#powerrail
      Move(in := "DB850_DefinicionMesas".Mesa[#Mesa].ConfigFB, out1 => #ConfigFB)
   END_RUNG
   // the same network as SCL:
   #ConfigFB := "DB850_DefinicionMesas".Mesa[#Mesa].ConfigFB;
END_REGION

REGION Network 3: REARME DEL ERROR DE MESA
   RUNG wire#powerrail
      Contact( #EstadoZona.Rearme_CBx )
      R_Coil( #EstadoVI.Error_Mx )
   END_RUNG
   // the same network as SCL:
   IF #EstadoZona.Rearme_CBx THEN #EstadoVI.Error_Mx := FALSE; END_IF;
END_REGION

REGION Network 4: ET71 - CONTROL DESCARGA MESA >>> SALIDA DE PILA DE BANDEJAS
   RUNG wire#powerrail
      Contact( #Mx_ET70 )
      Contact( #CNT_ApHsMx.QD )
      I_Contact( #Mx_ET02 )
      I_Contact( #PRV_AVTF_Pila_Bandejas )
      S_SR(operand := #Mx_ET71, r1 := #Mx_ET01)
   END_RUNG
   // the same network as SCL:
   IF #Mx_ET70 AND #CNT_ApHsMx.QD AND NOT #Mx_ET02 AND NOT #PRV_AVTF_Pila_Bandejas THEN
       #Mx_ET71 := TRUE;   // SR flip-flop
   END_IF;
   IF #Mx_ET01 THEN #Mx_ET71 := FALSE; END_IF;
END_REGION

REGION Network 5: ET70
   RUNG wire#powerrail
      Contact( #Mx_ET02 )
      I_Contact( #DejarCargaEnMesa )
      I_Contact( #Ord_ApilarBandeja )
      Contact( #Ord_SalidaPila )
      Contact( #NXT_Carga_OK )
      I_Contact( #EstadoZona.ParoBlando_CBx )
      S_SR(operand := #Mx_ET70, r1 := #Mx_ET71)
   END_RUNG
   // the same network as SCL:
   IF #Mx_ET02 AND NOT #DejarCargaEnMesa AND NOT #Ord_ApilarBandeja AND #Ord_SalidaPila AND #NXT_Carga_OK AND NOT #EstadoZona.ParoBlando_CBx THEN
       #Mx_ET70 := TRUE;   // SR flip-flop
   END_IF;
   IF #Mx_ET71 THEN #Mx_ET70 := FALSE; END_IF;
END_REGION

REGION Network 6: ET61 - CONTROL DESCARGA MESA >> APILADO DE LA BANDEJA
   RUNG wire#powerrail
      Contact( #Mx_ET60 )
      Contact( #CNT_ApHsMx.QD )
      I_Contact( #Mx_ET02 )
      S_SR(operand := #Mx_ET61, r1 := #Mx_ET01)
   END_RUNG
   // the same network as SCL:
   IF #Mx_ET60 AND #CNT_ApHsMx.QD AND NOT #Mx_ET02 THEN
       #Mx_ET61 := TRUE;   // SR flip-flop
   END_IF;
   IF #Mx_ET01 THEN #Mx_ET61 := FALSE; END_IF;
END_REGION

REGION Network 7: ET60
   RUNG wire#powerrail
      Contact( #Mx_ET02 )
      Contact( #DejarCargaEnMesa )
      Contact( #Ord_ApilarBandeja )
      I_Contact( #Ord_SalidaPila )
      I_Contact( #EstadoZona.ParoBlando_CBx )
      S_SR(operand := #Mx_ET60, r1 := #Mx_ET61)
   END_RUNG
   // the same network as SCL:
   IF #Mx_ET02 AND #DejarCargaEnMesa AND #Ord_ApilarBandeja AND NOT #Ord_SalidaPila AND NOT #EstadoZona.ParoBlando_CBx THEN
       #Mx_ET60 := TRUE;   // SR flip-flop
   END_IF;
   IF #Mx_ET61 THEN #Mx_ET60 := FALSE; END_IF;
END_REGION

REGION Network 8: ET51 - CONTROL DESCARGA MESA >>> SALIDA DE BANDEJA
   RUNG wire#powerrail
      Contact( #Mx_ET50 )
      Contact( #CNT_ApHsMx.QD )
      I_Contact( #Mx_ET02 )
      S_SR(operand := #Mx_ET51, r1 := wire#w1)
   END_RUNG
   RUNG wire#powerrail
      Contact( #Mx_ET01 )
   END_RUNG wire#w1
   RUNG wire#powerrail
      Contact( #Mx_ET10 )
   END_RUNG wire#w1
   // the same network as SCL:
   IF #Mx_ET50 AND #CNT_ApHsMx.QD AND NOT #Mx_ET02 THEN
       #Mx_ET51 := TRUE;   // SR flip-flop
   END_IF;
   IF #Mx_ET01 OR #Mx_ET10 THEN #Mx_ET51 := FALSE; END_IF;
END_REGION

REGION Network 9: ET50
   RUNG wire#powerrail
      Contact( #Mx_ET02 )
      I_Contact( #DejarCargaEnMesa )
      I_Contact( #Ord_ApilarBandeja )
      I_Contact( #Ord_SalidaPila )
      Contact( #NXT_Carga_OK )
      I_Contact( #EstadoZona.ParoBlando_CBx )
      S_SR(operand := #Mx_ET50, r1 := #Mx_ET51)
   END_RUNG
   // the same network as SCL:
   IF #Mx_ET02 AND NOT #DejarCargaEnMesa AND NOT #Ord_ApilarBandeja AND NOT #Ord_SalidaPila AND #NXT_Carga_OK AND NOT #EstadoZona.ParoBlando_CBx THEN
       #Mx_ET50 := TRUE;   // SR flip-flop
   END_IF;
   IF #Mx_ET51 THEN #Mx_ET50 := FALSE; END_IF;
END_REGION

REGION Network 10: ET02 - ESTADO REPOSO CARGADA
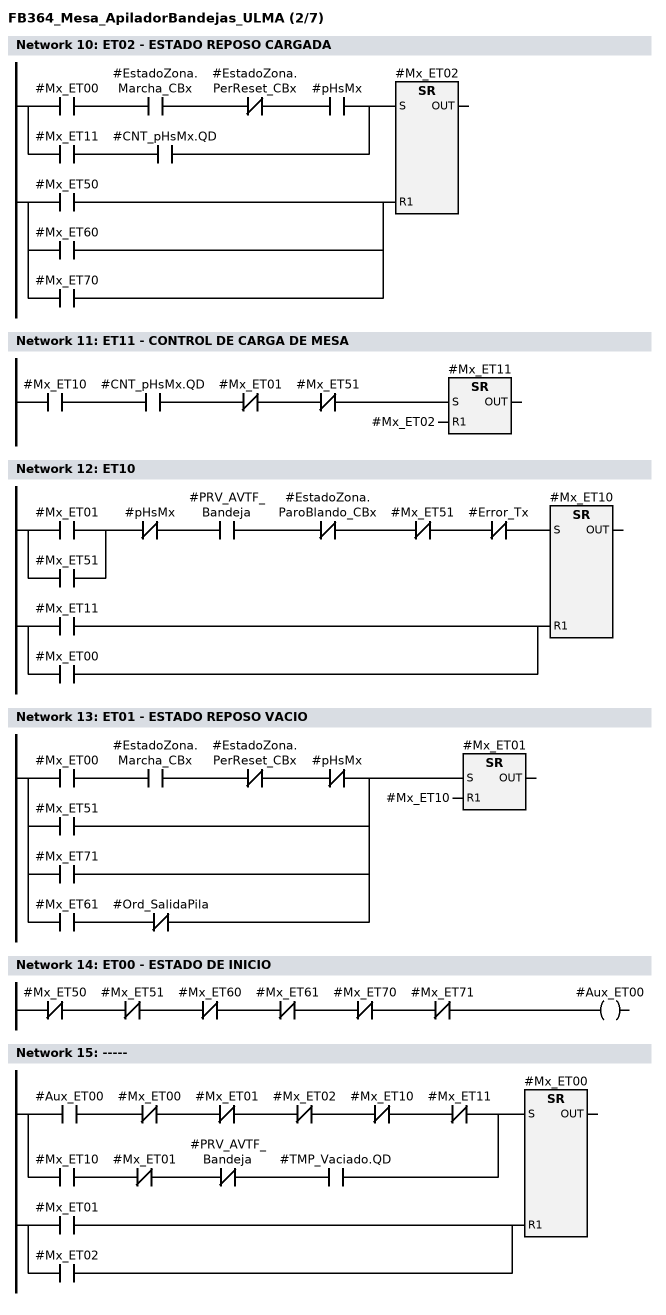
   RUNG wire#powerrail
      Contact( #Mx_ET00 )
      Contact( #EstadoZona.Marcha_CBx )
      I_Contact( #EstadoZona.PerReset_CBx )
      Contact( #pHsMx )
      wire#w1
      S_SR(operand := #Mx_ET02, r1 := wire#w2)
   END_RUNG
   RUNG wire#powerrail
      Contact( #Mx_ET11 )
      Contact( #CNT_pHsMx.QD )
   END_RUNG wire#w1
   RUNG wire#powerrail
      Contact( #Mx_ET50 )
   END_RUNG wire#w2
   RUNG wire#powerrail
      Contact( #Mx_ET60 )
   END_RUNG wire#w2
   RUNG wire#powerrail
      Contact( #Mx_ET70 )
   END_RUNG wire#w2
   // the same network as SCL:
   IF (#Mx_ET00 AND #EstadoZona.Marcha_CBx AND NOT #EstadoZona.PerReset_CBx AND #pHsMx) OR (#Mx_ET11 AND #CNT_pHsMx.QD) THEN
       #Mx_ET02 := TRUE;   // SR flip-flop
   END_IF;
   IF #Mx_ET50 OR #Mx_ET60 OR #Mx_ET70 THEN #Mx_ET02 := FALSE; END_IF;
END_REGION

REGION Network 11: ET11 - CONTROL DE CARGA DE MESA
   RUNG wire#powerrail
      Contact( #Mx_ET10 )
      Contact( #CNT_pHsMx.QD )
      I_Contact( #Mx_ET01 )
      I_Contact( #Mx_ET51 )
      S_SR(operand := #Mx_ET11, r1 := #Mx_ET02)
   END_RUNG
   // the same network as SCL:
   IF #Mx_ET10 AND #CNT_pHsMx.QD AND NOT #Mx_ET01 AND NOT #Mx_ET51 THEN
       #Mx_ET11 := TRUE;   // SR flip-flop
   END_IF;
   IF #Mx_ET02 THEN #Mx_ET11 := FALSE; END_IF;
END_REGION

REGION Network 12: ET10
   RUNG wire#powerrail
      Contact( #Mx_ET01 )
      wire#w1
      I_Contact( #pHsMx )
      Contact( #PRV_AVTF_Bandeja )
      I_Contact( #EstadoZona.ParoBlando_CBx )
      I_Contact( #Mx_ET51 )
      I_Contact( #Error_Tx )
      S_SR(operand := #Mx_ET10, r1 := wire#w2)
   END_RUNG
   RUNG wire#powerrail
      Contact( #Mx_ET51 )
   END_RUNG wire#w1
   RUNG wire#powerrail
      Contact( #Mx_ET11 )
   END_RUNG wire#w2
   RUNG wire#powerrail
      Contact( #Mx_ET00 )
   END_RUNG wire#w2
   // the same network as SCL:
   IF (#Mx_ET01 OR #Mx_ET51) AND NOT #pHsMx AND #PRV_AVTF_Bandeja AND NOT #EstadoZona.ParoBlando_CBx AND NOT #Mx_ET51 AND NOT #Error_Tx THEN
       #Mx_ET10 := TRUE;   // SR flip-flop
   END_IF;
   IF #Mx_ET11 OR #Mx_ET00 THEN #Mx_ET10 := FALSE; END_IF;
END_REGION

REGION Network 13: ET01 - ESTADO REPOSO VACIO
   RUNG wire#powerrail
      Contact( #Mx_ET00 )
      Contact( #EstadoZona.Marcha_CBx )
      I_Contact( #EstadoZona.PerReset_CBx )
      I_Contact( #pHsMx )
      wire#w1
      S_SR(operand := #Mx_ET01, r1 := #Mx_ET10)
   END_RUNG
   RUNG wire#powerrail
      Contact( #Mx_ET51 )
   END_RUNG wire#w1
   RUNG wire#powerrail
      Contact( #Mx_ET71 )
   END_RUNG wire#w1
   RUNG wire#powerrail
      Contact( #Mx_ET61 )
      I_Contact( #Ord_SalidaPila )
   END_RUNG wire#w1
   // the same network as SCL:
   IF (#Mx_ET00 AND #EstadoZona.Marcha_CBx AND NOT #EstadoZona.PerReset_CBx AND NOT #pHsMx) OR #Mx_ET51 OR #Mx_ET71 OR (#Mx_ET61 AND NOT #Ord_SalidaPila) THEN
       #Mx_ET01 := TRUE;   // SR flip-flop
   END_IF;
   IF #Mx_ET10 THEN #Mx_ET01 := FALSE; END_IF;
END_REGION

REGION Network 14: ET00 - ESTADO DE INICIO
   RUNG wire#powerrail
      I_Contact( #Mx_ET50 )
      I_Contact( #Mx_ET51 )
      I_Contact( #Mx_ET60 )
      I_Contact( #Mx_ET61 )
      I_Contact( #Mx_ET70 )
      I_Contact( #Mx_ET71 )
      Coil( #Aux_ET00 )
   END_RUNG
   // the same network as SCL:
   #Aux_ET00 := NOT #Mx_ET50 AND NOT #Mx_ET51 AND NOT #Mx_ET60 AND NOT #Mx_ET61 AND NOT #Mx_ET70 AND NOT #Mx_ET71;
END_REGION

REGION Network 15: -----
   RUNG wire#powerrail
      Contact( #Aux_ET00 )
      I_Contact( #Mx_ET00 )
      I_Contact( #Mx_ET01 )
      I_Contact( #Mx_ET02 )
      I_Contact( #Mx_ET10 )
      I_Contact( #Mx_ET11 )
      wire#w1
      S_SR(operand := #Mx_ET00, r1 := wire#w2)
   END_RUNG
   RUNG wire#powerrail
      Contact( #Mx_ET10 )
      I_Contact( #Mx_ET01 )
      I_Contact( #PRV_AVTF_Bandeja )
      Contact( #TMP_Vaciado.QD )
   END_RUNG wire#w1
   RUNG wire#powerrail
      Contact( #Mx_ET01 )
   END_RUNG wire#w2
   RUNG wire#powerrail
      Contact( #Mx_ET02 )
   END_RUNG wire#w2
   // the same network as SCL:
   IF (#Aux_ET00 AND NOT #Mx_ET00 AND NOT #Mx_ET01 AND NOT #Mx_ET02 AND NOT #Mx_ET10 AND NOT #Mx_ET11) OR (#Mx_ET10 AND NOT #Mx_ET01 AND NOT #PRV_AVTF_Bandeja AND #TMP_Vaciado.QD) THEN
       #Mx_ET00 := TRUE;   // SR flip-flop
   END_IF;
   IF #Mx_ET01 OR #Mx_ET02 THEN #Mx_ET00 := FALSE; END_IF;
END_REGION

REGION Network 16: CONTADOR DE PRESENCIA
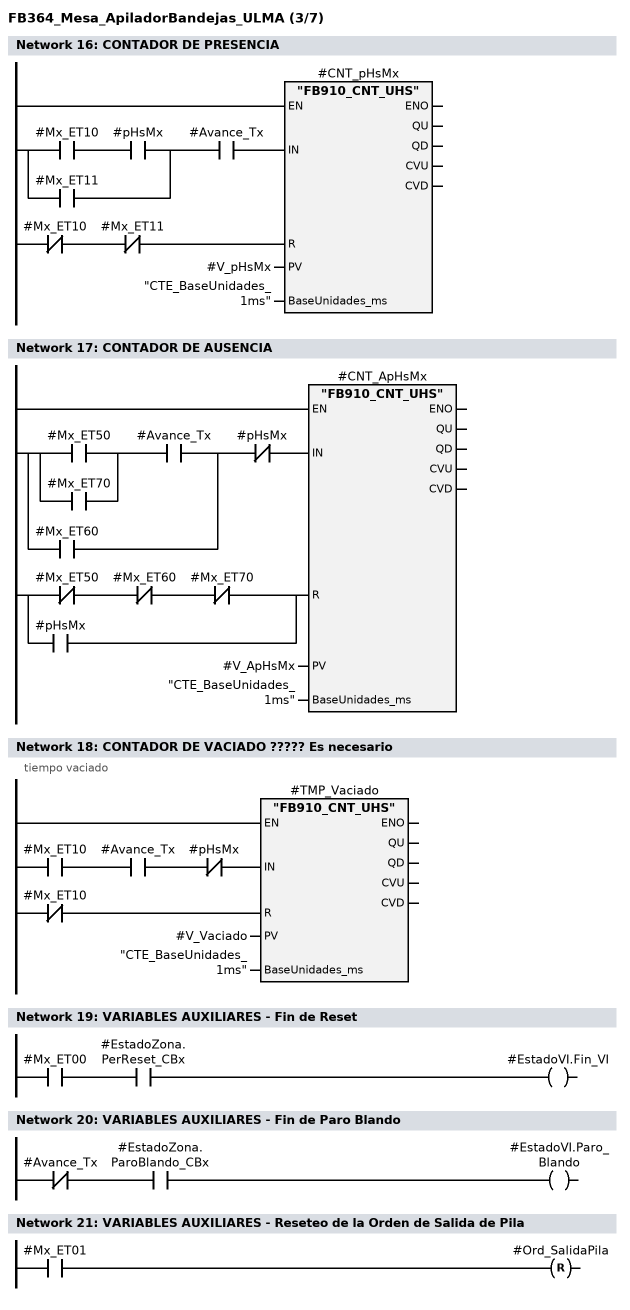
   RUNG wire#powerrail
      #CNT_pHsMx(IN := wire#w2, R := wire#w3, PV := #V_pHsMx, BaseUnidades_ms := "CTE_BaseUnidades_1ms", QU =>, QD =>, CVU =>, CVD =>)
   END_RUNG
   RUNG wire#powerrail
      Contact( #Mx_ET10 )
      Contact( #pHsMx )
      wire#w1
      Contact( #Avance_Tx )
   END_RUNG wire#w2
   RUNG wire#powerrail
      Contact( #Mx_ET11 )
   END_RUNG wire#w1
   RUNG wire#powerrail
      I_Contact( #Mx_ET10 )
      I_Contact( #Mx_ET11 )
   END_RUNG wire#w3
   // the same network as SCL:
   #CNT_pHsMx(IN := ((#Mx_ET10 AND #pHsMx) OR #Mx_ET11) AND #Avance_Tx,   // "FB910_CNT_UHS"
              R := NOT #Mx_ET10 AND NOT #Mx_ET11,
              PV := #V_pHsMx,
              BaseUnidades_ms := "CTE_BaseUnidades_1ms");
END_REGION

REGION Network 17: CONTADOR DE AUSENCIA
   RUNG wire#powerrail
      #CNT_ApHsMx(IN := wire#w3, R := wire#w4, PV := #V_ApHsMx, BaseUnidades_ms := "CTE_BaseUnidades_1ms", QU =>, QD =>, CVU =>, CVD =>)
   END_RUNG
   RUNG wire#powerrail
      Contact( #Mx_ET50 )
      wire#w1
      Contact( #Avance_Tx )
      wire#w2
      I_Contact( #pHsMx )
   END_RUNG wire#w3
   RUNG wire#powerrail
      Contact( #Mx_ET70 )
   END_RUNG wire#w1
   RUNG wire#powerrail
      Contact( #Mx_ET60 )
   END_RUNG wire#w2
   RUNG wire#powerrail
      I_Contact( #Mx_ET50 )
      I_Contact( #Mx_ET60 )
      I_Contact( #Mx_ET70 )
   END_RUNG wire#w4
   RUNG wire#powerrail
      Contact( #pHsMx )
   END_RUNG wire#w4
   // the same network as SCL:
   #CNT_ApHsMx(IN := (((#Mx_ET50 OR #Mx_ET70) AND #Avance_Tx) OR #Mx_ET60) AND NOT #pHsMx,   // "FB910_CNT_UHS"
               R := (NOT #Mx_ET50 AND NOT #Mx_ET60 AND NOT #Mx_ET70) OR #pHsMx,
               PV := #V_ApHsMx,
               BaseUnidades_ms := "CTE_BaseUnidades_1ms");
END_REGION

REGION Network 18: CONTADOR DE VACIADO ????? Es necesario
   // tiempo vaciado
   RUNG wire#powerrail
      #TMP_Vaciado(IN := wire#w1, R := wire#w2, PV := #V_Vaciado, BaseUnidades_ms := "CTE_BaseUnidades_1ms", QU =>, QD =>, CVU =>, CVD =>)
   END_RUNG
   RUNG wire#powerrail
      Contact( #Mx_ET10 )
      Contact( #Avance_Tx )
      I_Contact( #pHsMx )
   END_RUNG wire#w1
   RUNG wire#powerrail
      I_Contact( #Mx_ET10 )
   END_RUNG wire#w2
   // the same network as SCL:
   #TMP_Vaciado(IN := #Mx_ET10 AND #Avance_Tx AND NOT #pHsMx,   // "FB910_CNT_UHS"
                R := NOT #Mx_ET10,
                PV := #V_Vaciado,
                BaseUnidades_ms := "CTE_BaseUnidades_1ms");
END_REGION

REGION Network 19: VARIABLES AUXILIARES - Fin de Reset
   RUNG wire#powerrail
      Contact( #Mx_ET00 )
      Contact( #EstadoZona.PerReset_CBx )
      Coil( #EstadoVI.Fin_VI )
   END_RUNG
   // the same network as SCL:
   #EstadoVI.Fin_VI := #Mx_ET00 AND #EstadoZona.PerReset_CBx;
END_REGION

REGION Network 20: VARIABLES AUXILIARES - Fin de Paro Blando
   RUNG wire#powerrail
      I_Contact( #Avance_Tx )
      Contact( #EstadoZona.ParoBlando_CBx )
      Coil( #EstadoVI.Paro_Blando )
   END_RUNG
   // the same network as SCL:
   #EstadoVI.Paro_Blando := NOT #Avance_Tx AND #EstadoZona.ParoBlando_CBx;
END_REGION

REGION Network 21: VARIABLES AUXILIARES - Reseteo de la Orden de Salida de Pila
   RUNG wire#powerrail
      Contact( #Mx_ET01 )
      R_Coil( #Ord_SalidaPila )
   END_RUNG
   // the same network as SCL:
   IF #Mx_ET01 THEN #Ord_SalidaPila := FALSE; END_IF;
END_REGION

REGION Network 22: VARIABLES AUXILIARES - Permiso de Entrada - PRV_Carga_OK
